// TIA Portal V17 export
// export: Created 2025-07-01T14:25:34.6961243Z, ExportSetting WithDefaults, DisplayName Totally Integrated Automation Portal, DisplayVersion V17 Update 8, DisplayName TIA Portal Openness, DisplayVersion V17 Update 8, DisplayName TIA Portal Version Control Interface, DisplayVersion V17, DisplayName SINAMICS Startdrive Advanced, DisplayVersion V17 SP2, DisplayName SINAMICS Startdrive G110M, G120, G120C, G120D, G120P, G115D, DisplayVersion V17 SP2, DisplayName SINAMICS Startdrive G130, G150, S120, S150, SINAMICS MV, S210, DisplayVersion V17 SP2, DisplayName STEP 7 Professional, DisplayVersion V17 Update 8, DisplayName SINUMERIK ONE STEP 7 Toolbox, DisplayVersion V17 Update 12, DisplayName SINUMERIK ONE PLC Basic Program Plus, DisplayVersion V17 Update 12, DisplayName SINUMERIK 840D sl STEP 7 Toolbox, DisplayVersion V17 Update 12, DisplayName STEP 7 Safety, DisplayVersion V17 Update 6, DisplayName WinCC Advanced, DisplayVersion V17 Update 8
FUNCTION "FC342_NCK_M_CH1_UNIT_1_STA_0" : Void   // FC342, LAD
TITLE = Channel 1 data
{ S7_Optimized_Access := 'FALSE' }
AUTHOR : ETXETAR
VERSION : 1.0
// stored: AutoNumber false, IsIECCheckEnabled false, SetENOAutomatically false, UDAEnableTagReadback false
BEGIN

REGION Network 1: ACKNOWLEDGE M404-UNIT 1 FIXTURE 1 VERIFY PART AND TOOL IS CLAMPED DURING MACHINING (WHEN TRUE DO). TOGGLED / ACKNOWLEDGE M46-VERIFY FIXTURE 1 PART AND TOOL IS CLAMPED DURING
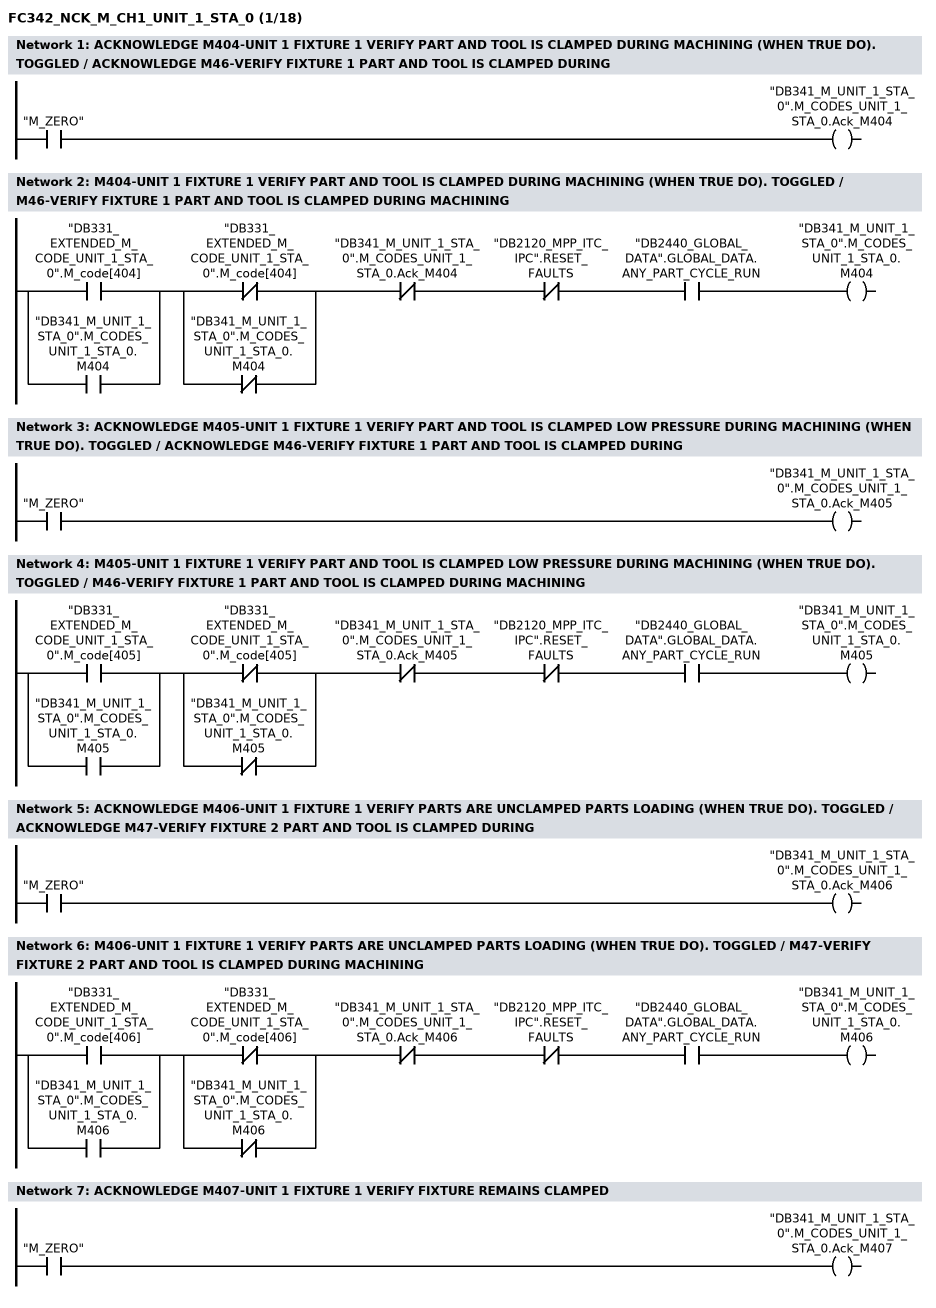
   RUNG wire#powerrail
      Contact( "M_ZERO" )
      Coil( "DB341_M_UNIT_1_STA_0".M_CODES_UNIT_1_STA_0.Ack_M404 )
   END_RUNG
   // the same network as SCL:
   "DB341_M_UNIT_1_STA_0".M_CODES_UNIT_1_STA_0.Ack_M404 := "M_ZERO";
END_REGION

REGION Network 2: M404-UNIT 1 FIXTURE 1 VERIFY PART AND TOOL IS CLAMPED DURING MACHINING (WHEN TRUE DO). TOGGLED / M46-VERIFY FIXTURE 1 PART AND TOOL IS CLAMPED DURING MACHINING
   RUNG wire#powerrail
      Contact( "DB331_EXTENDED_M_CODE_UNIT_1_STA_0".M_code[404] )
      wire#w1
      I_Contact( "DB331_EXTENDED_M_CODE_UNIT_1_STA_0".M_code[404] )
      wire#w2
      I_Contact( "DB341_M_UNIT_1_STA_0".M_CODES_UNIT_1_STA_0.Ack_M404 )
      I_Contact( "DB2120_MPP_ITC_IPC".RESET_FAULTS )
      Contact( "DB2440_GLOBAL_DATA".GLOBAL_DATA.ANY_PART_CYCLE_RUN )
      Coil( "DB341_M_UNIT_1_STA_0".M_CODES_UNIT_1_STA_0.M404 )
   END_RUNG
   RUNG wire#powerrail
      Contact( "DB341_M_UNIT_1_STA_0".M_CODES_UNIT_1_STA_0.M404 )
   END_RUNG wire#w1
   RUNG wire#w1
      I_Contact( "DB341_M_UNIT_1_STA_0".M_CODES_UNIT_1_STA_0.M404 )
   END_RUNG wire#w2
   // the same network as SCL:
   "DB341_M_UNIT_1_STA_0".M_CODES_UNIT_1_STA_0.M404 := ("DB331_EXTENDED_M_CODE_UNIT_1_STA_0".M_code[404] OR "DB341_M_UNIT_1_STA_0".M_CODES_UNIT_1_STA_0.M404) AND (NOT "DB331_EXTENDED_M_CODE_UNIT_1_STA_0".M_code[404] OR NOT "DB341_M_UNIT_1_STA_0".M_CODES_UNIT_1_STA_0.M404) AND NOT "DB341_M_UNIT_1_STA_0".M_CODES_UNIT_1_STA_0.Ack_M404 AND NOT "DB2120_MPP_ITC_IPC".RESET_FAULTS AND "DB2440_GLOBAL_DATA".GLOBAL_DATA.ANY_PART_CYCLE_RUN;
END_REGION

REGION Network 3: ACKNOWLEDGE M405-UNIT 1 FIXTURE 1 VERIFY PART AND TOOL IS CLAMPED LOW PRESSURE DURING MACHINING (WHEN TRUE DO). TOGGLED / ACKNOWLEDGE M46-VERIFY FIXTURE 1 PART AND TOOL IS CLAMPED DURING
   RUNG wire#powerrail
      Contact( "M_ZERO" )
      Coil( "DB341_M_UNIT_1_STA_0".M_CODES_UNIT_1_STA_0.Ack_M405 )
   END_RUNG
   // the same network as SCL:
   "DB341_M_UNIT_1_STA_0".M_CODES_UNIT_1_STA_0.Ack_M405 := "M_ZERO";
END_REGION

REGION Network 4: M405-UNIT 1 FIXTURE 1 VERIFY PART AND TOOL IS CLAMPED LOW PRESSURE DURING MACHINING (WHEN TRUE DO). TOGGLED / M46-VERIFY FIXTURE 1 PART AND TOOL IS CLAMPED DURING MACHINING
   RUNG wire#powerrail
      Contact( "DB331_EXTENDED_M_CODE_UNIT_1_STA_0".M_code[405] )
      wire#w1
      I_Contact( "DB331_EXTENDED_M_CODE_UNIT_1_STA_0".M_code[405] )
      wire#w2
      I_Contact( "DB341_M_UNIT_1_STA_0".M_CODES_UNIT_1_STA_0.Ack_M405 )
      I_Contact( "DB2120_MPP_ITC_IPC".RESET_FAULTS )
      Contact( "DB2440_GLOBAL_DATA".GLOBAL_DATA.ANY_PART_CYCLE_RUN )
      Coil( "DB341_M_UNIT_1_STA_0".M_CODES_UNIT_1_STA_0.M405 )
   END_RUNG
   RUNG wire#powerrail
      Contact( "DB341_M_UNIT_1_STA_0".M_CODES_UNIT_1_STA_0.M405 )
   END_RUNG wire#w1
   RUNG wire#w1
      I_Contact( "DB341_M_UNIT_1_STA_0".M_CODES_UNIT_1_STA_0.M405 )
   END_RUNG wire#w2
   // the same network as SCL:
   "DB341_M_UNIT_1_STA_0".M_CODES_UNIT_1_STA_0.M405 := ("DB331_EXTENDED_M_CODE_UNIT_1_STA_0".M_code[405] OR "DB341_M_UNIT_1_STA_0".M_CODES_UNIT_1_STA_0.M405) AND (NOT "DB331_EXTENDED_M_CODE_UNIT_1_STA_0".M_code[405] OR NOT "DB341_M_UNIT_1_STA_0".M_CODES_UNIT_1_STA_0.M405) AND NOT "DB341_M_UNIT_1_STA_0".M_CODES_UNIT_1_STA_0.Ack_M405 AND NOT "DB2120_MPP_ITC_IPC".RESET_FAULTS AND "DB2440_GLOBAL_DATA".GLOBAL_DATA.ANY_PART_CYCLE_RUN;
END_REGION

REGION Network 5: ACKNOWLEDGE M406-UNIT 1 FIXTURE 1 VERIFY PARTS ARE UNCLAMPED PARTS LOADING (WHEN TRUE DO). TOGGLED / ACKNOWLEDGE M47-VERIFY FIXTURE 2 PART AND TOOL IS CLAMPED DURING
   RUNG wire#powerrail
      Contact( "M_ZERO" )
      Coil( "DB341_M_UNIT_1_STA_0".M_CODES_UNIT_1_STA_0.Ack_M406 )
   END_RUNG
   // the same network as SCL:
   "DB341_M_UNIT_1_STA_0".M_CODES_UNIT_1_STA_0.Ack_M406 := "M_ZERO";
END_REGION

REGION Network 6: M406-UNIT 1 FIXTURE 1 VERIFY PARTS ARE UNCLAMPED PARTS LOADING (WHEN TRUE DO). TOGGLED / M47-VERIFY FIXTURE 2 PART AND TOOL IS CLAMPED DURING MACHINING
   RUNG wire#powerrail
      Contact( "DB331_EXTENDED_M_CODE_UNIT_1_STA_0".M_code[406] )
      wire#w1
      I_Contact( "DB331_EXTENDED_M_CODE_UNIT_1_STA_0".M_code[406] )
      wire#w2
      I_Contact( "DB341_M_UNIT_1_STA_0".M_CODES_UNIT_1_STA_0.Ack_M406 )
      I_Contact( "DB2120_MPP_ITC_IPC".RESET_FAULTS )
      Contact( "DB2440_GLOBAL_DATA".GLOBAL_DATA.ANY_PART_CYCLE_RUN )
      Coil( "DB341_M_UNIT_1_STA_0".M_CODES_UNIT_1_STA_0.M406 )
   END_RUNG
   RUNG wire#powerrail
      Contact( "DB341_M_UNIT_1_STA_0".M_CODES_UNIT_1_STA_0.M406 )
   END_RUNG wire#w1
   RUNG wire#w1
      I_Contact( "DB341_M_UNIT_1_STA_0".M_CODES_UNIT_1_STA_0.M406 )
   END_RUNG wire#w2
   // the same network as SCL:
   "DB341_M_UNIT_1_STA_0".M_CODES_UNIT_1_STA_0.M406 := ("DB331_EXTENDED_M_CODE_UNIT_1_STA_0".M_code[406] OR "DB341_M_UNIT_1_STA_0".M_CODES_UNIT_1_STA_0.M406) AND (NOT "DB331_EXTENDED_M_CODE_UNIT_1_STA_0".M_code[406] OR NOT "DB341_M_UNIT_1_STA_0".M_CODES_UNIT_1_STA_0.M406) AND NOT "DB341_M_UNIT_1_STA_0".M_CODES_UNIT_1_STA_0.Ack_M406 AND NOT "DB2120_MPP_ITC_IPC".RESET_FAULTS AND "DB2440_GLOBAL_DATA".GLOBAL_DATA.ANY_PART_CYCLE_RUN;
END_REGION

REGION Network 7: ACKNOWLEDGE M407-UNIT 1 FIXTURE 1 VERIFY FIXTURE REMAINS CLAMPED
   RUNG wire#powerrail
      Contact( "M_ZERO" )
      Coil( "DB341_M_UNIT_1_STA_0".M_CODES_UNIT_1_STA_0.Ack_M407 )
   END_RUNG
   // the same network as SCL:
   "DB341_M_UNIT_1_STA_0".M_CODES_UNIT_1_STA_0.Ack_M407 := "M_ZERO";
END_REGION

REGION Network 8: M407-UNIT 1 FIXTURE 1 VERIFY FIXTURE REMAINS CLAMPED
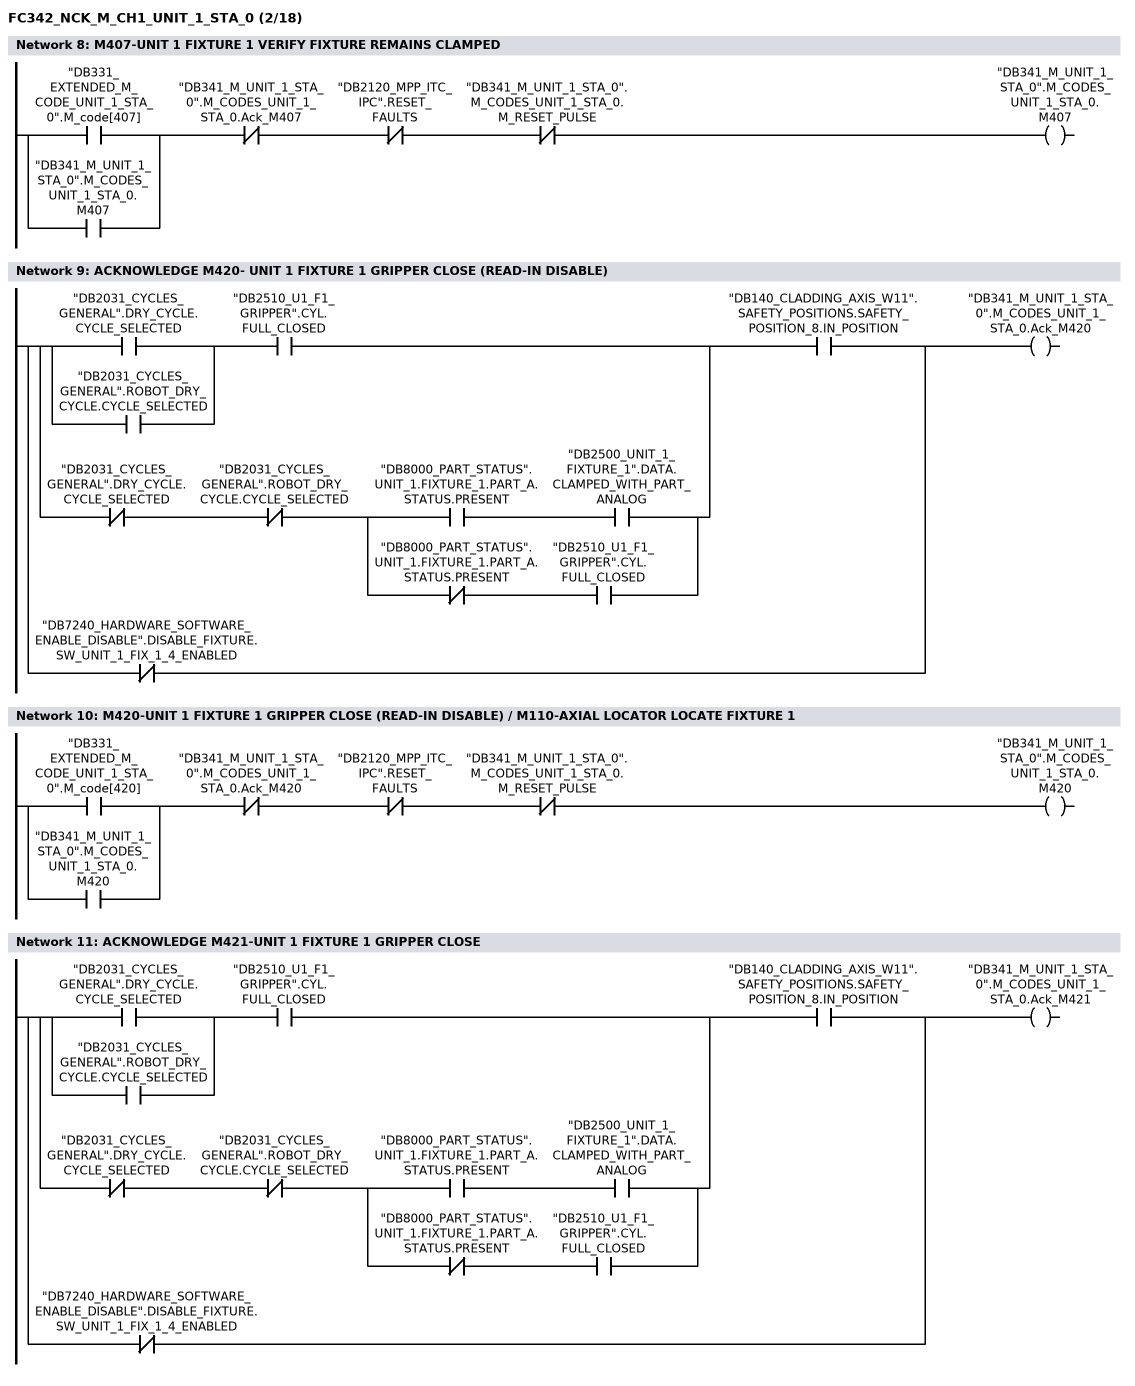
   RUNG wire#powerrail
      Contact( "DB331_EXTENDED_M_CODE_UNIT_1_STA_0".M_code[407] )
      wire#w1
      I_Contact( "DB341_M_UNIT_1_STA_0".M_CODES_UNIT_1_STA_0.Ack_M407 )
      I_Contact( "DB2120_MPP_ITC_IPC".RESET_FAULTS )
      I_Contact( "DB341_M_UNIT_1_STA_0".M_CODES_UNIT_1_STA_0.M_RESET_PULSE )
      Coil( "DB341_M_UNIT_1_STA_0".M_CODES_UNIT_1_STA_0.M407 )
   END_RUNG
   RUNG wire#powerrail
      Contact( "DB341_M_UNIT_1_STA_0".M_CODES_UNIT_1_STA_0.M407 )
   END_RUNG wire#w1
   // the same network as SCL:
   "DB341_M_UNIT_1_STA_0".M_CODES_UNIT_1_STA_0.M407 := ("DB331_EXTENDED_M_CODE_UNIT_1_STA_0".M_code[407] OR "DB341_M_UNIT_1_STA_0".M_CODES_UNIT_1_STA_0.M407) AND NOT "DB341_M_UNIT_1_STA_0".M_CODES_UNIT_1_STA_0.Ack_M407 AND NOT "DB2120_MPP_ITC_IPC".RESET_FAULTS AND NOT "DB341_M_UNIT_1_STA_0".M_CODES_UNIT_1_STA_0.M_RESET_PULSE;
END_REGION

REGION Network 9: ACKNOWLEDGE M420- UNIT 1 FIXTURE 1 GRIPPER CLOSE (READ-IN DISABLE)
   RUNG wire#powerrail
      Contact( "DB2031_CYCLES_GENERAL".DRY_CYCLE.CYCLE_SELECTED )
      wire#w1
      Contact( "DB2510_U1_F1_GRIPPER".CYL.FULL_CLOSED )
      wire#w2
      Contact( "DB140_CLADDING_AXIS_W11".SAFETY_POSITIONS.SAFETY_POSITION_8.IN_POSITION )
      wire#w4
      Coil( "DB341_M_UNIT_1_STA_0".M_CODES_UNIT_1_STA_0.Ack_M420 )
   END_RUNG
   RUNG wire#powerrail
      Contact( "DB2031_CYCLES_GENERAL".ROBOT_DRY_CYCLE.CYCLE_SELECTED )
   END_RUNG wire#w1
   RUNG wire#powerrail
      I_Contact( "DB2031_CYCLES_GENERAL".DRY_CYCLE.CYCLE_SELECTED )
      I_Contact( "DB2031_CYCLES_GENERAL".ROBOT_DRY_CYCLE.CYCLE_SELECTED )
      wire#w3
      Contact( "DB8000_PART_STATUS".UNIT_1.FIXTURE_1.PART_A.STATUS.PRESENT )
      Contact( "DB2500_UNIT_1_FIXTURE_1".DATA.CLAMPED_WITH_PART_ANALOG )
   END_RUNG wire#w2
   RUNG wire#w3
      I_Contact( "DB8000_PART_STATUS".UNIT_1.FIXTURE_1.PART_A.STATUS.PRESENT )
      Contact( "DB2510_U1_F1_GRIPPER".CYL.FULL_CLOSED )
   END_RUNG wire#w2
   RUNG wire#powerrail
      I_Contact( "DB7240_HARDWARE_SOFTWARE_ENABLE_DISABLE".DISABLE_FIXTURE.SW_UNIT_1_FIX_1_4_ENABLED )
   END_RUNG wire#w4
   // the same network as SCL:
   "DB341_M_UNIT_1_STA_0".M_CODES_UNIT_1_STA_0.Ack_M420 := (((("DB2031_CYCLES_GENERAL".DRY_CYCLE.CYCLE_SELECTED OR "DB2031_CYCLES_GENERAL".ROBOT_DRY_CYCLE.CYCLE_SELECTED) AND "DB2510_U1_F1_GRIPPER".CYL.FULL_CLOSED) OR (NOT "DB2031_CYCLES_GENERAL".DRY_CYCLE.CYCLE_SELECTED AND NOT "DB2031_CYCLES_GENERAL".ROBOT_DRY_CYCLE.CYCLE_SELECTED AND (("DB8000_PART_STATUS".UNIT_1.FIXTURE_1.PART_A.STATUS.PRESENT AND "DB2500_UNIT_1_FIXTURE_1".DATA.CLAMPED_WITH_PART_ANALOG) OR (NOT "DB8000_PART_STATUS".UNIT_1.FIXTURE_1.PART_A.STATUS.PRESENT AND "DB2510_U1_F1_GRIPPER".CYL.FULL_CLOSED)))) AND "DB140_CLADDING_AXIS_W11".SAFETY_POSITIONS.SAFETY_POSITION_8.IN_POSITION) OR NOT "DB7240_HARDWARE_SOFTWARE_ENABLE_DISABLE".DISABLE_FIXTURE.SW_UNIT_1_FIX_1_4_ENABLED;
END_REGION

REGION Network 10: M420-UNIT 1 FIXTURE 1 GRIPPER CLOSE (READ-IN DISABLE) / M110-AXIAL LOCATOR LOCATE FIXTURE 1
   RUNG wire#powerrail
      Contact( "DB331_EXTENDED_M_CODE_UNIT_1_STA_0".M_code[420] )
      wire#w1
      I_Contact( "DB341_M_UNIT_1_STA_0".M_CODES_UNIT_1_STA_0.Ack_M420 )
      I_Contact( "DB2120_MPP_ITC_IPC".RESET_FAULTS )
      I_Contact( "DB341_M_UNIT_1_STA_0".M_CODES_UNIT_1_STA_0.M_RESET_PULSE )
      Coil( "DB341_M_UNIT_1_STA_0".M_CODES_UNIT_1_STA_0.M420 )
   END_RUNG
   RUNG wire#powerrail
      Contact( "DB341_M_UNIT_1_STA_0".M_CODES_UNIT_1_STA_0.M420 )
   END_RUNG wire#w1
   // the same network as SCL:
   "DB341_M_UNIT_1_STA_0".M_CODES_UNIT_1_STA_0.M420 := ("DB331_EXTENDED_M_CODE_UNIT_1_STA_0".M_code[420] OR "DB341_M_UNIT_1_STA_0".M_CODES_UNIT_1_STA_0.M420) AND NOT "DB341_M_UNIT_1_STA_0".M_CODES_UNIT_1_STA_0.Ack_M420 AND NOT "DB2120_MPP_ITC_IPC".RESET_FAULTS AND NOT "DB341_M_UNIT_1_STA_0".M_CODES_UNIT_1_STA_0.M_RESET_PULSE;
END_REGION

REGION Network 11: ACKNOWLEDGE M421-UNIT 1 FIXTURE 1 GRIPPER CLOSE
   RUNG wire#powerrail
      Contact( "DB2031_CYCLES_GENERAL".DRY_CYCLE.CYCLE_SELECTED )
      wire#w1
      Contact( "DB2510_U1_F1_GRIPPER".CYL.FULL_CLOSED )
      wire#w2
      Contact( "DB140_CLADDING_AXIS_W11".SAFETY_POSITIONS.SAFETY_POSITION_8.IN_POSITION )
      wire#w4
      Coil( "DB341_M_UNIT_1_STA_0".M_CODES_UNIT_1_STA_0.Ack_M421 )
   END_RUNG
   RUNG wire#powerrail
      Contact( "DB2031_CYCLES_GENERAL".ROBOT_DRY_CYCLE.CYCLE_SELECTED )
   END_RUNG wire#w1
   RUNG wire#powerrail
      I_Contact( "DB2031_CYCLES_GENERAL".DRY_CYCLE.CYCLE_SELECTED )
      I_Contact( "DB2031_CYCLES_GENERAL".ROBOT_DRY_CYCLE.CYCLE_SELECTED )
      wire#w3
      Contact( "DB8000_PART_STATUS".UNIT_1.FIXTURE_1.PART_A.STATUS.PRESENT )
      Contact( "DB2500_UNIT_1_FIXTURE_1".DATA.CLAMPED_WITH_PART_ANALOG )
   END_RUNG wire#w2
   RUNG wire#w3
      I_Contact( "DB8000_PART_STATUS".UNIT_1.FIXTURE_1.PART_A.STATUS.PRESENT )
      Contact( "DB2510_U1_F1_GRIPPER".CYL.FULL_CLOSED )
   END_RUNG wire#w2
   RUNG wire#powerrail
      I_Contact( "DB7240_HARDWARE_SOFTWARE_ENABLE_DISABLE".DISABLE_FIXTURE.SW_UNIT_1_FIX_1_4_ENABLED )
   END_RUNG wire#w4
   // the same network as SCL:
   "DB341_M_UNIT_1_STA_0".M_CODES_UNIT_1_STA_0.Ack_M421 := (((("DB2031_CYCLES_GENERAL".DRY_CYCLE.CYCLE_SELECTED OR "DB2031_CYCLES_GENERAL".ROBOT_DRY_CYCLE.CYCLE_SELECTED) AND "DB2510_U1_F1_GRIPPER".CYL.FULL_CLOSED) OR (NOT "DB2031_CYCLES_GENERAL".DRY_CYCLE.CYCLE_SELECTED AND NOT "DB2031_CYCLES_GENERAL".ROBOT_DRY_CYCLE.CYCLE_SELECTED AND (("DB8000_PART_STATUS".UNIT_1.FIXTURE_1.PART_A.STATUS.PRESENT AND "DB2500_UNIT_1_FIXTURE_1".DATA.CLAMPED_WITH_PART_ANALOG) OR (NOT "DB8000_PART_STATUS".UNIT_1.FIXTURE_1.PART_A.STATUS.PRESENT AND "DB2510_U1_F1_GRIPPER".CYL.FULL_CLOSED)))) AND "DB140_CLADDING_AXIS_W11".SAFETY_POSITIONS.SAFETY_POSITION_8.IN_POSITION) OR NOT "DB7240_HARDWARE_SOFTWARE_ENABLE_DISABLE".DISABLE_FIXTURE.SW_UNIT_1_FIX_1_4_ENABLED;
END_REGION

REGION Network 12: M421-UNIT 1 FIXTURE 1 GRIPPER CLOSE / M110-AXIAL LOCATOR LOCATE FIXTURE 1
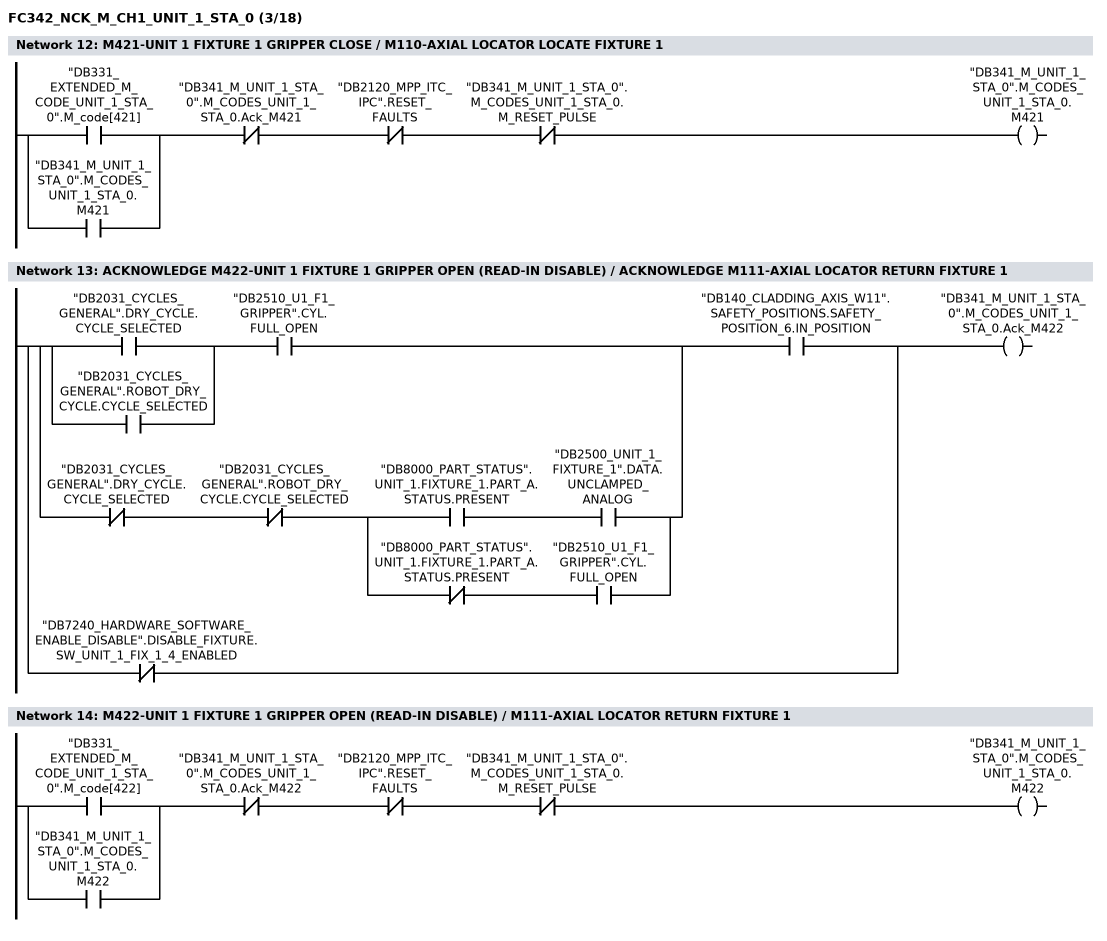
   RUNG wire#powerrail
      Contact( "DB331_EXTENDED_M_CODE_UNIT_1_STA_0".M_code[421] )
      wire#w1
      I_Contact( "DB341_M_UNIT_1_STA_0".M_CODES_UNIT_1_STA_0.Ack_M421 )
      I_Contact( "DB2120_MPP_ITC_IPC".RESET_FAULTS )
      I_Contact( "DB341_M_UNIT_1_STA_0".M_CODES_UNIT_1_STA_0.M_RESET_PULSE )
      Coil( "DB341_M_UNIT_1_STA_0".M_CODES_UNIT_1_STA_0.M421 )
   END_RUNG
   RUNG wire#powerrail
      Contact( "DB341_M_UNIT_1_STA_0".M_CODES_UNIT_1_STA_0.M421 )
   END_RUNG wire#w1
   // the same network as SCL:
   "DB341_M_UNIT_1_STA_0".M_CODES_UNIT_1_STA_0.M421 := ("DB331_EXTENDED_M_CODE_UNIT_1_STA_0".M_code[421] OR "DB341_M_UNIT_1_STA_0".M_CODES_UNIT_1_STA_0.M421) AND NOT "DB341_M_UNIT_1_STA_0".M_CODES_UNIT_1_STA_0.Ack_M421 AND NOT "DB2120_MPP_ITC_IPC".RESET_FAULTS AND NOT "DB341_M_UNIT_1_STA_0".M_CODES_UNIT_1_STA_0.M_RESET_PULSE;
END_REGION

REGION Network 13: ACKNOWLEDGE M422-UNIT 1 FIXTURE 1 GRIPPER OPEN (READ-IN DISABLE) / ACKNOWLEDGE M111-AXIAL LOCATOR RETURN FIXTURE 1
   RUNG wire#powerrail
      Contact( "DB2031_CYCLES_GENERAL".DRY_CYCLE.CYCLE_SELECTED )
      wire#w1
      Contact( "DB2510_U1_F1_GRIPPER".CYL.FULL_OPEN )
      wire#w2
      Contact( "DB140_CLADDING_AXIS_W11".SAFETY_POSITIONS.SAFETY_POSITION_6.IN_POSITION )
      wire#w4
      Coil( "DB341_M_UNIT_1_STA_0".M_CODES_UNIT_1_STA_0.Ack_M422 )
   END_RUNG
   RUNG wire#powerrail
      Contact( "DB2031_CYCLES_GENERAL".ROBOT_DRY_CYCLE.CYCLE_SELECTED )
   END_RUNG wire#w1
   RUNG wire#powerrail
      I_Contact( "DB2031_CYCLES_GENERAL".DRY_CYCLE.CYCLE_SELECTED )
      I_Contact( "DB2031_CYCLES_GENERAL".ROBOT_DRY_CYCLE.CYCLE_SELECTED )
      wire#w3
      Contact( "DB8000_PART_STATUS".UNIT_1.FIXTURE_1.PART_A.STATUS.PRESENT )
      Contact( "DB2500_UNIT_1_FIXTURE_1".DATA.UNCLAMPED_ANALOG )
   END_RUNG wire#w2
   RUNG wire#w3
      I_Contact( "DB8000_PART_STATUS".UNIT_1.FIXTURE_1.PART_A.STATUS.PRESENT )
      Contact( "DB2510_U1_F1_GRIPPER".CYL.FULL_OPEN )
   END_RUNG wire#w2
   RUNG wire#powerrail
      I_Contact( "DB7240_HARDWARE_SOFTWARE_ENABLE_DISABLE".DISABLE_FIXTURE.SW_UNIT_1_FIX_1_4_ENABLED )
   END_RUNG wire#w4
   // the same network as SCL:
   "DB341_M_UNIT_1_STA_0".M_CODES_UNIT_1_STA_0.Ack_M422 := (((("DB2031_CYCLES_GENERAL".DRY_CYCLE.CYCLE_SELECTED OR "DB2031_CYCLES_GENERAL".ROBOT_DRY_CYCLE.CYCLE_SELECTED) AND "DB2510_U1_F1_GRIPPER".CYL.FULL_OPEN) OR (NOT "DB2031_CYCLES_GENERAL".DRY_CYCLE.CYCLE_SELECTED AND NOT "DB2031_CYCLES_GENERAL".ROBOT_DRY_CYCLE.CYCLE_SELECTED AND (("DB8000_PART_STATUS".UNIT_1.FIXTURE_1.PART_A.STATUS.PRESENT AND "DB2500_UNIT_1_FIXTURE_1".DATA.UNCLAMPED_ANALOG) OR (NOT "DB8000_PART_STATUS".UNIT_1.FIXTURE_1.PART_A.STATUS.PRESENT AND "DB2510_U1_F1_GRIPPER".CYL.FULL_OPEN)))) AND "DB140_CLADDING_AXIS_W11".SAFETY_POSITIONS.SAFETY_POSITION_6.IN_POSITION) OR NOT "DB7240_HARDWARE_SOFTWARE_ENABLE_DISABLE".DISABLE_FIXTURE.SW_UNIT_1_FIX_1_4_ENABLED;
END_REGION

REGION Network 14: M422-UNIT 1 FIXTURE 1 GRIPPER OPEN (READ-IN DISABLE) / M111-AXIAL LOCATOR RETURN FIXTURE 1
   RUNG wire#powerrail
      Contact( "DB331_EXTENDED_M_CODE_UNIT_1_STA_0".M_code[422] )
      wire#w1
      I_Contact( "DB341_M_UNIT_1_STA_0".M_CODES_UNIT_1_STA_0.Ack_M422 )
      I_Contact( "DB2120_MPP_ITC_IPC".RESET_FAULTS )
      I_Contact( "DB341_M_UNIT_1_STA_0".M_CODES_UNIT_1_STA_0.M_RESET_PULSE )
      Coil( "DB341_M_UNIT_1_STA_0".M_CODES_UNIT_1_STA_0.M422 )
   END_RUNG
   RUNG wire#powerrail
      Contact( "DB341_M_UNIT_1_STA_0".M_CODES_UNIT_1_STA_0.M422 )
   END_RUNG wire#w1
   // the same network as SCL:
   "DB341_M_UNIT_1_STA_0".M_CODES_UNIT_1_STA_0.M422 := ("DB331_EXTENDED_M_CODE_UNIT_1_STA_0".M_code[422] OR "DB341_M_UNIT_1_STA_0".M_CODES_UNIT_1_STA_0.M422) AND NOT "DB341_M_UNIT_1_STA_0".M_CODES_UNIT_1_STA_0.Ack_M422 AND NOT "DB2120_MPP_ITC_IPC".RESET_FAULTS AND NOT "DB341_M_UNIT_1_STA_0".M_CODES_UNIT_1_STA_0.M_RESET_PULSE;
END_REGION

REGION Network 15: ACKNOWLEDGE M423-UNIT 1 FIXTURE 1 GRIPPER OPEN / ACKNOWLEDGE M111-AXIAL LOCATOR RETURN FIXTURE 1
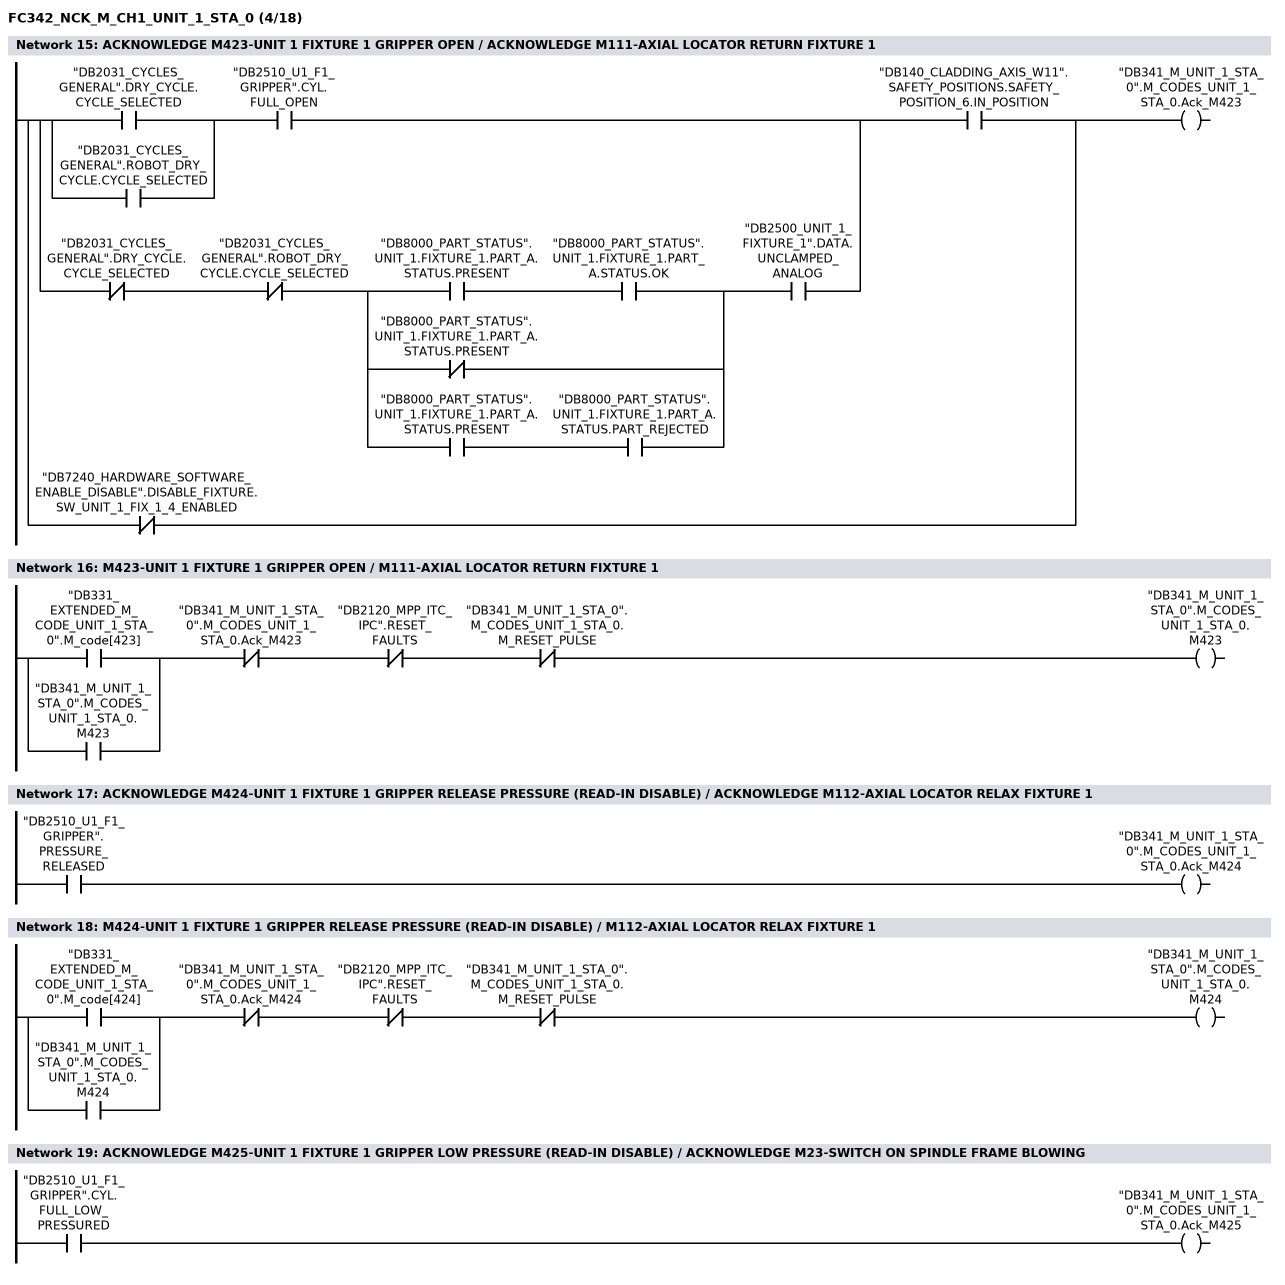
   RUNG wire#powerrail
      Contact( "DB2031_CYCLES_GENERAL".DRY_CYCLE.CYCLE_SELECTED )
      wire#w1
      Contact( "DB2510_U1_F1_GRIPPER".CYL.FULL_OPEN )
      wire#w2
      Contact( "DB140_CLADDING_AXIS_W11".SAFETY_POSITIONS.SAFETY_POSITION_6.IN_POSITION )
      wire#w5
      Coil( "DB341_M_UNIT_1_STA_0".M_CODES_UNIT_1_STA_0.Ack_M423 )
   END_RUNG
   RUNG wire#powerrail
      Contact( "DB2031_CYCLES_GENERAL".ROBOT_DRY_CYCLE.CYCLE_SELECTED )
   END_RUNG wire#w1
   RUNG wire#powerrail
      I_Contact( "DB2031_CYCLES_GENERAL".DRY_CYCLE.CYCLE_SELECTED )
      I_Contact( "DB2031_CYCLES_GENERAL".ROBOT_DRY_CYCLE.CYCLE_SELECTED )
      wire#w3
      Contact( "DB8000_PART_STATUS".UNIT_1.FIXTURE_1.PART_A.STATUS.PRESENT )
      Contact( "DB8000_PART_STATUS".UNIT_1.FIXTURE_1.PART_A.STATUS.OK )
      wire#w4
      Contact( "DB2500_UNIT_1_FIXTURE_1".DATA.UNCLAMPED_ANALOG )
   END_RUNG wire#w2
   RUNG wire#w3
      I_Contact( "DB8000_PART_STATUS".UNIT_1.FIXTURE_1.PART_A.STATUS.PRESENT )
   END_RUNG wire#w4
   RUNG wire#w3
      Contact( "DB8000_PART_STATUS".UNIT_1.FIXTURE_1.PART_A.STATUS.PRESENT )
      Contact( "DB8000_PART_STATUS".UNIT_1.FIXTURE_1.PART_A.STATUS.PART_REJECTED )
   END_RUNG wire#w4
   RUNG wire#powerrail
      I_Contact( "DB7240_HARDWARE_SOFTWARE_ENABLE_DISABLE".DISABLE_FIXTURE.SW_UNIT_1_FIX_1_4_ENABLED )
   END_RUNG wire#w5
   // the same network as SCL:
   "DB341_M_UNIT_1_STA_0".M_CODES_UNIT_1_STA_0.Ack_M423 := (((("DB2031_CYCLES_GENERAL".DRY_CYCLE.CYCLE_SELECTED OR "DB2031_CYCLES_GENERAL".ROBOT_DRY_CYCLE.CYCLE_SELECTED) AND "DB2510_U1_F1_GRIPPER".CYL.FULL_OPEN) OR (NOT "DB2031_CYCLES_GENERAL".DRY_CYCLE.CYCLE_SELECTED AND NOT "DB2031_CYCLES_GENERAL".ROBOT_DRY_CYCLE.CYCLE_SELECTED AND (("DB8000_PART_STATUS".UNIT_1.FIXTURE_1.PART_A.STATUS.PRESENT AND "DB8000_PART_STATUS".UNIT_1.FIXTURE_1.PART_A.STATUS.OK) OR NOT "DB8000_PART_STATUS".UNIT_1.FIXTURE_1.PART_A.STATUS.PRESENT OR ("DB8000_PART_STATUS".UNIT_1.FIXTURE_1.PART_A.STATUS.PRESENT AND "DB8000_PART_STATUS".UNIT_1.FIXTURE_1.PART_A.STATUS.PART_REJECTED)) AND "DB2500_UNIT_1_FIXTURE_1".DATA.UNCLAMPED_ANALOG)) AND "DB140_CLADDING_AXIS_W11".SAFETY_POSITIONS.SAFETY_POSITION_6.IN_POSITION) OR NOT "DB7240_HARDWARE_SOFTWARE_ENABLE_DISABLE".DISABLE_FIXTURE.SW_UNIT_1_FIX_1_4_ENABLED;
END_REGION

REGION Network 16: M423-UNIT 1 FIXTURE 1 GRIPPER OPEN / M111-AXIAL LOCATOR RETURN FIXTURE 1
   RUNG wire#powerrail
      Contact( "DB331_EXTENDED_M_CODE_UNIT_1_STA_0".M_code[423] )
      wire#w1
      I_Contact( "DB341_M_UNIT_1_STA_0".M_CODES_UNIT_1_STA_0.Ack_M423 )
      I_Contact( "DB2120_MPP_ITC_IPC".RESET_FAULTS )
      I_Contact( "DB341_M_UNIT_1_STA_0".M_CODES_UNIT_1_STA_0.M_RESET_PULSE )
      Coil( "DB341_M_UNIT_1_STA_0".M_CODES_UNIT_1_STA_0.M423 )
   END_RUNG
   RUNG wire#powerrail
      Contact( "DB341_M_UNIT_1_STA_0".M_CODES_UNIT_1_STA_0.M423 )
   END_RUNG wire#w1
   // the same network as SCL:
   "DB341_M_UNIT_1_STA_0".M_CODES_UNIT_1_STA_0.M423 := ("DB331_EXTENDED_M_CODE_UNIT_1_STA_0".M_code[423] OR "DB341_M_UNIT_1_STA_0".M_CODES_UNIT_1_STA_0.M423) AND NOT "DB341_M_UNIT_1_STA_0".M_CODES_UNIT_1_STA_0.Ack_M423 AND NOT "DB2120_MPP_ITC_IPC".RESET_FAULTS AND NOT "DB341_M_UNIT_1_STA_0".M_CODES_UNIT_1_STA_0.M_RESET_PULSE;
END_REGION

REGION Network 17: ACKNOWLEDGE M424-UNIT 1 FIXTURE 1 GRIPPER RELEASE PRESSURE (READ-IN DISABLE) / ACKNOWLEDGE M112-AXIAL LOCATOR RELAX FIXTURE 1
   RUNG wire#powerrail
      Contact( "DB2510_U1_F1_GRIPPER".PRESSURE_RELEASED )
      Coil( "DB341_M_UNIT_1_STA_0".M_CODES_UNIT_1_STA_0.Ack_M424 )
   END_RUNG
   // the same network as SCL:
   "DB341_M_UNIT_1_STA_0".M_CODES_UNIT_1_STA_0.Ack_M424 := "DB2510_U1_F1_GRIPPER".PRESSURE_RELEASED;
END_REGION

REGION Network 18: M424-UNIT 1 FIXTURE 1 GRIPPER RELEASE PRESSURE (READ-IN DISABLE) / M112-AXIAL LOCATOR RELAX FIXTURE 1
   RUNG wire#powerrail
      Contact( "DB331_EXTENDED_M_CODE_UNIT_1_STA_0".M_code[424] )
      wire#w1
      I_Contact( "DB341_M_UNIT_1_STA_0".M_CODES_UNIT_1_STA_0.Ack_M424 )
      I_Contact( "DB2120_MPP_ITC_IPC".RESET_FAULTS )
      I_Contact( "DB341_M_UNIT_1_STA_0".M_CODES_UNIT_1_STA_0.M_RESET_PULSE )
      Coil( "DB341_M_UNIT_1_STA_0".M_CODES_UNIT_1_STA_0.M424 )
   END_RUNG
   RUNG wire#powerrail
      Contact( "DB341_M_UNIT_1_STA_0".M_CODES_UNIT_1_STA_0.M424 )
   END_RUNG wire#w1
   // the same network as SCL:
   "DB341_M_UNIT_1_STA_0".M_CODES_UNIT_1_STA_0.M424 := ("DB331_EXTENDED_M_CODE_UNIT_1_STA_0".M_code[424] OR "DB341_M_UNIT_1_STA_0".M_CODES_UNIT_1_STA_0.M424) AND NOT "DB341_M_UNIT_1_STA_0".M_CODES_UNIT_1_STA_0.Ack_M424 AND NOT "DB2120_MPP_ITC_IPC".RESET_FAULTS AND NOT "DB341_M_UNIT_1_STA_0".M_CODES_UNIT_1_STA_0.M_RESET_PULSE;
END_REGION

REGION Network 19: ACKNOWLEDGE M425-UNIT 1 FIXTURE 1 GRIPPER LOW PRESSURE (READ-IN DISABLE) / ACKNOWLEDGE M23-SWITCH ON SPINDLE FRAME BLOWING
   RUNG wire#powerrail
      Contact( "DB2510_U1_F1_GRIPPER".CYL.FULL_LOW_PRESSURED )
      Coil( "DB341_M_UNIT_1_STA_0".M_CODES_UNIT_1_STA_0.Ack_M425 )
   END_RUNG
   // the same network as SCL:
   "DB341_M_UNIT_1_STA_0".M_CODES_UNIT_1_STA_0.Ack_M425 := "DB2510_U1_F1_GRIPPER".CYL.FULL_LOW_PRESSURED;
END_REGION

REGION Network 20: M425-UNIT 1 FIXTURE 1 GRIPPER LOW PRESSURE (READ-IN DISABLE) / M23-SWITCH ON SPINDLE FRAME BLOWING
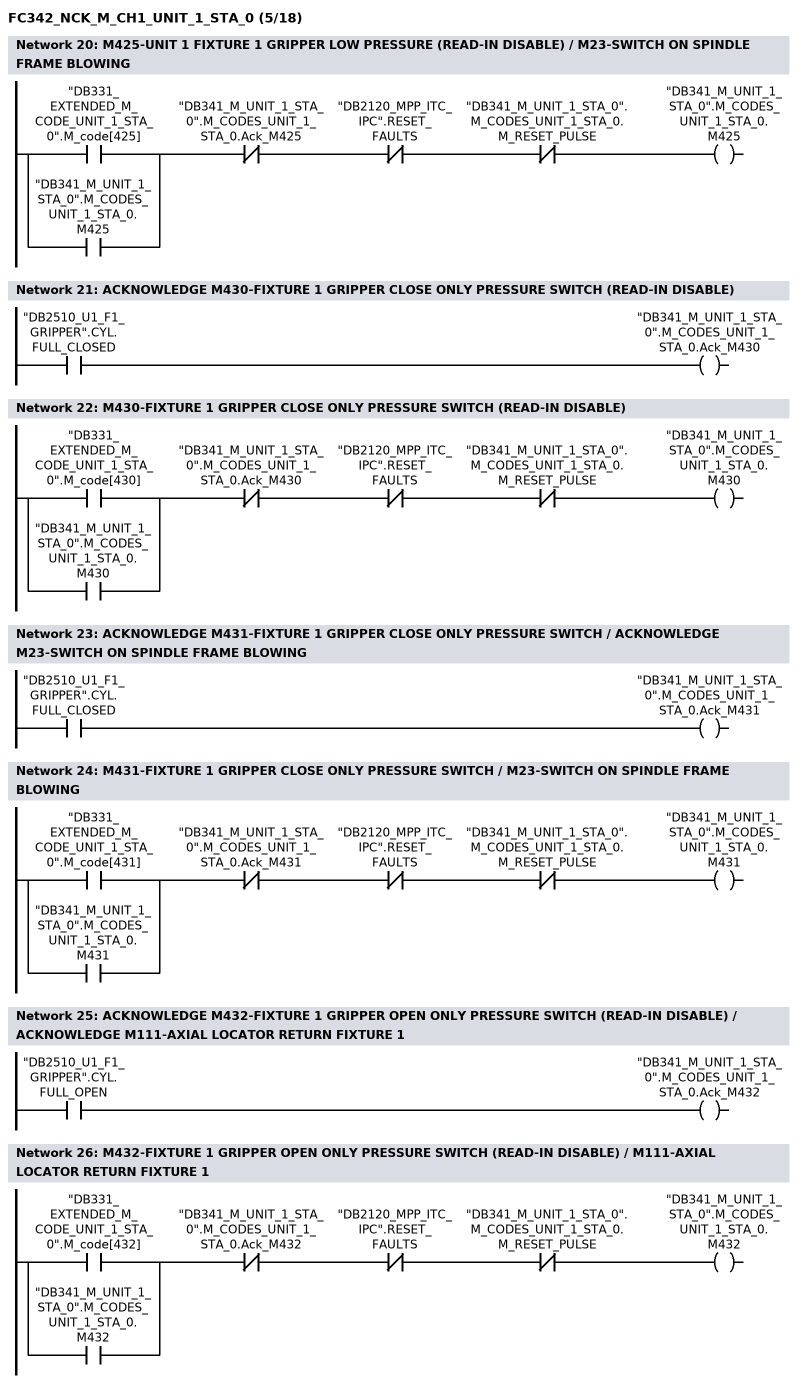
   RUNG wire#powerrail
      Contact( "DB331_EXTENDED_M_CODE_UNIT_1_STA_0".M_code[425] )
      wire#w1
      I_Contact( "DB341_M_UNIT_1_STA_0".M_CODES_UNIT_1_STA_0.Ack_M425 )
      I_Contact( "DB2120_MPP_ITC_IPC".RESET_FAULTS )
      I_Contact( "DB341_M_UNIT_1_STA_0".M_CODES_UNIT_1_STA_0.M_RESET_PULSE )
      Coil( "DB341_M_UNIT_1_STA_0".M_CODES_UNIT_1_STA_0.M425 )
   END_RUNG
   RUNG wire#powerrail
      Contact( "DB341_M_UNIT_1_STA_0".M_CODES_UNIT_1_STA_0.M425 )
   END_RUNG wire#w1
   // the same network as SCL:
   "DB341_M_UNIT_1_STA_0".M_CODES_UNIT_1_STA_0.M425 := ("DB331_EXTENDED_M_CODE_UNIT_1_STA_0".M_code[425] OR "DB341_M_UNIT_1_STA_0".M_CODES_UNIT_1_STA_0.M425) AND NOT "DB341_M_UNIT_1_STA_0".M_CODES_UNIT_1_STA_0.Ack_M425 AND NOT "DB2120_MPP_ITC_IPC".RESET_FAULTS AND NOT "DB341_M_UNIT_1_STA_0".M_CODES_UNIT_1_STA_0.M_RESET_PULSE;
END_REGION

REGION Network 21: ACKNOWLEDGE M430-FIXTURE 1 GRIPPER CLOSE ONLY PRESSURE SWITCH (READ-IN DISABLE)
   RUNG wire#powerrail
      Contact( "DB2510_U1_F1_GRIPPER".CYL.FULL_CLOSED )
      Coil( "DB341_M_UNIT_1_STA_0".M_CODES_UNIT_1_STA_0.Ack_M430 )
   END_RUNG
   // the same network as SCL:
   "DB341_M_UNIT_1_STA_0".M_CODES_UNIT_1_STA_0.Ack_M430 := "DB2510_U1_F1_GRIPPER".CYL.FULL_CLOSED;
END_REGION

REGION Network 22: M430-FIXTURE 1 GRIPPER CLOSE ONLY PRESSURE SWITCH (READ-IN DISABLE)
   RUNG wire#powerrail
      Contact( "DB331_EXTENDED_M_CODE_UNIT_1_STA_0".M_code[430] )
      wire#w1
      I_Contact( "DB341_M_UNIT_1_STA_0".M_CODES_UNIT_1_STA_0.Ack_M430 )
      I_Contact( "DB2120_MPP_ITC_IPC".RESET_FAULTS )
      I_Contact( "DB341_M_UNIT_1_STA_0".M_CODES_UNIT_1_STA_0.M_RESET_PULSE )
      Coil( "DB341_M_UNIT_1_STA_0".M_CODES_UNIT_1_STA_0.M430 )
   END_RUNG
   RUNG wire#powerrail
      Contact( "DB341_M_UNIT_1_STA_0".M_CODES_UNIT_1_STA_0.M430 )
   END_RUNG wire#w1
   // the same network as SCL:
   "DB341_M_UNIT_1_STA_0".M_CODES_UNIT_1_STA_0.M430 := ("DB331_EXTENDED_M_CODE_UNIT_1_STA_0".M_code[430] OR "DB341_M_UNIT_1_STA_0".M_CODES_UNIT_1_STA_0.M430) AND NOT "DB341_M_UNIT_1_STA_0".M_CODES_UNIT_1_STA_0.Ack_M430 AND NOT "DB2120_MPP_ITC_IPC".RESET_FAULTS AND NOT "DB341_M_UNIT_1_STA_0".M_CODES_UNIT_1_STA_0.M_RESET_PULSE;
END_REGION

REGION Network 23: ACKNOWLEDGE M431-FIXTURE 1 GRIPPER CLOSE ONLY PRESSURE SWITCH / ACKNOWLEDGE M23-SWITCH ON SPINDLE FRAME BLOWING
   RUNG wire#powerrail
      Contact( "DB2510_U1_F1_GRIPPER".CYL.FULL_CLOSED )
      Coil( "DB341_M_UNIT_1_STA_0".M_CODES_UNIT_1_STA_0.Ack_M431 )
   END_RUNG
   // the same network as SCL:
   "DB341_M_UNIT_1_STA_0".M_CODES_UNIT_1_STA_0.Ack_M431 := "DB2510_U1_F1_GRIPPER".CYL.FULL_CLOSED;
END_REGION

REGION Network 24: M431-FIXTURE 1 GRIPPER CLOSE ONLY PRESSURE SWITCH / M23-SWITCH ON SPINDLE FRAME BLOWING
   RUNG wire#powerrail
      Contact( "DB331_EXTENDED_M_CODE_UNIT_1_STA_0".M_code[431] )
      wire#w1
      I_Contact( "DB341_M_UNIT_1_STA_0".M_CODES_UNIT_1_STA_0.Ack_M431 )
      I_Contact( "DB2120_MPP_ITC_IPC".RESET_FAULTS )
      I_Contact( "DB341_M_UNIT_1_STA_0".M_CODES_UNIT_1_STA_0.M_RESET_PULSE )
      Coil( "DB341_M_UNIT_1_STA_0".M_CODES_UNIT_1_STA_0.M431 )
   END_RUNG
   RUNG wire#powerrail
      Contact( "DB341_M_UNIT_1_STA_0".M_CODES_UNIT_1_STA_0.M431 )
   END_RUNG wire#w1
   // the same network as SCL:
   "DB341_M_UNIT_1_STA_0".M_CODES_UNIT_1_STA_0.M431 := ("DB331_EXTENDED_M_CODE_UNIT_1_STA_0".M_code[431] OR "DB341_M_UNIT_1_STA_0".M_CODES_UNIT_1_STA_0.M431) AND NOT "DB341_M_UNIT_1_STA_0".M_CODES_UNIT_1_STA_0.Ack_M431 AND NOT "DB2120_MPP_ITC_IPC".RESET_FAULTS AND NOT "DB341_M_UNIT_1_STA_0".M_CODES_UNIT_1_STA_0.M_RESET_PULSE;
END_REGION

REGION Network 25: ACKNOWLEDGE M432-FIXTURE 1 GRIPPER OPEN ONLY PRESSURE SWITCH (READ-IN DISABLE) / ACKNOWLEDGE M111-AXIAL LOCATOR RETURN FIXTURE 1
   RUNG wire#powerrail
      Contact( "DB2510_U1_F1_GRIPPER".CYL.FULL_OPEN )
      Coil( "DB341_M_UNIT_1_STA_0".M_CODES_UNIT_1_STA_0.Ack_M432 )
   END_RUNG
   // the same network as SCL:
   "DB341_M_UNIT_1_STA_0".M_CODES_UNIT_1_STA_0.Ack_M432 := "DB2510_U1_F1_GRIPPER".CYL.FULL_OPEN;
END_REGION

REGION Network 26: M432-FIXTURE 1 GRIPPER OPEN ONLY PRESSURE SWITCH (READ-IN DISABLE) / M111-AXIAL LOCATOR RETURN FIXTURE 1
   RUNG wire#powerrail
      Contact( "DB331_EXTENDED_M_CODE_UNIT_1_STA_0".M_code[432] )
      wire#w1
      I_Contact( "DB341_M_UNIT_1_STA_0".M_CODES_UNIT_1_STA_0.Ack_M432 )
      I_Contact( "DB2120_MPP_ITC_IPC".RESET_FAULTS )
      I_Contact( "DB341_M_UNIT_1_STA_0".M_CODES_UNIT_1_STA_0.M_RESET_PULSE )
      Coil( "DB341_M_UNIT_1_STA_0".M_CODES_UNIT_1_STA_0.M432 )
   END_RUNG
   RUNG wire#powerrail
      Contact( "DB341_M_UNIT_1_STA_0".M_CODES_UNIT_1_STA_0.M432 )
   END_RUNG wire#w1
   // the same network as SCL:
   "DB341_M_UNIT_1_STA_0".M_CODES_UNIT_1_STA_0.M432 := ("DB331_EXTENDED_M_CODE_UNIT_1_STA_0".M_code[432] OR "DB341_M_UNIT_1_STA_0".M_CODES_UNIT_1_STA_0.M432) AND NOT "DB341_M_UNIT_1_STA_0".M_CODES_UNIT_1_STA_0.Ack_M432 AND NOT "DB2120_MPP_ITC_IPC".RESET_FAULTS AND NOT "DB341_M_UNIT_1_STA_0".M_CODES_UNIT_1_STA_0.M_RESET_PULSE;
END_REGION

REGION Network 27: ACKNOWLEDGE M433-FIXTURE 1 GRIPPER OPEN ONLY PRESSURE SWITCH / ACKNOWLEDGE M111-AXIAL LOCATOR RETURN FIXTURE 1
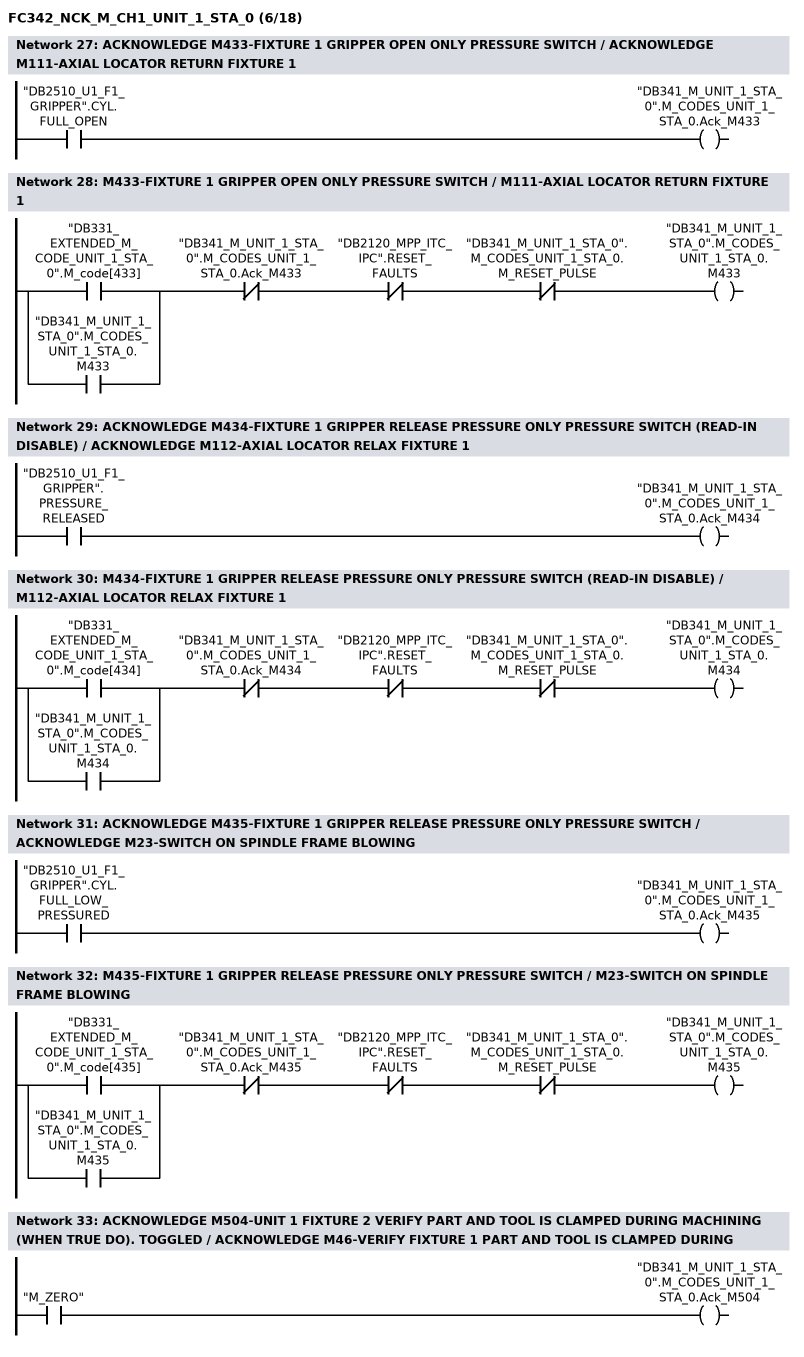
   RUNG wire#powerrail
      Contact( "DB2510_U1_F1_GRIPPER".CYL.FULL_OPEN )
      Coil( "DB341_M_UNIT_1_STA_0".M_CODES_UNIT_1_STA_0.Ack_M433 )
   END_RUNG
   // the same network as SCL:
   "DB341_M_UNIT_1_STA_0".M_CODES_UNIT_1_STA_0.Ack_M433 := "DB2510_U1_F1_GRIPPER".CYL.FULL_OPEN;
END_REGION

REGION Network 28: M433-FIXTURE 1 GRIPPER OPEN ONLY PRESSURE SWITCH / M111-AXIAL LOCATOR RETURN FIXTURE 1
   RUNG wire#powerrail
      Contact( "DB331_EXTENDED_M_CODE_UNIT_1_STA_0".M_code[433] )
      wire#w1
      I_Contact( "DB341_M_UNIT_1_STA_0".M_CODES_UNIT_1_STA_0.Ack_M433 )
      I_Contact( "DB2120_MPP_ITC_IPC".RESET_FAULTS )
      I_Contact( "DB341_M_UNIT_1_STA_0".M_CODES_UNIT_1_STA_0.M_RESET_PULSE )
      Coil( "DB341_M_UNIT_1_STA_0".M_CODES_UNIT_1_STA_0.M433 )
   END_RUNG
   RUNG wire#powerrail
      Contact( "DB341_M_UNIT_1_STA_0".M_CODES_UNIT_1_STA_0.M433 )
   END_RUNG wire#w1
   // the same network as SCL:
   "DB341_M_UNIT_1_STA_0".M_CODES_UNIT_1_STA_0.M433 := ("DB331_EXTENDED_M_CODE_UNIT_1_STA_0".M_code[433] OR "DB341_M_UNIT_1_STA_0".M_CODES_UNIT_1_STA_0.M433) AND NOT "DB341_M_UNIT_1_STA_0".M_CODES_UNIT_1_STA_0.Ack_M433 AND NOT "DB2120_MPP_ITC_IPC".RESET_FAULTS AND NOT "DB341_M_UNIT_1_STA_0".M_CODES_UNIT_1_STA_0.M_RESET_PULSE;
END_REGION

REGION Network 29: ACKNOWLEDGE M434-FIXTURE 1 GRIPPER RELEASE PRESSURE ONLY PRESSURE SWITCH (READ-IN DISABLE) / ACKNOWLEDGE M112-AXIAL LOCATOR RELAX FIXTURE 1
   RUNG wire#powerrail
      Contact( "DB2510_U1_F1_GRIPPER".PRESSURE_RELEASED )
      Coil( "DB341_M_UNIT_1_STA_0".M_CODES_UNIT_1_STA_0.Ack_M434 )
   END_RUNG
   // the same network as SCL:
   "DB341_M_UNIT_1_STA_0".M_CODES_UNIT_1_STA_0.Ack_M434 := "DB2510_U1_F1_GRIPPER".PRESSURE_RELEASED;
END_REGION

REGION Network 30: M434-FIXTURE 1 GRIPPER RELEASE PRESSURE ONLY PRESSURE SWITCH (READ-IN DISABLE) / M112-AXIAL LOCATOR RELAX FIXTURE 1
   RUNG wire#powerrail
      Contact( "DB331_EXTENDED_M_CODE_UNIT_1_STA_0".M_code[434] )
      wire#w1
      I_Contact( "DB341_M_UNIT_1_STA_0".M_CODES_UNIT_1_STA_0.Ack_M434 )
      I_Contact( "DB2120_MPP_ITC_IPC".RESET_FAULTS )
      I_Contact( "DB341_M_UNIT_1_STA_0".M_CODES_UNIT_1_STA_0.M_RESET_PULSE )
      Coil( "DB341_M_UNIT_1_STA_0".M_CODES_UNIT_1_STA_0.M434 )
   END_RUNG
   RUNG wire#powerrail
      Contact( "DB341_M_UNIT_1_STA_0".M_CODES_UNIT_1_STA_0.M434 )
   END_RUNG wire#w1
   // the same network as SCL:
   "DB341_M_UNIT_1_STA_0".M_CODES_UNIT_1_STA_0.M434 := ("DB331_EXTENDED_M_CODE_UNIT_1_STA_0".M_code[434] OR "DB341_M_UNIT_1_STA_0".M_CODES_UNIT_1_STA_0.M434) AND NOT "DB341_M_UNIT_1_STA_0".M_CODES_UNIT_1_STA_0.Ack_M434 AND NOT "DB2120_MPP_ITC_IPC".RESET_FAULTS AND NOT "DB341_M_UNIT_1_STA_0".M_CODES_UNIT_1_STA_0.M_RESET_PULSE;
END_REGION

REGION Network 31: ACKNOWLEDGE M435-FIXTURE 1 GRIPPER RELEASE PRESSURE ONLY PRESSURE SWITCH / ACKNOWLEDGE M23-SWITCH ON SPINDLE FRAME BLOWING
   RUNG wire#powerrail
      Contact( "DB2510_U1_F1_GRIPPER".CYL.FULL_LOW_PRESSURED )
      Coil( "DB341_M_UNIT_1_STA_0".M_CODES_UNIT_1_STA_0.Ack_M435 )
   END_RUNG
   // the same network as SCL:
   "DB341_M_UNIT_1_STA_0".M_CODES_UNIT_1_STA_0.Ack_M435 := "DB2510_U1_F1_GRIPPER".CYL.FULL_LOW_PRESSURED;
END_REGION

REGION Network 32: M435-FIXTURE 1 GRIPPER RELEASE PRESSURE ONLY PRESSURE SWITCH / M23-SWITCH ON SPINDLE FRAME BLOWING
   RUNG wire#powerrail
      Contact( "DB331_EXTENDED_M_CODE_UNIT_1_STA_0".M_code[435] )
      wire#w1
      I_Contact( "DB341_M_UNIT_1_STA_0".M_CODES_UNIT_1_STA_0.Ack_M435 )
      I_Contact( "DB2120_MPP_ITC_IPC".RESET_FAULTS )
      I_Contact( "DB341_M_UNIT_1_STA_0".M_CODES_UNIT_1_STA_0.M_RESET_PULSE )
      Coil( "DB341_M_UNIT_1_STA_0".M_CODES_UNIT_1_STA_0.M435 )
   END_RUNG
   RUNG wire#powerrail
      Contact( "DB341_M_UNIT_1_STA_0".M_CODES_UNIT_1_STA_0.M435 )
   END_RUNG wire#w1
   // the same network as SCL:
   "DB341_M_UNIT_1_STA_0".M_CODES_UNIT_1_STA_0.M435 := ("DB331_EXTENDED_M_CODE_UNIT_1_STA_0".M_code[435] OR "DB341_M_UNIT_1_STA_0".M_CODES_UNIT_1_STA_0.M435) AND NOT "DB341_M_UNIT_1_STA_0".M_CODES_UNIT_1_STA_0.Ack_M435 AND NOT "DB2120_MPP_ITC_IPC".RESET_FAULTS AND NOT "DB341_M_UNIT_1_STA_0".M_CODES_UNIT_1_STA_0.M_RESET_PULSE;
END_REGION

REGION Network 33: ACKNOWLEDGE M504-UNIT 1 FIXTURE 2 VERIFY PART AND TOOL IS CLAMPED DURING MACHINING (WHEN TRUE DO). TOGGLED / ACKNOWLEDGE M46-VERIFY FIXTURE 1 PART AND TOOL IS CLAMPED DURING
   RUNG wire#powerrail
      Contact( "M_ZERO" )
      Coil( "DB341_M_UNIT_1_STA_0".M_CODES_UNIT_1_STA_0.Ack_M504 )
   END_RUNG
   // the same network as SCL:
   "DB341_M_UNIT_1_STA_0".M_CODES_UNIT_1_STA_0.Ack_M504 := "M_ZERO";
END_REGION

REGION Network 34: M504-UNIT 1 FIXTURE 2 VERIFY PART AND TOOL IS CLAMPED DURING MACHINING (WHEN TRUE DO). TOGGLED / M46-VERIFY FIXTURE 1 PART AND TOOL IS CLAMPED DURING MACHINING
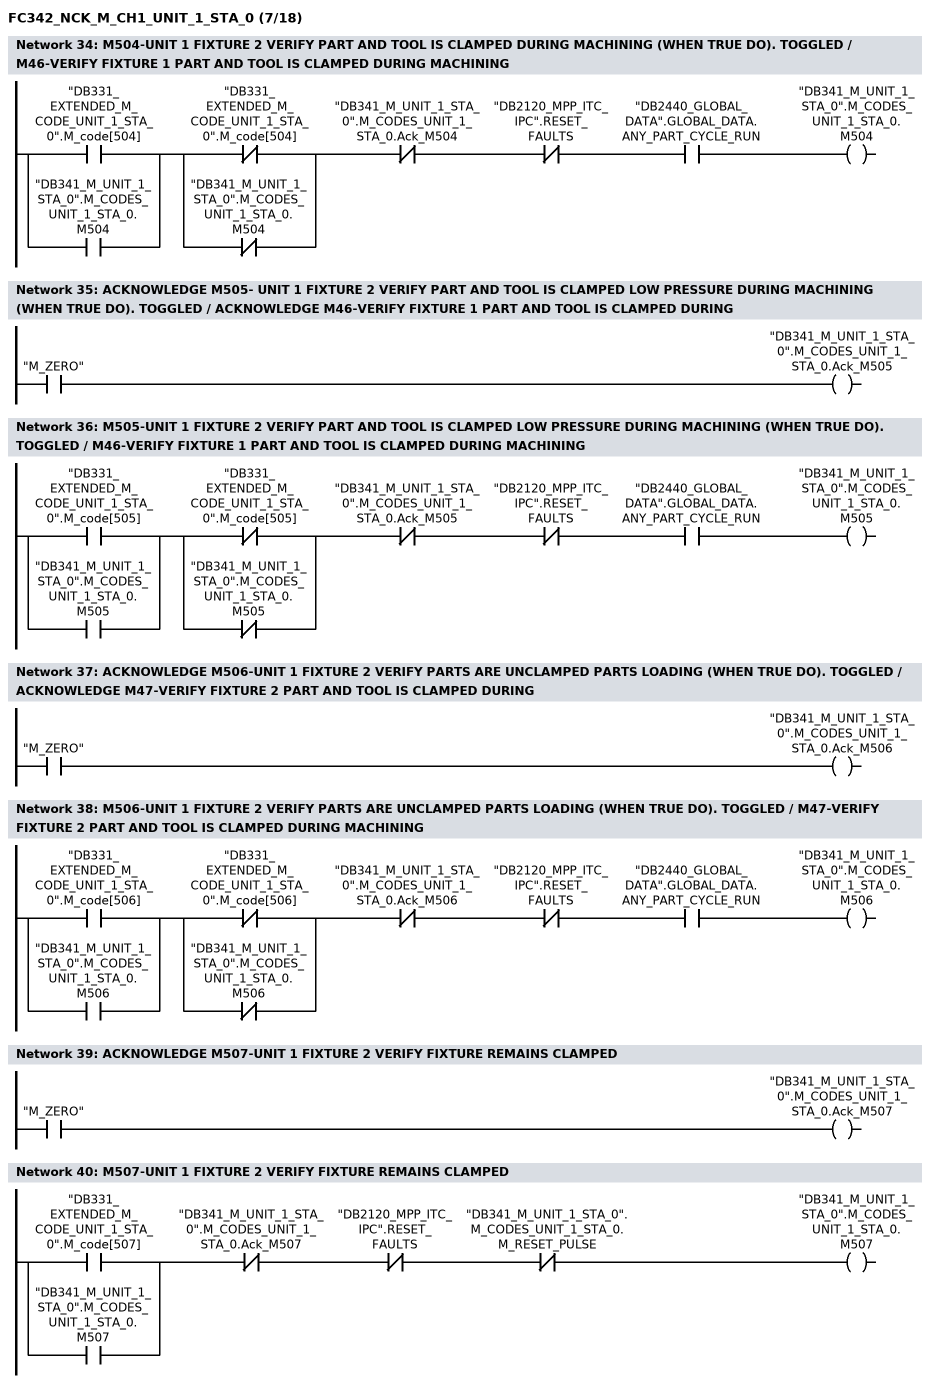
   RUNG wire#powerrail
      Contact( "DB331_EXTENDED_M_CODE_UNIT_1_STA_0".M_code[504] )
      wire#w1
      I_Contact( "DB331_EXTENDED_M_CODE_UNIT_1_STA_0".M_code[504] )
      wire#w2
      I_Contact( "DB341_M_UNIT_1_STA_0".M_CODES_UNIT_1_STA_0.Ack_M504 )
      I_Contact( "DB2120_MPP_ITC_IPC".RESET_FAULTS )
      Contact( "DB2440_GLOBAL_DATA".GLOBAL_DATA.ANY_PART_CYCLE_RUN )
      Coil( "DB341_M_UNIT_1_STA_0".M_CODES_UNIT_1_STA_0.M504 )
   END_RUNG
   RUNG wire#powerrail
      Contact( "DB341_M_UNIT_1_STA_0".M_CODES_UNIT_1_STA_0.M504 )
   END_RUNG wire#w1
   RUNG wire#w1
      I_Contact( "DB341_M_UNIT_1_STA_0".M_CODES_UNIT_1_STA_0.M504 )
   END_RUNG wire#w2
   // the same network as SCL:
   "DB341_M_UNIT_1_STA_0".M_CODES_UNIT_1_STA_0.M504 := ("DB331_EXTENDED_M_CODE_UNIT_1_STA_0".M_code[504] OR "DB341_M_UNIT_1_STA_0".M_CODES_UNIT_1_STA_0.M504) AND (NOT "DB331_EXTENDED_M_CODE_UNIT_1_STA_0".M_code[504] OR NOT "DB341_M_UNIT_1_STA_0".M_CODES_UNIT_1_STA_0.M504) AND NOT "DB341_M_UNIT_1_STA_0".M_CODES_UNIT_1_STA_0.Ack_M504 AND NOT "DB2120_MPP_ITC_IPC".RESET_FAULTS AND "DB2440_GLOBAL_DATA".GLOBAL_DATA.ANY_PART_CYCLE_RUN;
END_REGION

REGION Network 35: ACKNOWLEDGE M505- UNIT 1 FIXTURE 2 VERIFY PART AND TOOL IS CLAMPED LOW PRESSURE DURING MACHINING (WHEN TRUE DO). TOGGLED / ACKNOWLEDGE M46-VERIFY FIXTURE 1 PART AND TOOL IS CLAMPED DURING
   RUNG wire#powerrail
      Contact( "M_ZERO" )
      Coil( "DB341_M_UNIT_1_STA_0".M_CODES_UNIT_1_STA_0.Ack_M505 )
   END_RUNG
   // the same network as SCL:
   "DB341_M_UNIT_1_STA_0".M_CODES_UNIT_1_STA_0.Ack_M505 := "M_ZERO";
END_REGION

REGION Network 36: M505-UNIT 1 FIXTURE 2 VERIFY PART AND TOOL IS CLAMPED LOW PRESSURE DURING MACHINING (WHEN TRUE DO). TOGGLED / M46-VERIFY FIXTURE 1 PART AND TOOL IS CLAMPED DURING MACHINING
   RUNG wire#powerrail
      Contact( "DB331_EXTENDED_M_CODE_UNIT_1_STA_0".M_code[505] )
      wire#w1
      I_Contact( "DB331_EXTENDED_M_CODE_UNIT_1_STA_0".M_code[505] )
      wire#w2
      I_Contact( "DB341_M_UNIT_1_STA_0".M_CODES_UNIT_1_STA_0.Ack_M505 )
      I_Contact( "DB2120_MPP_ITC_IPC".RESET_FAULTS )
      Contact( "DB2440_GLOBAL_DATA".GLOBAL_DATA.ANY_PART_CYCLE_RUN )
      Coil( "DB341_M_UNIT_1_STA_0".M_CODES_UNIT_1_STA_0.M505 )
   END_RUNG
   RUNG wire#powerrail
      Contact( "DB341_M_UNIT_1_STA_0".M_CODES_UNIT_1_STA_0.M505 )
   END_RUNG wire#w1
   RUNG wire#w1
      I_Contact( "DB341_M_UNIT_1_STA_0".M_CODES_UNIT_1_STA_0.M505 )
   END_RUNG wire#w2
   // the same network as SCL:
   "DB341_M_UNIT_1_STA_0".M_CODES_UNIT_1_STA_0.M505 := ("DB331_EXTENDED_M_CODE_UNIT_1_STA_0".M_code[505] OR "DB341_M_UNIT_1_STA_0".M_CODES_UNIT_1_STA_0.M505) AND (NOT "DB331_EXTENDED_M_CODE_UNIT_1_STA_0".M_code[505] OR NOT "DB341_M_UNIT_1_STA_0".M_CODES_UNIT_1_STA_0.M505) AND NOT "DB341_M_UNIT_1_STA_0".M_CODES_UNIT_1_STA_0.Ack_M505 AND NOT "DB2120_MPP_ITC_IPC".RESET_FAULTS AND "DB2440_GLOBAL_DATA".GLOBAL_DATA.ANY_PART_CYCLE_RUN;
END_REGION

REGION Network 37: ACKNOWLEDGE M506-UNIT 1 FIXTURE 2 VERIFY PARTS ARE UNCLAMPED PARTS LOADING (WHEN TRUE DO). TOGGLED / ACKNOWLEDGE M47-VERIFY FIXTURE 2 PART AND TOOL IS CLAMPED DURING
   RUNG wire#powerrail
      Contact( "M_ZERO" )
      Coil( "DB341_M_UNIT_1_STA_0".M_CODES_UNIT_1_STA_0.Ack_M506 )
   END_RUNG
   // the same network as SCL:
   "DB341_M_UNIT_1_STA_0".M_CODES_UNIT_1_STA_0.Ack_M506 := "M_ZERO";
END_REGION

REGION Network 38: M506-UNIT 1 FIXTURE 2 VERIFY PARTS ARE UNCLAMPED PARTS LOADING (WHEN TRUE DO). TOGGLED / M47-VERIFY FIXTURE 2 PART AND TOOL IS CLAMPED DURING MACHINING
   RUNG wire#powerrail
      Contact( "DB331_EXTENDED_M_CODE_UNIT_1_STA_0".M_code[506] )
      wire#w1
      I_Contact( "DB331_EXTENDED_M_CODE_UNIT_1_STA_0".M_code[506] )
      wire#w2
      I_Contact( "DB341_M_UNIT_1_STA_0".M_CODES_UNIT_1_STA_0.Ack_M506 )
      I_Contact( "DB2120_MPP_ITC_IPC".RESET_FAULTS )
      Contact( "DB2440_GLOBAL_DATA".GLOBAL_DATA.ANY_PART_CYCLE_RUN )
      Coil( "DB341_M_UNIT_1_STA_0".M_CODES_UNIT_1_STA_0.M506 )
   END_RUNG
   RUNG wire#powerrail
      Contact( "DB341_M_UNIT_1_STA_0".M_CODES_UNIT_1_STA_0.M506 )
   END_RUNG wire#w1
   RUNG wire#w1
      I_Contact( "DB341_M_UNIT_1_STA_0".M_CODES_UNIT_1_STA_0.M506 )
   END_RUNG wire#w2
   // the same network as SCL:
   "DB341_M_UNIT_1_STA_0".M_CODES_UNIT_1_STA_0.M506 := ("DB331_EXTENDED_M_CODE_UNIT_1_STA_0".M_code[506] OR "DB341_M_UNIT_1_STA_0".M_CODES_UNIT_1_STA_0.M506) AND (NOT "DB331_EXTENDED_M_CODE_UNIT_1_STA_0".M_code[506] OR NOT "DB341_M_UNIT_1_STA_0".M_CODES_UNIT_1_STA_0.M506) AND NOT "DB341_M_UNIT_1_STA_0".M_CODES_UNIT_1_STA_0.Ack_M506 AND NOT "DB2120_MPP_ITC_IPC".RESET_FAULTS AND "DB2440_GLOBAL_DATA".GLOBAL_DATA.ANY_PART_CYCLE_RUN;
END_REGION

REGION Network 39: ACKNOWLEDGE M507-UNIT 1 FIXTURE 2 VERIFY FIXTURE REMAINS CLAMPED
   RUNG wire#powerrail
      Contact( "M_ZERO" )
      Coil( "DB341_M_UNIT_1_STA_0".M_CODES_UNIT_1_STA_0.Ack_M507 )
   END_RUNG
   // the same network as SCL:
   "DB341_M_UNIT_1_STA_0".M_CODES_UNIT_1_STA_0.Ack_M507 := "M_ZERO";
END_REGION

REGION Network 40: M507-UNIT 1 FIXTURE 2 VERIFY FIXTURE REMAINS CLAMPED
   RUNG wire#powerrail
      Contact( "DB331_EXTENDED_M_CODE_UNIT_1_STA_0".M_code[507] )
      wire#w1
      I_Contact( "DB341_M_UNIT_1_STA_0".M_CODES_UNIT_1_STA_0.Ack_M507 )
      I_Contact( "DB2120_MPP_ITC_IPC".RESET_FAULTS )
      I_Contact( "DB341_M_UNIT_1_STA_0".M_CODES_UNIT_1_STA_0.M_RESET_PULSE )
      Coil( "DB341_M_UNIT_1_STA_0".M_CODES_UNIT_1_STA_0.M507 )
   END_RUNG
   RUNG wire#powerrail
      Contact( "DB341_M_UNIT_1_STA_0".M_CODES_UNIT_1_STA_0.M507 )
   END_RUNG wire#w1
   // the same network as SCL:
   "DB341_M_UNIT_1_STA_0".M_CODES_UNIT_1_STA_0.M507 := ("DB331_EXTENDED_M_CODE_UNIT_1_STA_0".M_code[507] OR "DB341_M_UNIT_1_STA_0".M_CODES_UNIT_1_STA_0.M507) AND NOT "DB341_M_UNIT_1_STA_0".M_CODES_UNIT_1_STA_0.Ack_M507 AND NOT "DB2120_MPP_ITC_IPC".RESET_FAULTS AND NOT "DB341_M_UNIT_1_STA_0".M_CODES_UNIT_1_STA_0.M_RESET_PULSE;
END_REGION

REGION Network 41: ACKNOWLEDGE M520- UNIT 1 FIXTURE 2 GRIPPER CLOSE (READ-IN DISABLE)
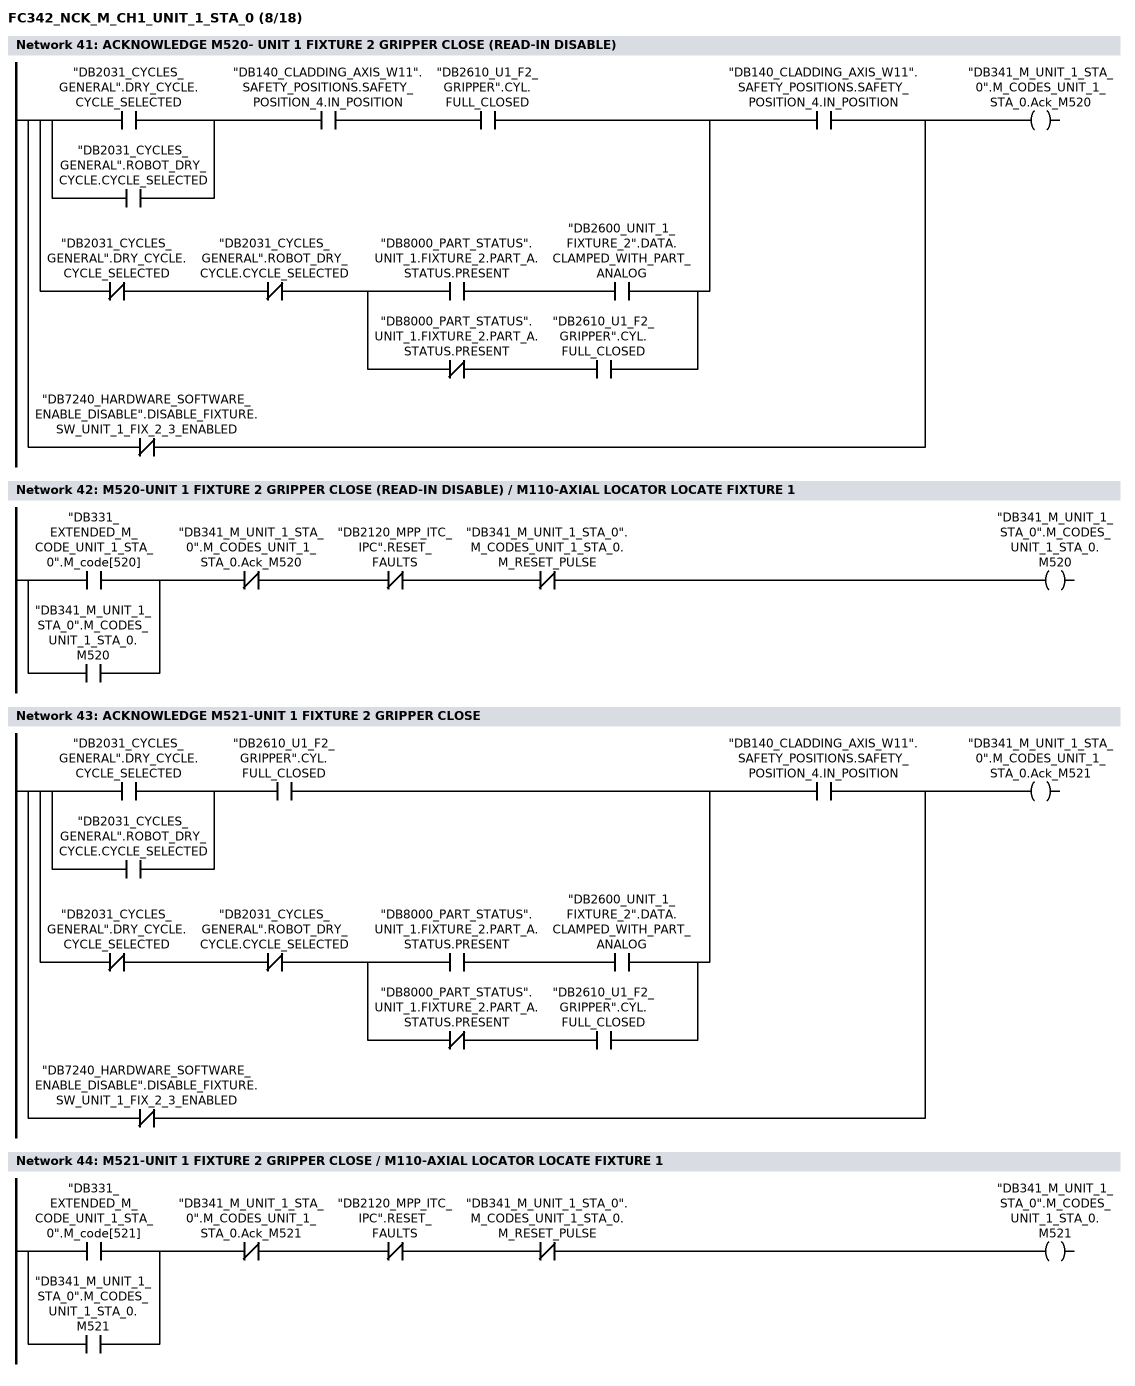
   RUNG wire#powerrail
      Contact( "DB2031_CYCLES_GENERAL".DRY_CYCLE.CYCLE_SELECTED )
      wire#w1
      Contact( "DB140_CLADDING_AXIS_W11".SAFETY_POSITIONS.SAFETY_POSITION_4.IN_POSITION )
      Contact( "DB2610_U1_F2_GRIPPER".CYL.FULL_CLOSED )
      wire#w2
      Contact( "DB140_CLADDING_AXIS_W11".SAFETY_POSITIONS.SAFETY_POSITION_4.IN_POSITION )
      wire#w4
      Coil( "DB341_M_UNIT_1_STA_0".M_CODES_UNIT_1_STA_0.Ack_M520 )
   END_RUNG
   RUNG wire#powerrail
      Contact( "DB2031_CYCLES_GENERAL".ROBOT_DRY_CYCLE.CYCLE_SELECTED )
   END_RUNG wire#w1
   RUNG wire#powerrail
      I_Contact( "DB2031_CYCLES_GENERAL".DRY_CYCLE.CYCLE_SELECTED )
      I_Contact( "DB2031_CYCLES_GENERAL".ROBOT_DRY_CYCLE.CYCLE_SELECTED )
      wire#w3
      Contact( "DB8000_PART_STATUS".UNIT_1.FIXTURE_2.PART_A.STATUS.PRESENT )
      Contact( "DB2600_UNIT_1_FIXTURE_2".DATA.CLAMPED_WITH_PART_ANALOG )
   END_RUNG wire#w2
   RUNG wire#w3
      I_Contact( "DB8000_PART_STATUS".UNIT_1.FIXTURE_2.PART_A.STATUS.PRESENT )
      Contact( "DB2610_U1_F2_GRIPPER".CYL.FULL_CLOSED )
   END_RUNG wire#w2
   RUNG wire#powerrail
      I_Contact( "DB7240_HARDWARE_SOFTWARE_ENABLE_DISABLE".DISABLE_FIXTURE.SW_UNIT_1_FIX_2_3_ENABLED )
   END_RUNG wire#w4
   // the same network as SCL:
   "DB341_M_UNIT_1_STA_0".M_CODES_UNIT_1_STA_0.Ack_M520 := (((("DB2031_CYCLES_GENERAL".DRY_CYCLE.CYCLE_SELECTED OR "DB2031_CYCLES_GENERAL".ROBOT_DRY_CYCLE.CYCLE_SELECTED) AND "DB140_CLADDING_AXIS_W11".SAFETY_POSITIONS.SAFETY_POSITION_4.IN_POSITION AND "DB2610_U1_F2_GRIPPER".CYL.FULL_CLOSED) OR (NOT "DB2031_CYCLES_GENERAL".DRY_CYCLE.CYCLE_SELECTED AND NOT "DB2031_CYCLES_GENERAL".ROBOT_DRY_CYCLE.CYCLE_SELECTED AND (("DB8000_PART_STATUS".UNIT_1.FIXTURE_2.PART_A.STATUS.PRESENT AND "DB2600_UNIT_1_FIXTURE_2".DATA.CLAMPED_WITH_PART_ANALOG) OR (NOT "DB8000_PART_STATUS".UNIT_1.FIXTURE_2.PART_A.STATUS.PRESENT AND "DB2610_U1_F2_GRIPPER".CYL.FULL_CLOSED)))) AND "DB140_CLADDING_AXIS_W11".SAFETY_POSITIONS.SAFETY_POSITION_4.IN_POSITION) OR NOT "DB7240_HARDWARE_SOFTWARE_ENABLE_DISABLE".DISABLE_FIXTURE.SW_UNIT_1_FIX_2_3_ENABLED;
END_REGION

REGION Network 42: M520-UNIT 1 FIXTURE 2 GRIPPER CLOSE (READ-IN DISABLE) / M110-AXIAL LOCATOR LOCATE FIXTURE 1
   RUNG wire#powerrail
      Contact( "DB331_EXTENDED_M_CODE_UNIT_1_STA_0".M_code[520] )
      wire#w1
      I_Contact( "DB341_M_UNIT_1_STA_0".M_CODES_UNIT_1_STA_0.Ack_M520 )
      I_Contact( "DB2120_MPP_ITC_IPC".RESET_FAULTS )
      I_Contact( "DB341_M_UNIT_1_STA_0".M_CODES_UNIT_1_STA_0.M_RESET_PULSE )
      Coil( "DB341_M_UNIT_1_STA_0".M_CODES_UNIT_1_STA_0.M520 )
   END_RUNG
   RUNG wire#powerrail
      Contact( "DB341_M_UNIT_1_STA_0".M_CODES_UNIT_1_STA_0.M520 )
   END_RUNG wire#w1
   // the same network as SCL:
   "DB341_M_UNIT_1_STA_0".M_CODES_UNIT_1_STA_0.M520 := ("DB331_EXTENDED_M_CODE_UNIT_1_STA_0".M_code[520] OR "DB341_M_UNIT_1_STA_0".M_CODES_UNIT_1_STA_0.M520) AND NOT "DB341_M_UNIT_1_STA_0".M_CODES_UNIT_1_STA_0.Ack_M520 AND NOT "DB2120_MPP_ITC_IPC".RESET_FAULTS AND NOT "DB341_M_UNIT_1_STA_0".M_CODES_UNIT_1_STA_0.M_RESET_PULSE;
END_REGION

REGION Network 43: ACKNOWLEDGE M521-UNIT 1 FIXTURE 2 GRIPPER CLOSE
   RUNG wire#powerrail
      Contact( "DB2031_CYCLES_GENERAL".DRY_CYCLE.CYCLE_SELECTED )
      wire#w1
      Contact( "DB2610_U1_F2_GRIPPER".CYL.FULL_CLOSED )
      wire#w2
      Contact( "DB140_CLADDING_AXIS_W11".SAFETY_POSITIONS.SAFETY_POSITION_4.IN_POSITION )
      wire#w4
      Coil( "DB341_M_UNIT_1_STA_0".M_CODES_UNIT_1_STA_0.Ack_M521 )
   END_RUNG
   RUNG wire#powerrail
      Contact( "DB2031_CYCLES_GENERAL".ROBOT_DRY_CYCLE.CYCLE_SELECTED )
   END_RUNG wire#w1
   RUNG wire#powerrail
      I_Contact( "DB2031_CYCLES_GENERAL".DRY_CYCLE.CYCLE_SELECTED )
      I_Contact( "DB2031_CYCLES_GENERAL".ROBOT_DRY_CYCLE.CYCLE_SELECTED )
      wire#w3
      Contact( "DB8000_PART_STATUS".UNIT_1.FIXTURE_2.PART_A.STATUS.PRESENT )
      Contact( "DB2600_UNIT_1_FIXTURE_2".DATA.CLAMPED_WITH_PART_ANALOG )
   END_RUNG wire#w2
   RUNG wire#w3
      I_Contact( "DB8000_PART_STATUS".UNIT_1.FIXTURE_2.PART_A.STATUS.PRESENT )
      Contact( "DB2610_U1_F2_GRIPPER".CYL.FULL_CLOSED )
   END_RUNG wire#w2
   RUNG wire#powerrail
      I_Contact( "DB7240_HARDWARE_SOFTWARE_ENABLE_DISABLE".DISABLE_FIXTURE.SW_UNIT_1_FIX_2_3_ENABLED )
   END_RUNG wire#w4
   // the same network as SCL:
   "DB341_M_UNIT_1_STA_0".M_CODES_UNIT_1_STA_0.Ack_M521 := (((("DB2031_CYCLES_GENERAL".DRY_CYCLE.CYCLE_SELECTED OR "DB2031_CYCLES_GENERAL".ROBOT_DRY_CYCLE.CYCLE_SELECTED) AND "DB2610_U1_F2_GRIPPER".CYL.FULL_CLOSED) OR (NOT "DB2031_CYCLES_GENERAL".DRY_CYCLE.CYCLE_SELECTED AND NOT "DB2031_CYCLES_GENERAL".ROBOT_DRY_CYCLE.CYCLE_SELECTED AND (("DB8000_PART_STATUS".UNIT_1.FIXTURE_2.PART_A.STATUS.PRESENT AND "DB2600_UNIT_1_FIXTURE_2".DATA.CLAMPED_WITH_PART_ANALOG) OR (NOT "DB8000_PART_STATUS".UNIT_1.FIXTURE_2.PART_A.STATUS.PRESENT AND "DB2610_U1_F2_GRIPPER".CYL.FULL_CLOSED)))) AND "DB140_CLADDING_AXIS_W11".SAFETY_POSITIONS.SAFETY_POSITION_4.IN_POSITION) OR NOT "DB7240_HARDWARE_SOFTWARE_ENABLE_DISABLE".DISABLE_FIXTURE.SW_UNIT_1_FIX_2_3_ENABLED;
END_REGION

REGION Network 44: M521-UNIT 1 FIXTURE 2 GRIPPER CLOSE / M110-AXIAL LOCATOR LOCATE FIXTURE 1
   RUNG wire#powerrail
      Contact( "DB331_EXTENDED_M_CODE_UNIT_1_STA_0".M_code[521] )
      wire#w1
      I_Contact( "DB341_M_UNIT_1_STA_0".M_CODES_UNIT_1_STA_0.Ack_M521 )
      I_Contact( "DB2120_MPP_ITC_IPC".RESET_FAULTS )
      I_Contact( "DB341_M_UNIT_1_STA_0".M_CODES_UNIT_1_STA_0.M_RESET_PULSE )
      Coil( "DB341_M_UNIT_1_STA_0".M_CODES_UNIT_1_STA_0.M521 )
   END_RUNG
   RUNG wire#powerrail
      Contact( "DB341_M_UNIT_1_STA_0".M_CODES_UNIT_1_STA_0.M521 )
   END_RUNG wire#w1
   // the same network as SCL:
   "DB341_M_UNIT_1_STA_0".M_CODES_UNIT_1_STA_0.M521 := ("DB331_EXTENDED_M_CODE_UNIT_1_STA_0".M_code[521] OR "DB341_M_UNIT_1_STA_0".M_CODES_UNIT_1_STA_0.M521) AND NOT "DB341_M_UNIT_1_STA_0".M_CODES_UNIT_1_STA_0.Ack_M521 AND NOT "DB2120_MPP_ITC_IPC".RESET_FAULTS AND NOT "DB341_M_UNIT_1_STA_0".M_CODES_UNIT_1_STA_0.M_RESET_PULSE;
END_REGION

REGION Network 45: ACKNOWLEDGE M522-UNIT 1 FIXTURE 2 GRIPPER OPEN (READ-IN DISABLE) / ACKNOWLEDGE M111-AXIAL LOCATOR RETURN FIXTURE 1
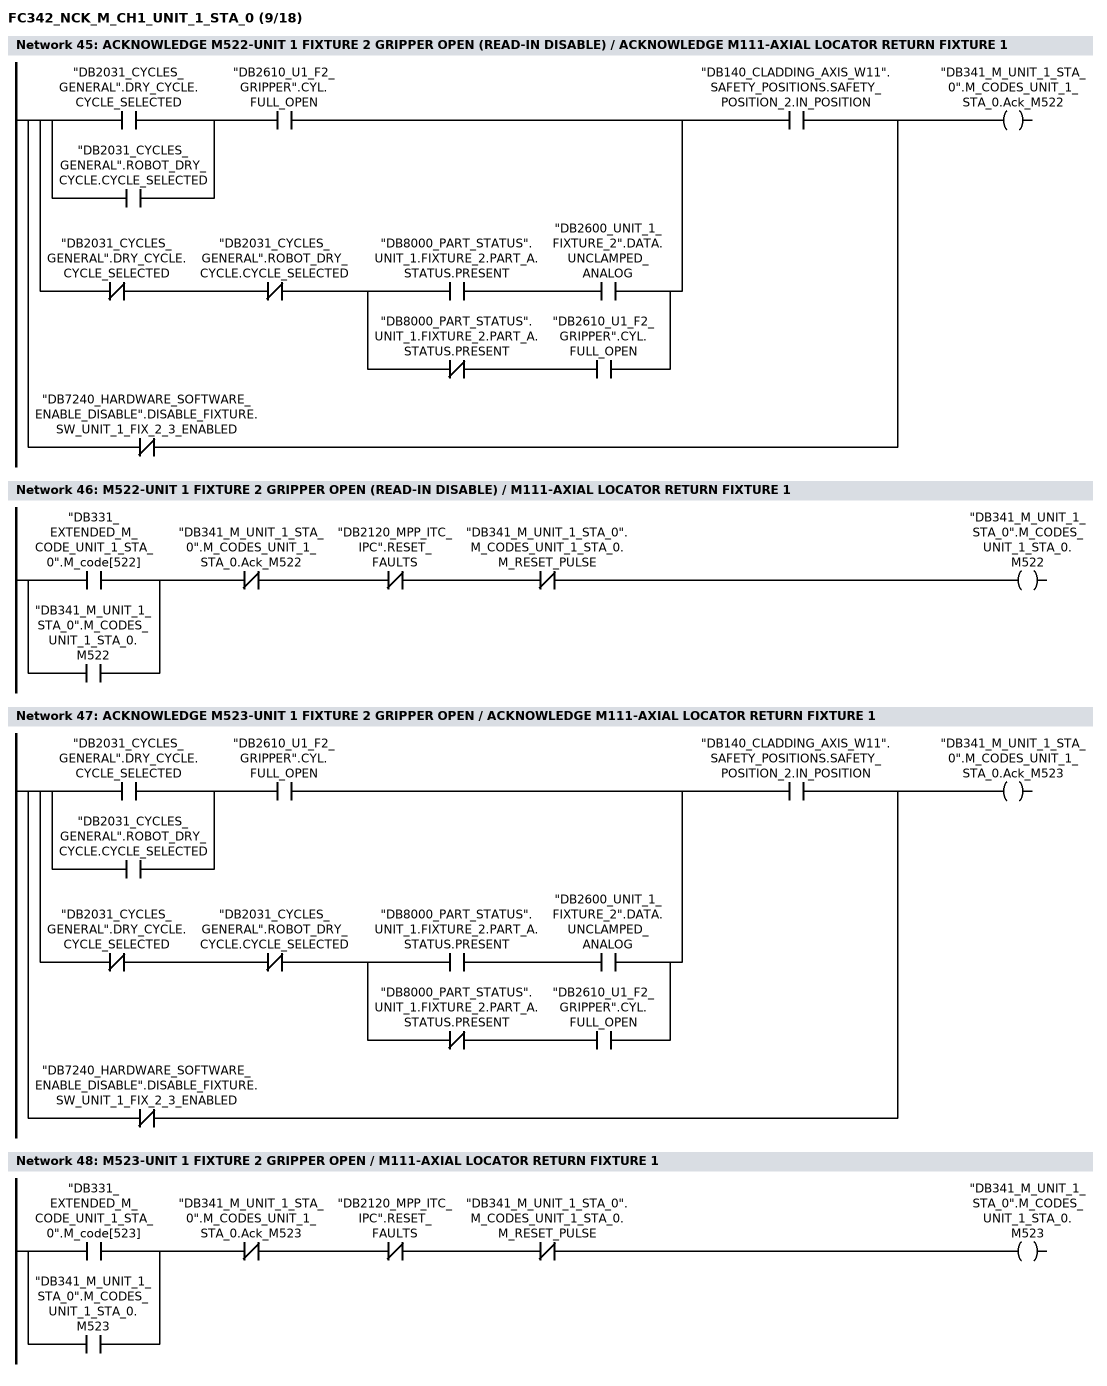
   RUNG wire#powerrail
      Contact( "DB2031_CYCLES_GENERAL".DRY_CYCLE.CYCLE_SELECTED )
      wire#w1
      Contact( "DB2610_U1_F2_GRIPPER".CYL.FULL_OPEN )
      wire#w2
      Contact( "DB140_CLADDING_AXIS_W11".SAFETY_POSITIONS.SAFETY_POSITION_2.IN_POSITION )
      wire#w4
      Coil( "DB341_M_UNIT_1_STA_0".M_CODES_UNIT_1_STA_0.Ack_M522 )
   END_RUNG
   RUNG wire#powerrail
      Contact( "DB2031_CYCLES_GENERAL".ROBOT_DRY_CYCLE.CYCLE_SELECTED )
   END_RUNG wire#w1
   RUNG wire#powerrail
      I_Contact( "DB2031_CYCLES_GENERAL".DRY_CYCLE.CYCLE_SELECTED )
      I_Contact( "DB2031_CYCLES_GENERAL".ROBOT_DRY_CYCLE.CYCLE_SELECTED )
      wire#w3
      Contact( "DB8000_PART_STATUS".UNIT_1.FIXTURE_2.PART_A.STATUS.PRESENT )
      Contact( "DB2600_UNIT_1_FIXTURE_2".DATA.UNCLAMPED_ANALOG )
   END_RUNG wire#w2
   RUNG wire#w3
      I_Contact( "DB8000_PART_STATUS".UNIT_1.FIXTURE_2.PART_A.STATUS.PRESENT )
      Contact( "DB2610_U1_F2_GRIPPER".CYL.FULL_OPEN )
   END_RUNG wire#w2
   RUNG wire#powerrail
      I_Contact( "DB7240_HARDWARE_SOFTWARE_ENABLE_DISABLE".DISABLE_FIXTURE.SW_UNIT_1_FIX_2_3_ENABLED )
   END_RUNG wire#w4
   // the same network as SCL:
   "DB341_M_UNIT_1_STA_0".M_CODES_UNIT_1_STA_0.Ack_M522 := (((("DB2031_CYCLES_GENERAL".DRY_CYCLE.CYCLE_SELECTED OR "DB2031_CYCLES_GENERAL".ROBOT_DRY_CYCLE.CYCLE_SELECTED) AND "DB2610_U1_F2_GRIPPER".CYL.FULL_OPEN) OR (NOT "DB2031_CYCLES_GENERAL".DRY_CYCLE.CYCLE_SELECTED AND NOT "DB2031_CYCLES_GENERAL".ROBOT_DRY_CYCLE.CYCLE_SELECTED AND (("DB8000_PART_STATUS".UNIT_1.FIXTURE_2.PART_A.STATUS.PRESENT AND "DB2600_UNIT_1_FIXTURE_2".DATA.UNCLAMPED_ANALOG) OR (NOT "DB8000_PART_STATUS".UNIT_1.FIXTURE_2.PART_A.STATUS.PRESENT AND "DB2610_U1_F2_GRIPPER".CYL.FULL_OPEN)))) AND "DB140_CLADDING_AXIS_W11".SAFETY_POSITIONS.SAFETY_POSITION_2.IN_POSITION) OR NOT "DB7240_HARDWARE_SOFTWARE_ENABLE_DISABLE".DISABLE_FIXTURE.SW_UNIT_1_FIX_2_3_ENABLED;
END_REGION

REGION Network 46: M522-UNIT 1 FIXTURE 2 GRIPPER OPEN (READ-IN DISABLE) / M111-AXIAL LOCATOR RETURN FIXTURE 1
   RUNG wire#powerrail
      Contact( "DB331_EXTENDED_M_CODE_UNIT_1_STA_0".M_code[522] )
      wire#w1
      I_Contact( "DB341_M_UNIT_1_STA_0".M_CODES_UNIT_1_STA_0.Ack_M522 )
      I_Contact( "DB2120_MPP_ITC_IPC".RESET_FAULTS )
      I_Contact( "DB341_M_UNIT_1_STA_0".M_CODES_UNIT_1_STA_0.M_RESET_PULSE )
      Coil( "DB341_M_UNIT_1_STA_0".M_CODES_UNIT_1_STA_0.M522 )
   END_RUNG
   RUNG wire#powerrail
      Contact( "DB341_M_UNIT_1_STA_0".M_CODES_UNIT_1_STA_0.M522 )
   END_RUNG wire#w1
   // the same network as SCL:
   "DB341_M_UNIT_1_STA_0".M_CODES_UNIT_1_STA_0.M522 := ("DB331_EXTENDED_M_CODE_UNIT_1_STA_0".M_code[522] OR "DB341_M_UNIT_1_STA_0".M_CODES_UNIT_1_STA_0.M522) AND NOT "DB341_M_UNIT_1_STA_0".M_CODES_UNIT_1_STA_0.Ack_M522 AND NOT "DB2120_MPP_ITC_IPC".RESET_FAULTS AND NOT "DB341_M_UNIT_1_STA_0".M_CODES_UNIT_1_STA_0.M_RESET_PULSE;
END_REGION

REGION Network 47: ACKNOWLEDGE M523-UNIT 1 FIXTURE 2 GRIPPER OPEN / ACKNOWLEDGE M111-AXIAL LOCATOR RETURN FIXTURE 1
   RUNG wire#powerrail
      Contact( "DB2031_CYCLES_GENERAL".DRY_CYCLE.CYCLE_SELECTED )
      wire#w1
      Contact( "DB2610_U1_F2_GRIPPER".CYL.FULL_OPEN )
      wire#w2
      Contact( "DB140_CLADDING_AXIS_W11".SAFETY_POSITIONS.SAFETY_POSITION_2.IN_POSITION )
      wire#w4
      Coil( "DB341_M_UNIT_1_STA_0".M_CODES_UNIT_1_STA_0.Ack_M523 )
   END_RUNG
   RUNG wire#powerrail
      Contact( "DB2031_CYCLES_GENERAL".ROBOT_DRY_CYCLE.CYCLE_SELECTED )
   END_RUNG wire#w1
   RUNG wire#powerrail
      I_Contact( "DB2031_CYCLES_GENERAL".DRY_CYCLE.CYCLE_SELECTED )
      I_Contact( "DB2031_CYCLES_GENERAL".ROBOT_DRY_CYCLE.CYCLE_SELECTED )
      wire#w3
      Contact( "DB8000_PART_STATUS".UNIT_1.FIXTURE_2.PART_A.STATUS.PRESENT )
      Contact( "DB2600_UNIT_1_FIXTURE_2".DATA.UNCLAMPED_ANALOG )
   END_RUNG wire#w2
   RUNG wire#w3
      I_Contact( "DB8000_PART_STATUS".UNIT_1.FIXTURE_2.PART_A.STATUS.PRESENT )
      Contact( "DB2610_U1_F2_GRIPPER".CYL.FULL_OPEN )
   END_RUNG wire#w2
   RUNG wire#powerrail
      I_Contact( "DB7240_HARDWARE_SOFTWARE_ENABLE_DISABLE".DISABLE_FIXTURE.SW_UNIT_1_FIX_2_3_ENABLED )
   END_RUNG wire#w4
   // the same network as SCL:
   "DB341_M_UNIT_1_STA_0".M_CODES_UNIT_1_STA_0.Ack_M523 := (((("DB2031_CYCLES_GENERAL".DRY_CYCLE.CYCLE_SELECTED OR "DB2031_CYCLES_GENERAL".ROBOT_DRY_CYCLE.CYCLE_SELECTED) AND "DB2610_U1_F2_GRIPPER".CYL.FULL_OPEN) OR (NOT "DB2031_CYCLES_GENERAL".DRY_CYCLE.CYCLE_SELECTED AND NOT "DB2031_CYCLES_GENERAL".ROBOT_DRY_CYCLE.CYCLE_SELECTED AND (("DB8000_PART_STATUS".UNIT_1.FIXTURE_2.PART_A.STATUS.PRESENT AND "DB2600_UNIT_1_FIXTURE_2".DATA.UNCLAMPED_ANALOG) OR (NOT "DB8000_PART_STATUS".UNIT_1.FIXTURE_2.PART_A.STATUS.PRESENT AND "DB2610_U1_F2_GRIPPER".CYL.FULL_OPEN)))) AND "DB140_CLADDING_AXIS_W11".SAFETY_POSITIONS.SAFETY_POSITION_2.IN_POSITION) OR NOT "DB7240_HARDWARE_SOFTWARE_ENABLE_DISABLE".DISABLE_FIXTURE.SW_UNIT_1_FIX_2_3_ENABLED;
END_REGION

REGION Network 48: M523-UNIT 1 FIXTURE 2 GRIPPER OPEN / M111-AXIAL LOCATOR RETURN FIXTURE 1
   RUNG wire#powerrail
      Contact( "DB331_EXTENDED_M_CODE_UNIT_1_STA_0".M_code[523] )
      wire#w1
      I_Contact( "DB341_M_UNIT_1_STA_0".M_CODES_UNIT_1_STA_0.Ack_M523 )
      I_Contact( "DB2120_MPP_ITC_IPC".RESET_FAULTS )
      I_Contact( "DB341_M_UNIT_1_STA_0".M_CODES_UNIT_1_STA_0.M_RESET_PULSE )
      Coil( "DB341_M_UNIT_1_STA_0".M_CODES_UNIT_1_STA_0.M523 )
   END_RUNG
   RUNG wire#powerrail
      Contact( "DB341_M_UNIT_1_STA_0".M_CODES_UNIT_1_STA_0.M523 )
   END_RUNG wire#w1
   // the same network as SCL:
   "DB341_M_UNIT_1_STA_0".M_CODES_UNIT_1_STA_0.M523 := ("DB331_EXTENDED_M_CODE_UNIT_1_STA_0".M_code[523] OR "DB341_M_UNIT_1_STA_0".M_CODES_UNIT_1_STA_0.M523) AND NOT "DB341_M_UNIT_1_STA_0".M_CODES_UNIT_1_STA_0.Ack_M523 AND NOT "DB2120_MPP_ITC_IPC".RESET_FAULTS AND NOT "DB341_M_UNIT_1_STA_0".M_CODES_UNIT_1_STA_0.M_RESET_PULSE;
END_REGION

REGION Network 49: ACKNOWLEDGE M524-UNIT 1 FIXTURE 2 GRIPPER RELEASE PRESSURE (READ-IN DISABLE) / ACKNOWLEDGE M112-AXIAL LOCATOR RELAX FIXTURE 1
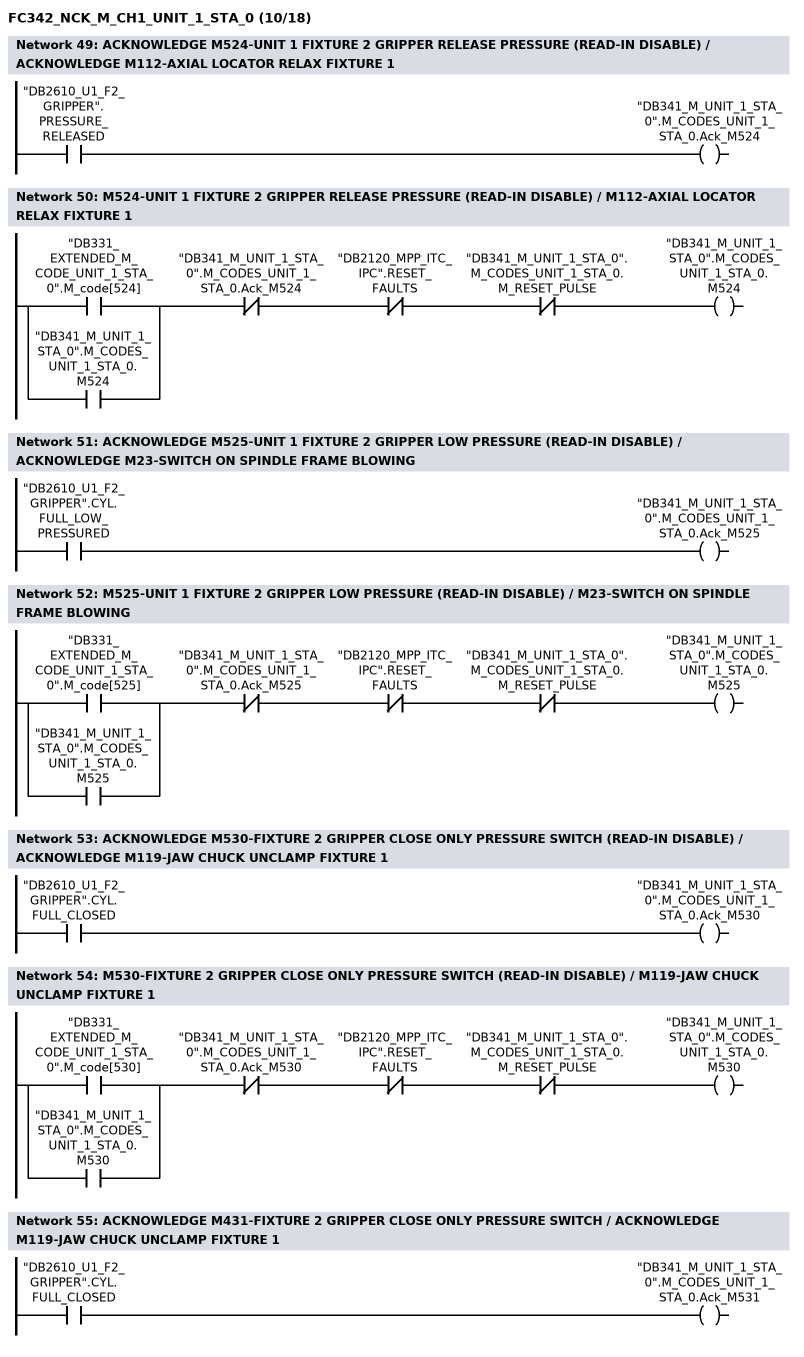
   RUNG wire#powerrail
      Contact( "DB2610_U1_F2_GRIPPER".PRESSURE_RELEASED )
      Coil( "DB341_M_UNIT_1_STA_0".M_CODES_UNIT_1_STA_0.Ack_M524 )
   END_RUNG
   // the same network as SCL:
   "DB341_M_UNIT_1_STA_0".M_CODES_UNIT_1_STA_0.Ack_M524 := "DB2610_U1_F2_GRIPPER".PRESSURE_RELEASED;
END_REGION

REGION Network 50: M524-UNIT 1 FIXTURE 2 GRIPPER RELEASE PRESSURE (READ-IN DISABLE) / M112-AXIAL LOCATOR RELAX FIXTURE 1
   RUNG wire#powerrail
      Contact( "DB331_EXTENDED_M_CODE_UNIT_1_STA_0".M_code[524] )
      wire#w1
      I_Contact( "DB341_M_UNIT_1_STA_0".M_CODES_UNIT_1_STA_0.Ack_M524 )
      I_Contact( "DB2120_MPP_ITC_IPC".RESET_FAULTS )
      I_Contact( "DB341_M_UNIT_1_STA_0".M_CODES_UNIT_1_STA_0.M_RESET_PULSE )
      Coil( "DB341_M_UNIT_1_STA_0".M_CODES_UNIT_1_STA_0.M524 )
   END_RUNG
   RUNG wire#powerrail
      Contact( "DB341_M_UNIT_1_STA_0".M_CODES_UNIT_1_STA_0.M524 )
   END_RUNG wire#w1
   // the same network as SCL:
   "DB341_M_UNIT_1_STA_0".M_CODES_UNIT_1_STA_0.M524 := ("DB331_EXTENDED_M_CODE_UNIT_1_STA_0".M_code[524] OR "DB341_M_UNIT_1_STA_0".M_CODES_UNIT_1_STA_0.M524) AND NOT "DB341_M_UNIT_1_STA_0".M_CODES_UNIT_1_STA_0.Ack_M524 AND NOT "DB2120_MPP_ITC_IPC".RESET_FAULTS AND NOT "DB341_M_UNIT_1_STA_0".M_CODES_UNIT_1_STA_0.M_RESET_PULSE;
END_REGION

REGION Network 51: ACKNOWLEDGE M525-UNIT 1 FIXTURE 2 GRIPPER LOW PRESSURE (READ-IN DISABLE) / ACKNOWLEDGE M23-SWITCH ON SPINDLE FRAME BLOWING
   RUNG wire#powerrail
      Contact( "DB2610_U1_F2_GRIPPER".CYL.FULL_LOW_PRESSURED )
      Coil( "DB341_M_UNIT_1_STA_0".M_CODES_UNIT_1_STA_0.Ack_M525 )
   END_RUNG
   // the same network as SCL:
   "DB341_M_UNIT_1_STA_0".M_CODES_UNIT_1_STA_0.Ack_M525 := "DB2610_U1_F2_GRIPPER".CYL.FULL_LOW_PRESSURED;
END_REGION

REGION Network 52: M525-UNIT 1 FIXTURE 2 GRIPPER LOW PRESSURE (READ-IN DISABLE) / M23-SWITCH ON SPINDLE FRAME BLOWING
   RUNG wire#powerrail
      Contact( "DB331_EXTENDED_M_CODE_UNIT_1_STA_0".M_code[525] )
      wire#w1
      I_Contact( "DB341_M_UNIT_1_STA_0".M_CODES_UNIT_1_STA_0.Ack_M525 )
      I_Contact( "DB2120_MPP_ITC_IPC".RESET_FAULTS )
      I_Contact( "DB341_M_UNIT_1_STA_0".M_CODES_UNIT_1_STA_0.M_RESET_PULSE )
      Coil( "DB341_M_UNIT_1_STA_0".M_CODES_UNIT_1_STA_0.M525 )
   END_RUNG
   RUNG wire#powerrail
      Contact( "DB341_M_UNIT_1_STA_0".M_CODES_UNIT_1_STA_0.M525 )
   END_RUNG wire#w1
   // the same network as SCL:
   "DB341_M_UNIT_1_STA_0".M_CODES_UNIT_1_STA_0.M525 := ("DB331_EXTENDED_M_CODE_UNIT_1_STA_0".M_code[525] OR "DB341_M_UNIT_1_STA_0".M_CODES_UNIT_1_STA_0.M525) AND NOT "DB341_M_UNIT_1_STA_0".M_CODES_UNIT_1_STA_0.Ack_M525 AND NOT "DB2120_MPP_ITC_IPC".RESET_FAULTS AND NOT "DB341_M_UNIT_1_STA_0".M_CODES_UNIT_1_STA_0.M_RESET_PULSE;
END_REGION

REGION Network 53: ACKNOWLEDGE M530-FIXTURE 2 GRIPPER CLOSE ONLY PRESSURE SWITCH (READ-IN DISABLE) / ACKNOWLEDGE M119-JAW CHUCK UNCLAMP FIXTURE 1
   RUNG wire#powerrail
      Contact( "DB2610_U1_F2_GRIPPER".CYL.FULL_CLOSED )
      Coil( "DB341_M_UNIT_1_STA_0".M_CODES_UNIT_1_STA_0.Ack_M530 )
   END_RUNG
   // the same network as SCL:
   "DB341_M_UNIT_1_STA_0".M_CODES_UNIT_1_STA_0.Ack_M530 := "DB2610_U1_F2_GRIPPER".CYL.FULL_CLOSED;
END_REGION

REGION Network 54: M530-FIXTURE 2 GRIPPER CLOSE ONLY PRESSURE SWITCH (READ-IN DISABLE) / M119-JAW CHUCK UNCLAMP FIXTURE 1
   RUNG wire#powerrail
      Contact( "DB331_EXTENDED_M_CODE_UNIT_1_STA_0".M_code[530] )
      wire#w1
      I_Contact( "DB341_M_UNIT_1_STA_0".M_CODES_UNIT_1_STA_0.Ack_M530 )
      I_Contact( "DB2120_MPP_ITC_IPC".RESET_FAULTS )
      I_Contact( "DB341_M_UNIT_1_STA_0".M_CODES_UNIT_1_STA_0.M_RESET_PULSE )
      Coil( "DB341_M_UNIT_1_STA_0".M_CODES_UNIT_1_STA_0.M530 )
   END_RUNG
   RUNG wire#powerrail
      Contact( "DB341_M_UNIT_1_STA_0".M_CODES_UNIT_1_STA_0.M530 )
   END_RUNG wire#w1
   // the same network as SCL:
   "DB341_M_UNIT_1_STA_0".M_CODES_UNIT_1_STA_0.M530 := ("DB331_EXTENDED_M_CODE_UNIT_1_STA_0".M_code[530] OR "DB341_M_UNIT_1_STA_0".M_CODES_UNIT_1_STA_0.M530) AND NOT "DB341_M_UNIT_1_STA_0".M_CODES_UNIT_1_STA_0.Ack_M530 AND NOT "DB2120_MPP_ITC_IPC".RESET_FAULTS AND NOT "DB341_M_UNIT_1_STA_0".M_CODES_UNIT_1_STA_0.M_RESET_PULSE;
END_REGION

REGION Network 55: ACKNOWLEDGE M431-FIXTURE 2 GRIPPER CLOSE ONLY PRESSURE SWITCH / ACKNOWLEDGE M119-JAW CHUCK UNCLAMP FIXTURE 1
   RUNG wire#powerrail
      Contact( "DB2610_U1_F2_GRIPPER".CYL.FULL_CLOSED )
      Coil( "DB341_M_UNIT_1_STA_0".M_CODES_UNIT_1_STA_0.Ack_M531 )
   END_RUNG
   // the same network as SCL:
   "DB341_M_UNIT_1_STA_0".M_CODES_UNIT_1_STA_0.Ack_M531 := "DB2610_U1_F2_GRIPPER".CYL.FULL_CLOSED;
END_REGION

REGION Network 56: M531-FIXTURE 2 GRIPPER CLOSE ONLY PRESSURE SWITCH / M119-JAW CHUCK UNCLAMP FIXTURE 1
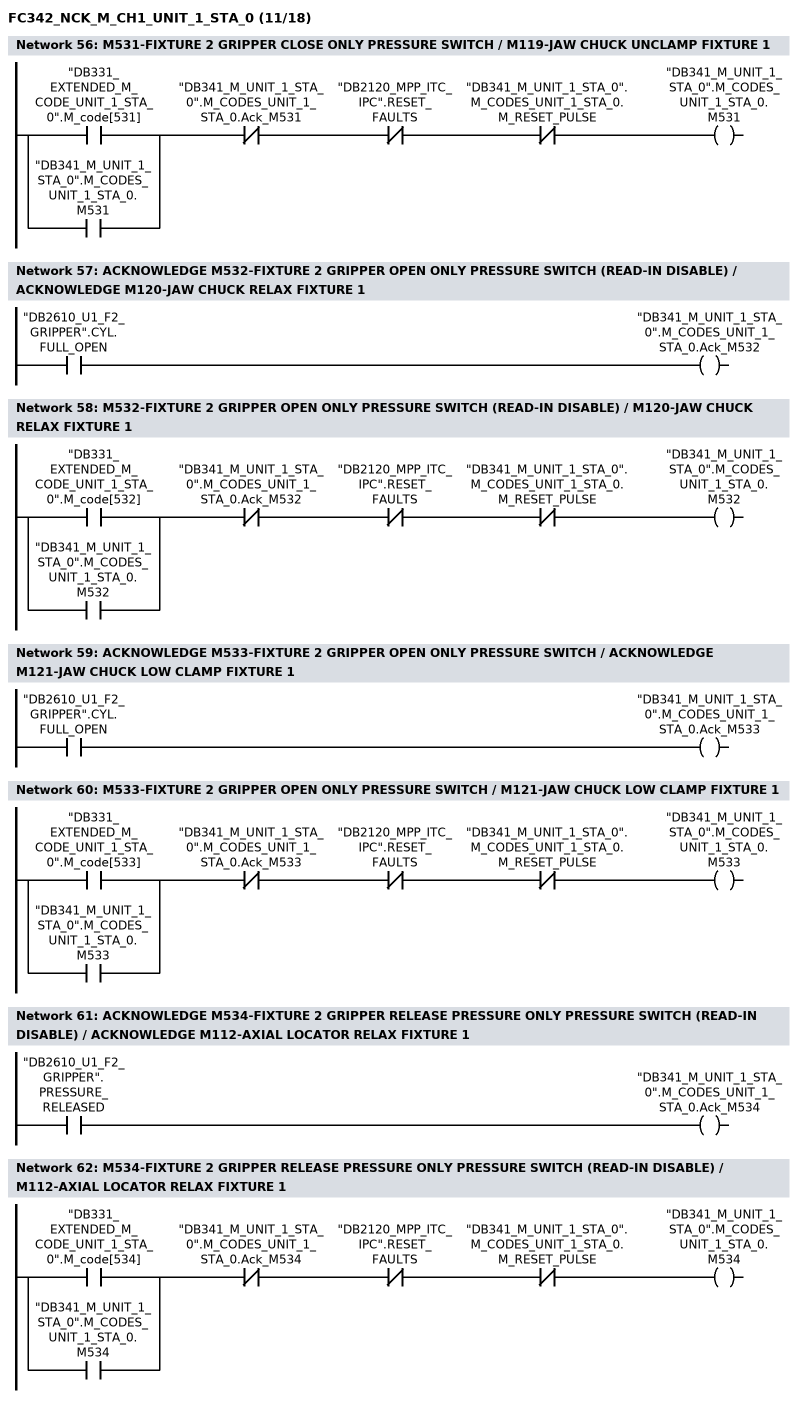
   RUNG wire#powerrail
      Contact( "DB331_EXTENDED_M_CODE_UNIT_1_STA_0".M_code[531] )
      wire#w1
      I_Contact( "DB341_M_UNIT_1_STA_0".M_CODES_UNIT_1_STA_0.Ack_M531 )
      I_Contact( "DB2120_MPP_ITC_IPC".RESET_FAULTS )
      I_Contact( "DB341_M_UNIT_1_STA_0".M_CODES_UNIT_1_STA_0.M_RESET_PULSE )
      Coil( "DB341_M_UNIT_1_STA_0".M_CODES_UNIT_1_STA_0.M531 )
   END_RUNG
   RUNG wire#powerrail
      Contact( "DB341_M_UNIT_1_STA_0".M_CODES_UNIT_1_STA_0.M531 )
   END_RUNG wire#w1
   // the same network as SCL:
   "DB341_M_UNIT_1_STA_0".M_CODES_UNIT_1_STA_0.M531 := ("DB331_EXTENDED_M_CODE_UNIT_1_STA_0".M_code[531] OR "DB341_M_UNIT_1_STA_0".M_CODES_UNIT_1_STA_0.M531) AND NOT "DB341_M_UNIT_1_STA_0".M_CODES_UNIT_1_STA_0.Ack_M531 AND NOT "DB2120_MPP_ITC_IPC".RESET_FAULTS AND NOT "DB341_M_UNIT_1_STA_0".M_CODES_UNIT_1_STA_0.M_RESET_PULSE;
END_REGION

REGION Network 57: ACKNOWLEDGE M532-FIXTURE 2 GRIPPER OPEN ONLY PRESSURE SWITCH (READ-IN DISABLE) / ACKNOWLEDGE M120-JAW CHUCK RELAX FIXTURE 1
   RUNG wire#powerrail
      Contact( "DB2610_U1_F2_GRIPPER".CYL.FULL_OPEN )
      Coil( "DB341_M_UNIT_1_STA_0".M_CODES_UNIT_1_STA_0.Ack_M532 )
   END_RUNG
   // the same network as SCL:
   "DB341_M_UNIT_1_STA_0".M_CODES_UNIT_1_STA_0.Ack_M532 := "DB2610_U1_F2_GRIPPER".CYL.FULL_OPEN;
END_REGION

REGION Network 58: M532-FIXTURE 2 GRIPPER OPEN ONLY PRESSURE SWITCH (READ-IN DISABLE) / M120-JAW CHUCK RELAX FIXTURE 1
   RUNG wire#powerrail
      Contact( "DB331_EXTENDED_M_CODE_UNIT_1_STA_0".M_code[532] )
      wire#w1
      I_Contact( "DB341_M_UNIT_1_STA_0".M_CODES_UNIT_1_STA_0.Ack_M532 )
      I_Contact( "DB2120_MPP_ITC_IPC".RESET_FAULTS )
      I_Contact( "DB341_M_UNIT_1_STA_0".M_CODES_UNIT_1_STA_0.M_RESET_PULSE )
      Coil( "DB341_M_UNIT_1_STA_0".M_CODES_UNIT_1_STA_0.M532 )
   END_RUNG
   RUNG wire#powerrail
      Contact( "DB341_M_UNIT_1_STA_0".M_CODES_UNIT_1_STA_0.M532 )
   END_RUNG wire#w1
   // the same network as SCL:
   "DB341_M_UNIT_1_STA_0".M_CODES_UNIT_1_STA_0.M532 := ("DB331_EXTENDED_M_CODE_UNIT_1_STA_0".M_code[532] OR "DB341_M_UNIT_1_STA_0".M_CODES_UNIT_1_STA_0.M532) AND NOT "DB341_M_UNIT_1_STA_0".M_CODES_UNIT_1_STA_0.Ack_M532 AND NOT "DB2120_MPP_ITC_IPC".RESET_FAULTS AND NOT "DB341_M_UNIT_1_STA_0".M_CODES_UNIT_1_STA_0.M_RESET_PULSE;
END_REGION

REGION Network 59: ACKNOWLEDGE M533-FIXTURE 2 GRIPPER OPEN ONLY PRESSURE SWITCH / ACKNOWLEDGE M121-JAW CHUCK LOW CLAMP FIXTURE 1
   RUNG wire#powerrail
      Contact( "DB2610_U1_F2_GRIPPER".CYL.FULL_OPEN )
      Coil( "DB341_M_UNIT_1_STA_0".M_CODES_UNIT_1_STA_0.Ack_M533 )
   END_RUNG
   // the same network as SCL:
   "DB341_M_UNIT_1_STA_0".M_CODES_UNIT_1_STA_0.Ack_M533 := "DB2610_U1_F2_GRIPPER".CYL.FULL_OPEN;
END_REGION

REGION Network 60: M533-FIXTURE 2 GRIPPER OPEN ONLY PRESSURE SWITCH / M121-JAW CHUCK LOW CLAMP FIXTURE 1
   RUNG wire#powerrail
      Contact( "DB331_EXTENDED_M_CODE_UNIT_1_STA_0".M_code[533] )
      wire#w1
      I_Contact( "DB341_M_UNIT_1_STA_0".M_CODES_UNIT_1_STA_0.Ack_M533 )
      I_Contact( "DB2120_MPP_ITC_IPC".RESET_FAULTS )
      I_Contact( "DB341_M_UNIT_1_STA_0".M_CODES_UNIT_1_STA_0.M_RESET_PULSE )
      Coil( "DB341_M_UNIT_1_STA_0".M_CODES_UNIT_1_STA_0.M533 )
   END_RUNG
   RUNG wire#powerrail
      Contact( "DB341_M_UNIT_1_STA_0".M_CODES_UNIT_1_STA_0.M533 )
   END_RUNG wire#w1
   // the same network as SCL:
   "DB341_M_UNIT_1_STA_0".M_CODES_UNIT_1_STA_0.M533 := ("DB331_EXTENDED_M_CODE_UNIT_1_STA_0".M_code[533] OR "DB341_M_UNIT_1_STA_0".M_CODES_UNIT_1_STA_0.M533) AND NOT "DB341_M_UNIT_1_STA_0".M_CODES_UNIT_1_STA_0.Ack_M533 AND NOT "DB2120_MPP_ITC_IPC".RESET_FAULTS AND NOT "DB341_M_UNIT_1_STA_0".M_CODES_UNIT_1_STA_0.M_RESET_PULSE;
END_REGION

REGION Network 61: ACKNOWLEDGE M534-FIXTURE 2 GRIPPER RELEASE PRESSURE ONLY PRESSURE SWITCH (READ-IN DISABLE) / ACKNOWLEDGE M112-AXIAL LOCATOR RELAX FIXTURE 1
   RUNG wire#powerrail
      Contact( "DB2610_U1_F2_GRIPPER".PRESSURE_RELEASED )
      Coil( "DB341_M_UNIT_1_STA_0".M_CODES_UNIT_1_STA_0.Ack_M534 )
   END_RUNG
   // the same network as SCL:
   "DB341_M_UNIT_1_STA_0".M_CODES_UNIT_1_STA_0.Ack_M534 := "DB2610_U1_F2_GRIPPER".PRESSURE_RELEASED;
END_REGION

REGION Network 62: M534-FIXTURE 2 GRIPPER RELEASE PRESSURE ONLY PRESSURE SWITCH (READ-IN DISABLE) / M112-AXIAL LOCATOR RELAX FIXTURE 1
   RUNG wire#powerrail
      Contact( "DB331_EXTENDED_M_CODE_UNIT_1_STA_0".M_code[534] )
      wire#w1
      I_Contact( "DB341_M_UNIT_1_STA_0".M_CODES_UNIT_1_STA_0.Ack_M534 )
      I_Contact( "DB2120_MPP_ITC_IPC".RESET_FAULTS )
      I_Contact( "DB341_M_UNIT_1_STA_0".M_CODES_UNIT_1_STA_0.M_RESET_PULSE )
      Coil( "DB341_M_UNIT_1_STA_0".M_CODES_UNIT_1_STA_0.M534 )
   END_RUNG
   RUNG wire#powerrail
      Contact( "DB341_M_UNIT_1_STA_0".M_CODES_UNIT_1_STA_0.M534 )
   END_RUNG wire#w1
   // the same network as SCL:
   "DB341_M_UNIT_1_STA_0".M_CODES_UNIT_1_STA_0.M534 := ("DB331_EXTENDED_M_CODE_UNIT_1_STA_0".M_code[534] OR "DB341_M_UNIT_1_STA_0".M_CODES_UNIT_1_STA_0.M534) AND NOT "DB341_M_UNIT_1_STA_0".M_CODES_UNIT_1_STA_0.Ack_M534 AND NOT "DB2120_MPP_ITC_IPC".RESET_FAULTS AND NOT "DB341_M_UNIT_1_STA_0".M_CODES_UNIT_1_STA_0.M_RESET_PULSE;
END_REGION

REGION Network 63: ACKNOWLEDGE M535-FIXTURE 2 GRIPPER RELEASE PRESSURE ONLY PRESSURE SWITCH / ACKNOWLEDGE M23-SWITCH ON SPINDLE FRAME BLOWING
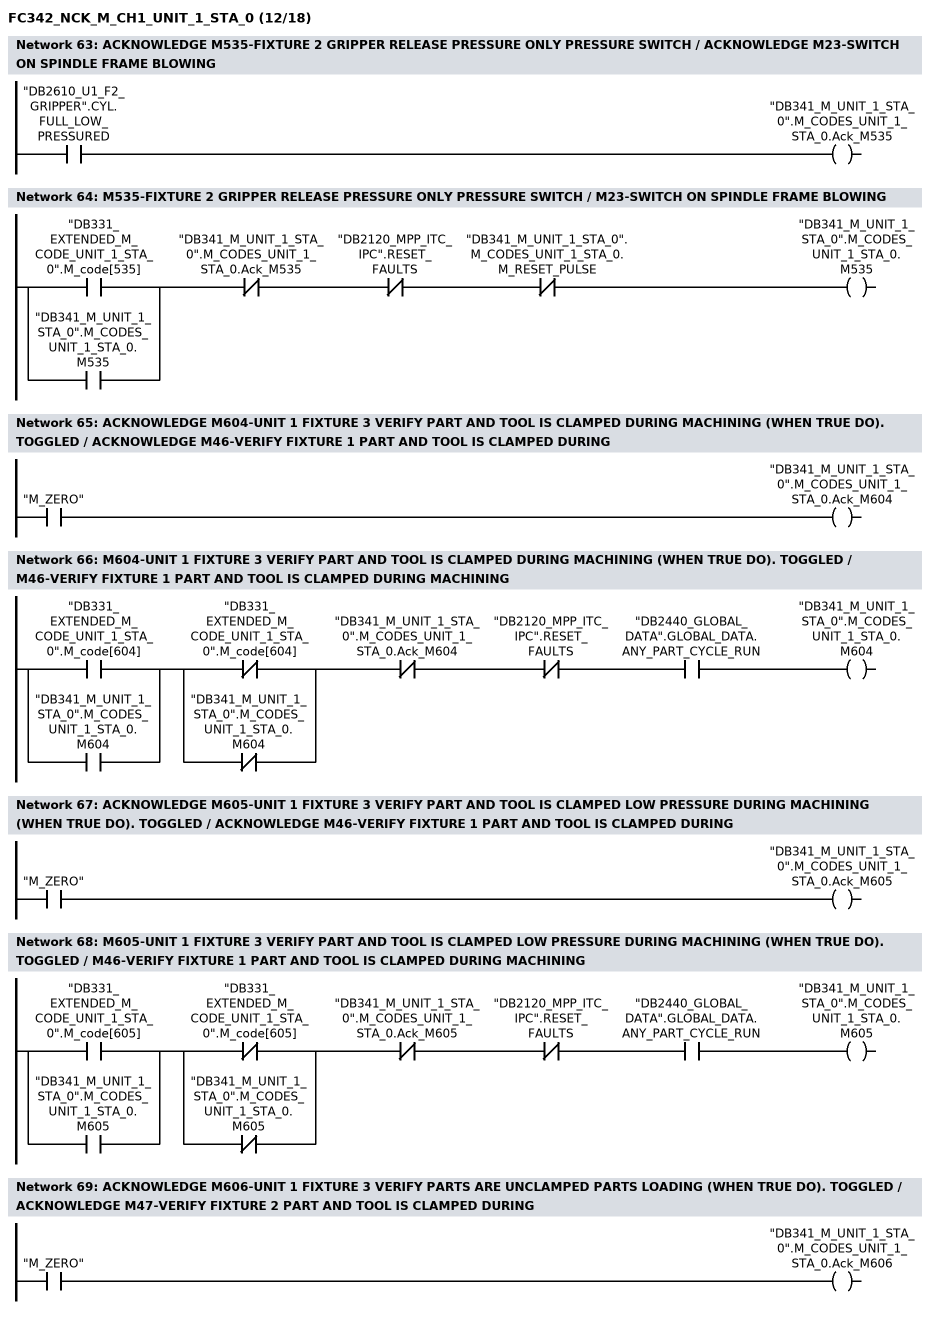
   RUNG wire#powerrail
      Contact( "DB2610_U1_F2_GRIPPER".CYL.FULL_LOW_PRESSURED )
      Coil( "DB341_M_UNIT_1_STA_0".M_CODES_UNIT_1_STA_0.Ack_M535 )
   END_RUNG
   // the same network as SCL:
   "DB341_M_UNIT_1_STA_0".M_CODES_UNIT_1_STA_0.Ack_M535 := "DB2610_U1_F2_GRIPPER".CYL.FULL_LOW_PRESSURED;
END_REGION

REGION Network 64: M535-FIXTURE 2 GRIPPER RELEASE PRESSURE ONLY PRESSURE SWITCH / M23-SWITCH ON SPINDLE FRAME BLOWING
   RUNG wire#powerrail
      Contact( "DB331_EXTENDED_M_CODE_UNIT_1_STA_0".M_code[535] )
      wire#w1
      I_Contact( "DB341_M_UNIT_1_STA_0".M_CODES_UNIT_1_STA_0.Ack_M535 )
      I_Contact( "DB2120_MPP_ITC_IPC".RESET_FAULTS )
      I_Contact( "DB341_M_UNIT_1_STA_0".M_CODES_UNIT_1_STA_0.M_RESET_PULSE )
      Coil( "DB341_M_UNIT_1_STA_0".M_CODES_UNIT_1_STA_0.M535 )
   END_RUNG
   RUNG wire#powerrail
      Contact( "DB341_M_UNIT_1_STA_0".M_CODES_UNIT_1_STA_0.M535 )
   END_RUNG wire#w1
   // the same network as SCL:
   "DB341_M_UNIT_1_STA_0".M_CODES_UNIT_1_STA_0.M535 := ("DB331_EXTENDED_M_CODE_UNIT_1_STA_0".M_code[535] OR "DB341_M_UNIT_1_STA_0".M_CODES_UNIT_1_STA_0.M535) AND NOT "DB341_M_UNIT_1_STA_0".M_CODES_UNIT_1_STA_0.Ack_M535 AND NOT "DB2120_MPP_ITC_IPC".RESET_FAULTS AND NOT "DB341_M_UNIT_1_STA_0".M_CODES_UNIT_1_STA_0.M_RESET_PULSE;
END_REGION

REGION Network 65: ACKNOWLEDGE M604-UNIT 1 FIXTURE 3 VERIFY PART AND TOOL IS CLAMPED DURING MACHINING (WHEN TRUE DO). TOGGLED / ACKNOWLEDGE M46-VERIFY FIXTURE 1 PART AND TOOL IS CLAMPED DURING
   RUNG wire#powerrail
      Contact( "M_ZERO" )
      Coil( "DB341_M_UNIT_1_STA_0".M_CODES_UNIT_1_STA_0.Ack_M604 )
   END_RUNG
   // the same network as SCL:
   "DB341_M_UNIT_1_STA_0".M_CODES_UNIT_1_STA_0.Ack_M604 := "M_ZERO";
END_REGION

REGION Network 66: M604-UNIT 1 FIXTURE 3 VERIFY PART AND TOOL IS CLAMPED DURING MACHINING (WHEN TRUE DO). TOGGLED / M46-VERIFY FIXTURE 1 PART AND TOOL IS CLAMPED DURING MACHINING
   RUNG wire#powerrail
      Contact( "DB331_EXTENDED_M_CODE_UNIT_1_STA_0".M_code[604] )
      wire#w1
      I_Contact( "DB331_EXTENDED_M_CODE_UNIT_1_STA_0".M_code[604] )
      wire#w2
      I_Contact( "DB341_M_UNIT_1_STA_0".M_CODES_UNIT_1_STA_0.Ack_M604 )
      I_Contact( "DB2120_MPP_ITC_IPC".RESET_FAULTS )
      Contact( "DB2440_GLOBAL_DATA".GLOBAL_DATA.ANY_PART_CYCLE_RUN )
      Coil( "DB341_M_UNIT_1_STA_0".M_CODES_UNIT_1_STA_0.M604 )
   END_RUNG
   RUNG wire#powerrail
      Contact( "DB341_M_UNIT_1_STA_0".M_CODES_UNIT_1_STA_0.M604 )
   END_RUNG wire#w1
   RUNG wire#w1
      I_Contact( "DB341_M_UNIT_1_STA_0".M_CODES_UNIT_1_STA_0.M604 )
   END_RUNG wire#w2
   // the same network as SCL:
   "DB341_M_UNIT_1_STA_0".M_CODES_UNIT_1_STA_0.M604 := ("DB331_EXTENDED_M_CODE_UNIT_1_STA_0".M_code[604] OR "DB341_M_UNIT_1_STA_0".M_CODES_UNIT_1_STA_0.M604) AND (NOT "DB331_EXTENDED_M_CODE_UNIT_1_STA_0".M_code[604] OR NOT "DB341_M_UNIT_1_STA_0".M_CODES_UNIT_1_STA_0.M604) AND NOT "DB341_M_UNIT_1_STA_0".M_CODES_UNIT_1_STA_0.Ack_M604 AND NOT "DB2120_MPP_ITC_IPC".RESET_FAULTS AND "DB2440_GLOBAL_DATA".GLOBAL_DATA.ANY_PART_CYCLE_RUN;
END_REGION

REGION Network 67: ACKNOWLEDGE M605-UNIT 1 FIXTURE 3 VERIFY PART AND TOOL IS CLAMPED LOW PRESSURE DURING MACHINING (WHEN TRUE DO). TOGGLED / ACKNOWLEDGE M46-VERIFY FIXTURE 1 PART AND TOOL IS CLAMPED DURING
   RUNG wire#powerrail
      Contact( "M_ZERO" )
      Coil( "DB341_M_UNIT_1_STA_0".M_CODES_UNIT_1_STA_0.Ack_M605 )
   END_RUNG
   // the same network as SCL:
   "DB341_M_UNIT_1_STA_0".M_CODES_UNIT_1_STA_0.Ack_M605 := "M_ZERO";
END_REGION

REGION Network 68: M605-UNIT 1 FIXTURE 3 VERIFY PART AND TOOL IS CLAMPED LOW PRESSURE DURING MACHINING (WHEN TRUE DO). TOGGLED / M46-VERIFY FIXTURE 1 PART AND TOOL IS CLAMPED DURING MACHINING
   RUNG wire#powerrail
      Contact( "DB331_EXTENDED_M_CODE_UNIT_1_STA_0".M_code[605] )
      wire#w1
      I_Contact( "DB331_EXTENDED_M_CODE_UNIT_1_STA_0".M_code[605] )
      wire#w2
      I_Contact( "DB341_M_UNIT_1_STA_0".M_CODES_UNIT_1_STA_0.Ack_M605 )
      I_Contact( "DB2120_MPP_ITC_IPC".RESET_FAULTS )
      Contact( "DB2440_GLOBAL_DATA".GLOBAL_DATA.ANY_PART_CYCLE_RUN )
      Coil( "DB341_M_UNIT_1_STA_0".M_CODES_UNIT_1_STA_0.M605 )
   END_RUNG
   RUNG wire#powerrail
      Contact( "DB341_M_UNIT_1_STA_0".M_CODES_UNIT_1_STA_0.M605 )
   END_RUNG wire#w1
   RUNG wire#w1
      I_Contact( "DB341_M_UNIT_1_STA_0".M_CODES_UNIT_1_STA_0.M605 )
   END_RUNG wire#w2
   // the same network as SCL:
   "DB341_M_UNIT_1_STA_0".M_CODES_UNIT_1_STA_0.M605 := ("DB331_EXTENDED_M_CODE_UNIT_1_STA_0".M_code[605] OR "DB341_M_UNIT_1_STA_0".M_CODES_UNIT_1_STA_0.M605) AND (NOT "DB331_EXTENDED_M_CODE_UNIT_1_STA_0".M_code[605] OR NOT "DB341_M_UNIT_1_STA_0".M_CODES_UNIT_1_STA_0.M605) AND NOT "DB341_M_UNIT_1_STA_0".M_CODES_UNIT_1_STA_0.Ack_M605 AND NOT "DB2120_MPP_ITC_IPC".RESET_FAULTS AND "DB2440_GLOBAL_DATA".GLOBAL_DATA.ANY_PART_CYCLE_RUN;
END_REGION

REGION Network 69: ACKNOWLEDGE M606-UNIT 1 FIXTURE 3 VERIFY PARTS ARE UNCLAMPED PARTS LOADING (WHEN TRUE DO). TOGGLED / ACKNOWLEDGE M47-VERIFY FIXTURE 2 PART AND TOOL IS CLAMPED DURING
   RUNG wire#powerrail
      Contact( "M_ZERO" )
      Coil( "DB341_M_UNIT_1_STA_0".M_CODES_UNIT_1_STA_0.Ack_M606 )
   END_RUNG
   // the same network as SCL:
   "DB341_M_UNIT_1_STA_0".M_CODES_UNIT_1_STA_0.Ack_M606 := "M_ZERO";
END_REGION

REGION Network 70: M606-UNIT 1 FIXTURE 3 VERIFY PARTS ARE UNCLAMPED PARTS LOADING (WHEN TRUE DO). TOGGLED / M47-VERIFY FIXTURE 2 PART AND TOOL IS CLAMPED DURING MACHINING
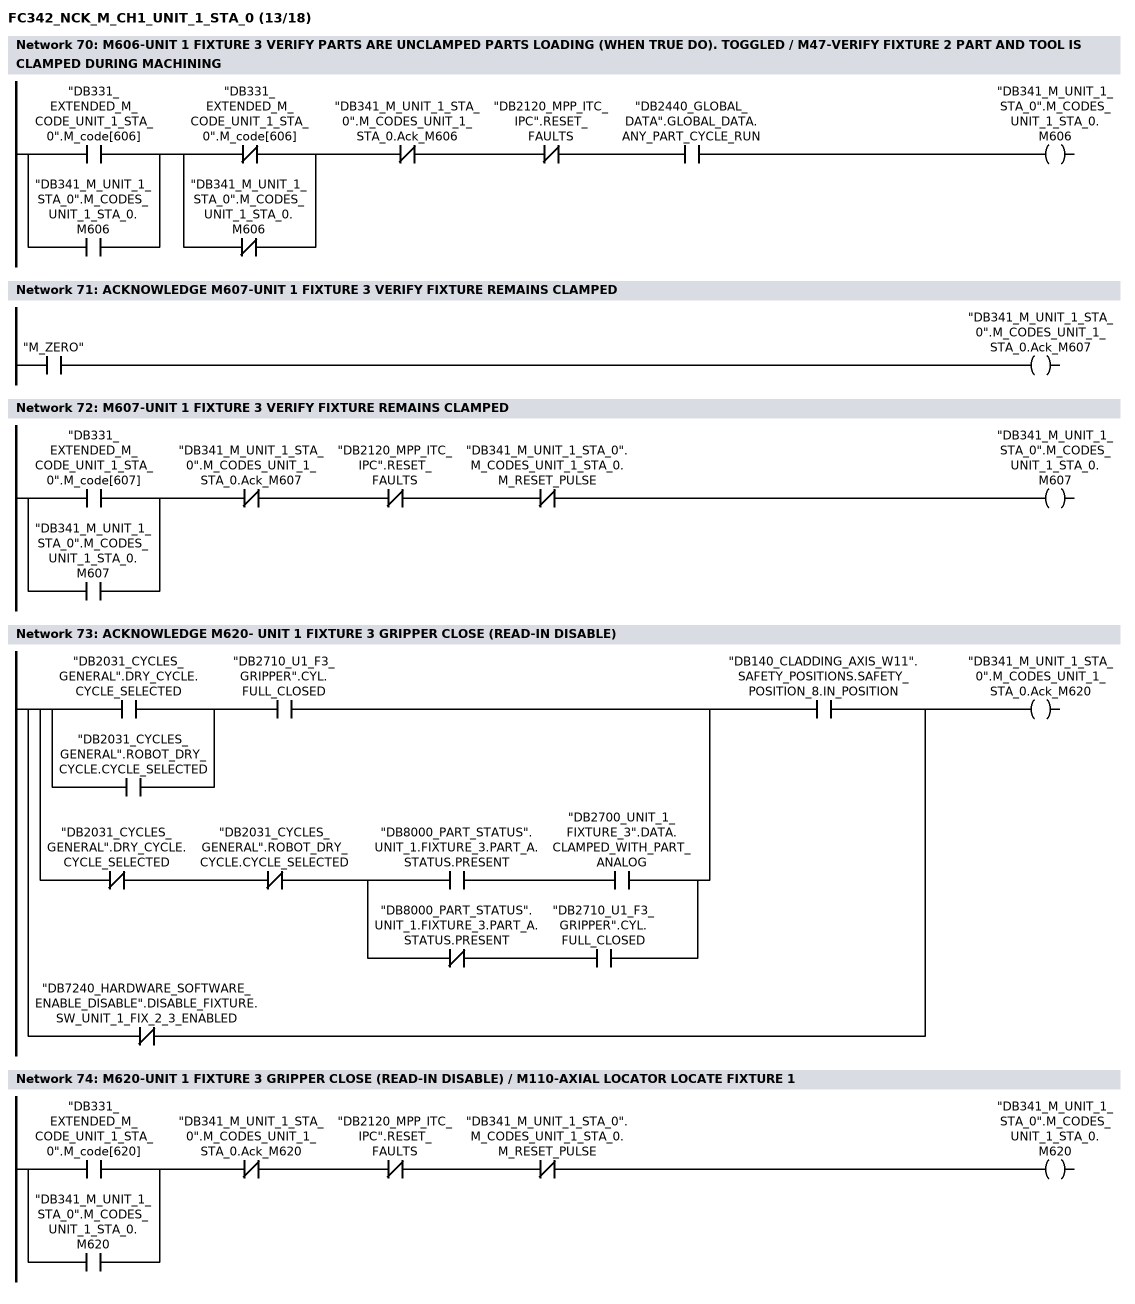
   RUNG wire#powerrail
      Contact( "DB331_EXTENDED_M_CODE_UNIT_1_STA_0".M_code[606] )
      wire#w1
      I_Contact( "DB331_EXTENDED_M_CODE_UNIT_1_STA_0".M_code[606] )
      wire#w2
      I_Contact( "DB341_M_UNIT_1_STA_0".M_CODES_UNIT_1_STA_0.Ack_M606 )
      I_Contact( "DB2120_MPP_ITC_IPC".RESET_FAULTS )
      Contact( "DB2440_GLOBAL_DATA".GLOBAL_DATA.ANY_PART_CYCLE_RUN )
      Coil( "DB341_M_UNIT_1_STA_0".M_CODES_UNIT_1_STA_0.M606 )
   END_RUNG
   RUNG wire#powerrail
      Contact( "DB341_M_UNIT_1_STA_0".M_CODES_UNIT_1_STA_0.M606 )
   END_RUNG wire#w1
   RUNG wire#w1
      I_Contact( "DB341_M_UNIT_1_STA_0".M_CODES_UNIT_1_STA_0.M606 )
   END_RUNG wire#w2
   // the same network as SCL:
   "DB341_M_UNIT_1_STA_0".M_CODES_UNIT_1_STA_0.M606 := ("DB331_EXTENDED_M_CODE_UNIT_1_STA_0".M_code[606] OR "DB341_M_UNIT_1_STA_0".M_CODES_UNIT_1_STA_0.M606) AND (NOT "DB331_EXTENDED_M_CODE_UNIT_1_STA_0".M_code[606] OR NOT "DB341_M_UNIT_1_STA_0".M_CODES_UNIT_1_STA_0.M606) AND NOT "DB341_M_UNIT_1_STA_0".M_CODES_UNIT_1_STA_0.Ack_M606 AND NOT "DB2120_MPP_ITC_IPC".RESET_FAULTS AND "DB2440_GLOBAL_DATA".GLOBAL_DATA.ANY_PART_CYCLE_RUN;
END_REGION

REGION Network 71: ACKNOWLEDGE M607-UNIT 1 FIXTURE 3 VERIFY FIXTURE REMAINS CLAMPED
   RUNG wire#powerrail
      Contact( "M_ZERO" )
      Coil( "DB341_M_UNIT_1_STA_0".M_CODES_UNIT_1_STA_0.Ack_M607 )
   END_RUNG
   // the same network as SCL:
   "DB341_M_UNIT_1_STA_0".M_CODES_UNIT_1_STA_0.Ack_M607 := "M_ZERO";
END_REGION

REGION Network 72: M607-UNIT 1 FIXTURE 3 VERIFY FIXTURE REMAINS CLAMPED
   RUNG wire#powerrail
      Contact( "DB331_EXTENDED_M_CODE_UNIT_1_STA_0".M_code[607] )
      wire#w1
      I_Contact( "DB341_M_UNIT_1_STA_0".M_CODES_UNIT_1_STA_0.Ack_M607 )
      I_Contact( "DB2120_MPP_ITC_IPC".RESET_FAULTS )
      I_Contact( "DB341_M_UNIT_1_STA_0".M_CODES_UNIT_1_STA_0.M_RESET_PULSE )
      Coil( "DB341_M_UNIT_1_STA_0".M_CODES_UNIT_1_STA_0.M607 )
   END_RUNG
   RUNG wire#powerrail
      Contact( "DB341_M_UNIT_1_STA_0".M_CODES_UNIT_1_STA_0.M607 )
   END_RUNG wire#w1
   // the same network as SCL:
   "DB341_M_UNIT_1_STA_0".M_CODES_UNIT_1_STA_0.M607 := ("DB331_EXTENDED_M_CODE_UNIT_1_STA_0".M_code[607] OR "DB341_M_UNIT_1_STA_0".M_CODES_UNIT_1_STA_0.M607) AND NOT "DB341_M_UNIT_1_STA_0".M_CODES_UNIT_1_STA_0.Ack_M607 AND NOT "DB2120_MPP_ITC_IPC".RESET_FAULTS AND NOT "DB341_M_UNIT_1_STA_0".M_CODES_UNIT_1_STA_0.M_RESET_PULSE;
END_REGION

REGION Network 73: ACKNOWLEDGE M620- UNIT 1 FIXTURE 3 GRIPPER CLOSE (READ-IN DISABLE)
   RUNG wire#powerrail
      Contact( "DB2031_CYCLES_GENERAL".DRY_CYCLE.CYCLE_SELECTED )
      wire#w1
      Contact( "DB2710_U1_F3_GRIPPER".CYL.FULL_CLOSED )
      wire#w2
      Contact( "DB140_CLADDING_AXIS_W11".SAFETY_POSITIONS.SAFETY_POSITION_8.IN_POSITION )
      wire#w4
      Coil( "DB341_M_UNIT_1_STA_0".M_CODES_UNIT_1_STA_0.Ack_M620 )
   END_RUNG
   RUNG wire#powerrail
      Contact( "DB2031_CYCLES_GENERAL".ROBOT_DRY_CYCLE.CYCLE_SELECTED )
   END_RUNG wire#w1
   RUNG wire#powerrail
      I_Contact( "DB2031_CYCLES_GENERAL".DRY_CYCLE.CYCLE_SELECTED )
      I_Contact( "DB2031_CYCLES_GENERAL".ROBOT_DRY_CYCLE.CYCLE_SELECTED )
      wire#w3
      Contact( "DB8000_PART_STATUS".UNIT_1.FIXTURE_3.PART_A.STATUS.PRESENT )
      Contact( "DB2700_UNIT_1_FIXTURE_3".DATA.CLAMPED_WITH_PART_ANALOG )
   END_RUNG wire#w2
   RUNG wire#w3
      I_Contact( "DB8000_PART_STATUS".UNIT_1.FIXTURE_3.PART_A.STATUS.PRESENT )
      Contact( "DB2710_U1_F3_GRIPPER".CYL.FULL_CLOSED )
   END_RUNG wire#w2
   RUNG wire#powerrail
      I_Contact( "DB7240_HARDWARE_SOFTWARE_ENABLE_DISABLE".DISABLE_FIXTURE.SW_UNIT_1_FIX_2_3_ENABLED )
   END_RUNG wire#w4
   // the same network as SCL:
   "DB341_M_UNIT_1_STA_0".M_CODES_UNIT_1_STA_0.Ack_M620 := (((("DB2031_CYCLES_GENERAL".DRY_CYCLE.CYCLE_SELECTED OR "DB2031_CYCLES_GENERAL".ROBOT_DRY_CYCLE.CYCLE_SELECTED) AND "DB2710_U1_F3_GRIPPER".CYL.FULL_CLOSED) OR (NOT "DB2031_CYCLES_GENERAL".DRY_CYCLE.CYCLE_SELECTED AND NOT "DB2031_CYCLES_GENERAL".ROBOT_DRY_CYCLE.CYCLE_SELECTED AND (("DB8000_PART_STATUS".UNIT_1.FIXTURE_3.PART_A.STATUS.PRESENT AND "DB2700_UNIT_1_FIXTURE_3".DATA.CLAMPED_WITH_PART_ANALOG) OR (NOT "DB8000_PART_STATUS".UNIT_1.FIXTURE_3.PART_A.STATUS.PRESENT AND "DB2710_U1_F3_GRIPPER".CYL.FULL_CLOSED)))) AND "DB140_CLADDING_AXIS_W11".SAFETY_POSITIONS.SAFETY_POSITION_8.IN_POSITION) OR NOT "DB7240_HARDWARE_SOFTWARE_ENABLE_DISABLE".DISABLE_FIXTURE.SW_UNIT_1_FIX_2_3_ENABLED;
END_REGION

REGION Network 74: M620-UNIT 1 FIXTURE 3 GRIPPER CLOSE (READ-IN DISABLE) / M110-AXIAL LOCATOR LOCATE FIXTURE 1
   RUNG wire#powerrail
      Contact( "DB331_EXTENDED_M_CODE_UNIT_1_STA_0".M_code[620] )
      wire#w1
      I_Contact( "DB341_M_UNIT_1_STA_0".M_CODES_UNIT_1_STA_0.Ack_M620 )
      I_Contact( "DB2120_MPP_ITC_IPC".RESET_FAULTS )
      I_Contact( "DB341_M_UNIT_1_STA_0".M_CODES_UNIT_1_STA_0.M_RESET_PULSE )
      Coil( "DB341_M_UNIT_1_STA_0".M_CODES_UNIT_1_STA_0.M620 )
   END_RUNG
   RUNG wire#powerrail
      Contact( "DB341_M_UNIT_1_STA_0".M_CODES_UNIT_1_STA_0.M620 )
   END_RUNG wire#w1
   // the same network as SCL:
   "DB341_M_UNIT_1_STA_0".M_CODES_UNIT_1_STA_0.M620 := ("DB331_EXTENDED_M_CODE_UNIT_1_STA_0".M_code[620] OR "DB341_M_UNIT_1_STA_0".M_CODES_UNIT_1_STA_0.M620) AND NOT "DB341_M_UNIT_1_STA_0".M_CODES_UNIT_1_STA_0.Ack_M620 AND NOT "DB2120_MPP_ITC_IPC".RESET_FAULTS AND NOT "DB341_M_UNIT_1_STA_0".M_CODES_UNIT_1_STA_0.M_RESET_PULSE;
END_REGION

REGION Network 75: ACKNOWLEDGE M621-UNIT 1 FIXTURE 3 GRIPPER CLOSE
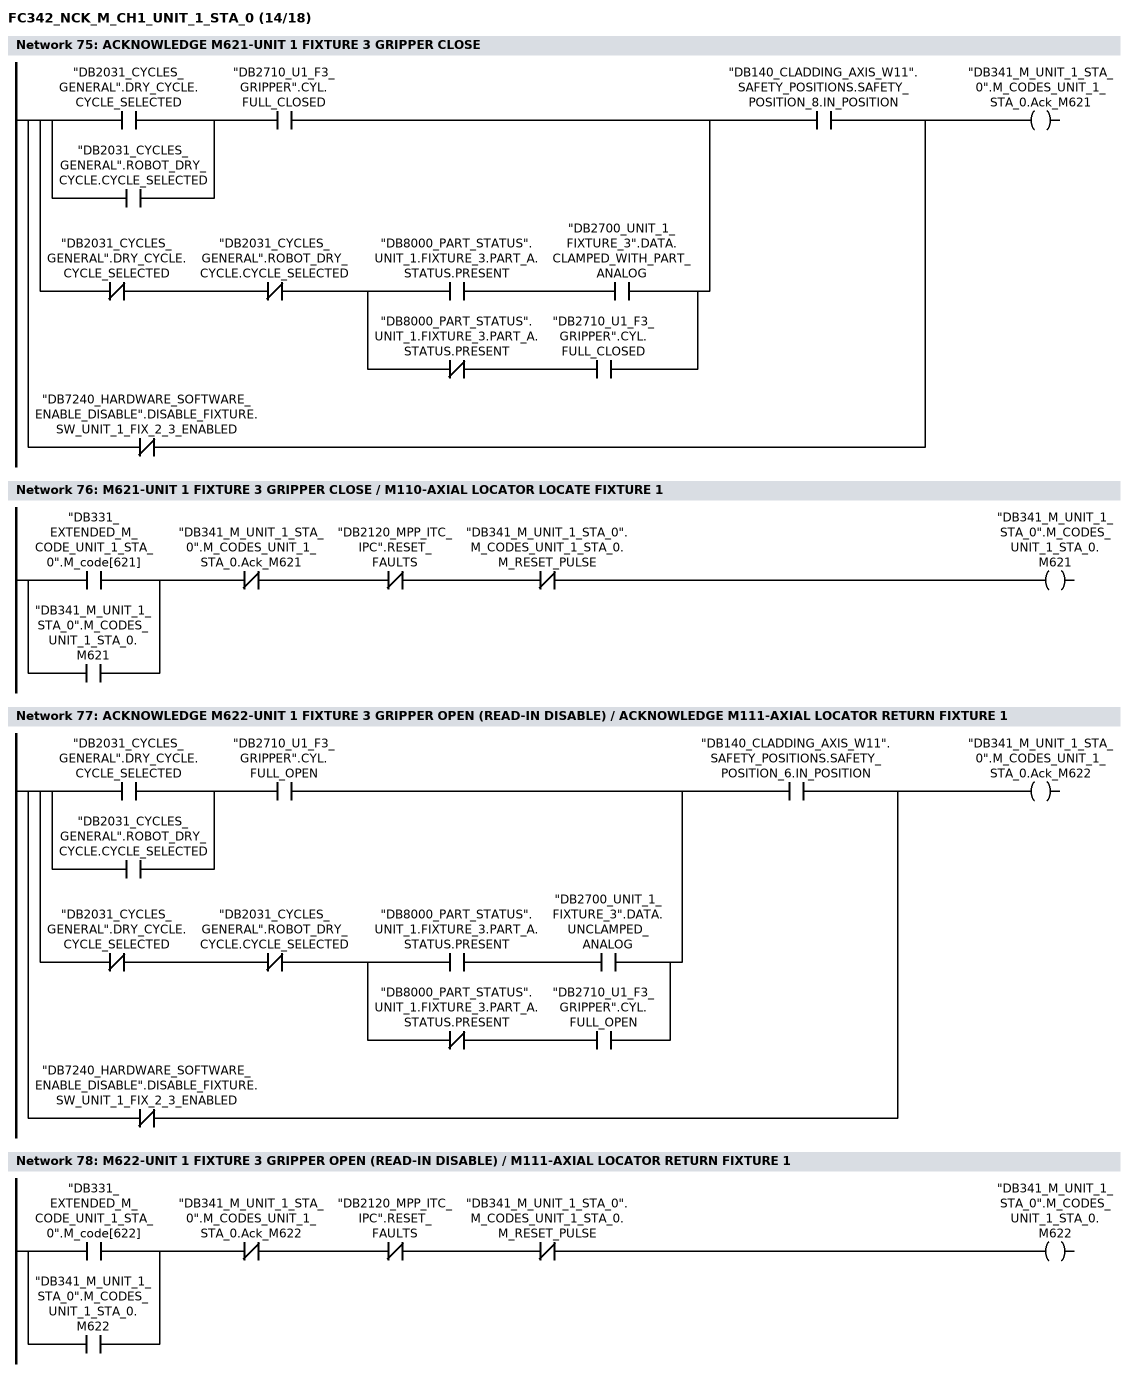
   RUNG wire#powerrail
      Contact( "DB2031_CYCLES_GENERAL".DRY_CYCLE.CYCLE_SELECTED )
      wire#w1
      Contact( "DB2710_U1_F3_GRIPPER".CYL.FULL_CLOSED )
      wire#w2
      Contact( "DB140_CLADDING_AXIS_W11".SAFETY_POSITIONS.SAFETY_POSITION_8.IN_POSITION )
      wire#w4
      Coil( "DB341_M_UNIT_1_STA_0".M_CODES_UNIT_1_STA_0.Ack_M621 )
   END_RUNG
   RUNG wire#powerrail
      Contact( "DB2031_CYCLES_GENERAL".ROBOT_DRY_CYCLE.CYCLE_SELECTED )
   END_RUNG wire#w1
   RUNG wire#powerrail
      I_Contact( "DB2031_CYCLES_GENERAL".DRY_CYCLE.CYCLE_SELECTED )
      I_Contact( "DB2031_CYCLES_GENERAL".ROBOT_DRY_CYCLE.CYCLE_SELECTED )
      wire#w3
      Contact( "DB8000_PART_STATUS".UNIT_1.FIXTURE_3.PART_A.STATUS.PRESENT )
      Contact( "DB2700_UNIT_1_FIXTURE_3".DATA.CLAMPED_WITH_PART_ANALOG )
   END_RUNG wire#w2
   RUNG wire#w3
      I_Contact( "DB8000_PART_STATUS".UNIT_1.FIXTURE_3.PART_A.STATUS.PRESENT )
      Contact( "DB2710_U1_F3_GRIPPER".CYL.FULL_CLOSED )
   END_RUNG wire#w2
   RUNG wire#powerrail
      I_Contact( "DB7240_HARDWARE_SOFTWARE_ENABLE_DISABLE".DISABLE_FIXTURE.SW_UNIT_1_FIX_2_3_ENABLED )
   END_RUNG wire#w4
   // the same network as SCL:
   "DB341_M_UNIT_1_STA_0".M_CODES_UNIT_1_STA_0.Ack_M621 := (((("DB2031_CYCLES_GENERAL".DRY_CYCLE.CYCLE_SELECTED OR "DB2031_CYCLES_GENERAL".ROBOT_DRY_CYCLE.CYCLE_SELECTED) AND "DB2710_U1_F3_GRIPPER".CYL.FULL_CLOSED) OR (NOT "DB2031_CYCLES_GENERAL".DRY_CYCLE.CYCLE_SELECTED AND NOT "DB2031_CYCLES_GENERAL".ROBOT_DRY_CYCLE.CYCLE_SELECTED AND (("DB8000_PART_STATUS".UNIT_1.FIXTURE_3.PART_A.STATUS.PRESENT AND "DB2700_UNIT_1_FIXTURE_3".DATA.CLAMPED_WITH_PART_ANALOG) OR (NOT "DB8000_PART_STATUS".UNIT_1.FIXTURE_3.PART_A.STATUS.PRESENT AND "DB2710_U1_F3_GRIPPER".CYL.FULL_CLOSED)))) AND "DB140_CLADDING_AXIS_W11".SAFETY_POSITIONS.SAFETY_POSITION_8.IN_POSITION) OR NOT "DB7240_HARDWARE_SOFTWARE_ENABLE_DISABLE".DISABLE_FIXTURE.SW_UNIT_1_FIX_2_3_ENABLED;
END_REGION

REGION Network 76: M621-UNIT 1 FIXTURE 3 GRIPPER CLOSE / M110-AXIAL LOCATOR LOCATE FIXTURE 1
   RUNG wire#powerrail
      Contact( "DB331_EXTENDED_M_CODE_UNIT_1_STA_0".M_code[621] )
      wire#w1
      I_Contact( "DB341_M_UNIT_1_STA_0".M_CODES_UNIT_1_STA_0.Ack_M621 )
      I_Contact( "DB2120_MPP_ITC_IPC".RESET_FAULTS )
      I_Contact( "DB341_M_UNIT_1_STA_0".M_CODES_UNIT_1_STA_0.M_RESET_PULSE )
      Coil( "DB341_M_UNIT_1_STA_0".M_CODES_UNIT_1_STA_0.M621 )
   END_RUNG
   RUNG wire#powerrail
      Contact( "DB341_M_UNIT_1_STA_0".M_CODES_UNIT_1_STA_0.M621 )
   END_RUNG wire#w1
   // the same network as SCL:
   "DB341_M_UNIT_1_STA_0".M_CODES_UNIT_1_STA_0.M621 := ("DB331_EXTENDED_M_CODE_UNIT_1_STA_0".M_code[621] OR "DB341_M_UNIT_1_STA_0".M_CODES_UNIT_1_STA_0.M621) AND NOT "DB341_M_UNIT_1_STA_0".M_CODES_UNIT_1_STA_0.Ack_M621 AND NOT "DB2120_MPP_ITC_IPC".RESET_FAULTS AND NOT "DB341_M_UNIT_1_STA_0".M_CODES_UNIT_1_STA_0.M_RESET_PULSE;
END_REGION

REGION Network 77: ACKNOWLEDGE M622-UNIT 1 FIXTURE 3 GRIPPER OPEN (READ-IN DISABLE) / ACKNOWLEDGE M111-AXIAL LOCATOR RETURN FIXTURE 1
   RUNG wire#powerrail
      Contact( "DB2031_CYCLES_GENERAL".DRY_CYCLE.CYCLE_SELECTED )
      wire#w1
      Contact( "DB2710_U1_F3_GRIPPER".CYL.FULL_OPEN )
      wire#w2
      Contact( "DB140_CLADDING_AXIS_W11".SAFETY_POSITIONS.SAFETY_POSITION_6.IN_POSITION )
      wire#w4
      Coil( "DB341_M_UNIT_1_STA_0".M_CODES_UNIT_1_STA_0.Ack_M622 )
   END_RUNG
   RUNG wire#powerrail
      Contact( "DB2031_CYCLES_GENERAL".ROBOT_DRY_CYCLE.CYCLE_SELECTED )
   END_RUNG wire#w1
   RUNG wire#powerrail
      I_Contact( "DB2031_CYCLES_GENERAL".DRY_CYCLE.CYCLE_SELECTED )
      I_Contact( "DB2031_CYCLES_GENERAL".ROBOT_DRY_CYCLE.CYCLE_SELECTED )
      wire#w3
      Contact( "DB8000_PART_STATUS".UNIT_1.FIXTURE_3.PART_A.STATUS.PRESENT )
      Contact( "DB2700_UNIT_1_FIXTURE_3".DATA.UNCLAMPED_ANALOG )
   END_RUNG wire#w2
   RUNG wire#w3
      I_Contact( "DB8000_PART_STATUS".UNIT_1.FIXTURE_3.PART_A.STATUS.PRESENT )
      Contact( "DB2710_U1_F3_GRIPPER".CYL.FULL_OPEN )
   END_RUNG wire#w2
   RUNG wire#powerrail
      I_Contact( "DB7240_HARDWARE_SOFTWARE_ENABLE_DISABLE".DISABLE_FIXTURE.SW_UNIT_1_FIX_2_3_ENABLED )
   END_RUNG wire#w4
   // the same network as SCL:
   "DB341_M_UNIT_1_STA_0".M_CODES_UNIT_1_STA_0.Ack_M622 := (((("DB2031_CYCLES_GENERAL".DRY_CYCLE.CYCLE_SELECTED OR "DB2031_CYCLES_GENERAL".ROBOT_DRY_CYCLE.CYCLE_SELECTED) AND "DB2710_U1_F3_GRIPPER".CYL.FULL_OPEN) OR (NOT "DB2031_CYCLES_GENERAL".DRY_CYCLE.CYCLE_SELECTED AND NOT "DB2031_CYCLES_GENERAL".ROBOT_DRY_CYCLE.CYCLE_SELECTED AND (("DB8000_PART_STATUS".UNIT_1.FIXTURE_3.PART_A.STATUS.PRESENT AND "DB2700_UNIT_1_FIXTURE_3".DATA.UNCLAMPED_ANALOG) OR (NOT "DB8000_PART_STATUS".UNIT_1.FIXTURE_3.PART_A.STATUS.PRESENT AND "DB2710_U1_F3_GRIPPER".CYL.FULL_OPEN)))) AND "DB140_CLADDING_AXIS_W11".SAFETY_POSITIONS.SAFETY_POSITION_6.IN_POSITION) OR NOT "DB7240_HARDWARE_SOFTWARE_ENABLE_DISABLE".DISABLE_FIXTURE.SW_UNIT_1_FIX_2_3_ENABLED;
END_REGION

REGION Network 78: M622-UNIT 1 FIXTURE 3 GRIPPER OPEN (READ-IN DISABLE) / M111-AXIAL LOCATOR RETURN FIXTURE 1
   RUNG wire#powerrail
      Contact( "DB331_EXTENDED_M_CODE_UNIT_1_STA_0".M_code[622] )
      wire#w1
      I_Contact( "DB341_M_UNIT_1_STA_0".M_CODES_UNIT_1_STA_0.Ack_M622 )
      I_Contact( "DB2120_MPP_ITC_IPC".RESET_FAULTS )
      I_Contact( "DB341_M_UNIT_1_STA_0".M_CODES_UNIT_1_STA_0.M_RESET_PULSE )
      Coil( "DB341_M_UNIT_1_STA_0".M_CODES_UNIT_1_STA_0.M622 )
   END_RUNG
   RUNG wire#powerrail
      Contact( "DB341_M_UNIT_1_STA_0".M_CODES_UNIT_1_STA_0.M622 )
   END_RUNG wire#w1
   // the same network as SCL:
   "DB341_M_UNIT_1_STA_0".M_CODES_UNIT_1_STA_0.M622 := ("DB331_EXTENDED_M_CODE_UNIT_1_STA_0".M_code[622] OR "DB341_M_UNIT_1_STA_0".M_CODES_UNIT_1_STA_0.M622) AND NOT "DB341_M_UNIT_1_STA_0".M_CODES_UNIT_1_STA_0.Ack_M622 AND NOT "DB2120_MPP_ITC_IPC".RESET_FAULTS AND NOT "DB341_M_UNIT_1_STA_0".M_CODES_UNIT_1_STA_0.M_RESET_PULSE;
END_REGION

REGION Network 79: ACKNOWLEDGE M623-UNIT 1 FIXTURE 3 GRIPPER OPEN / ACKNOWLEDGE M111-AXIAL LOCATOR RETURN FIXTURE 1
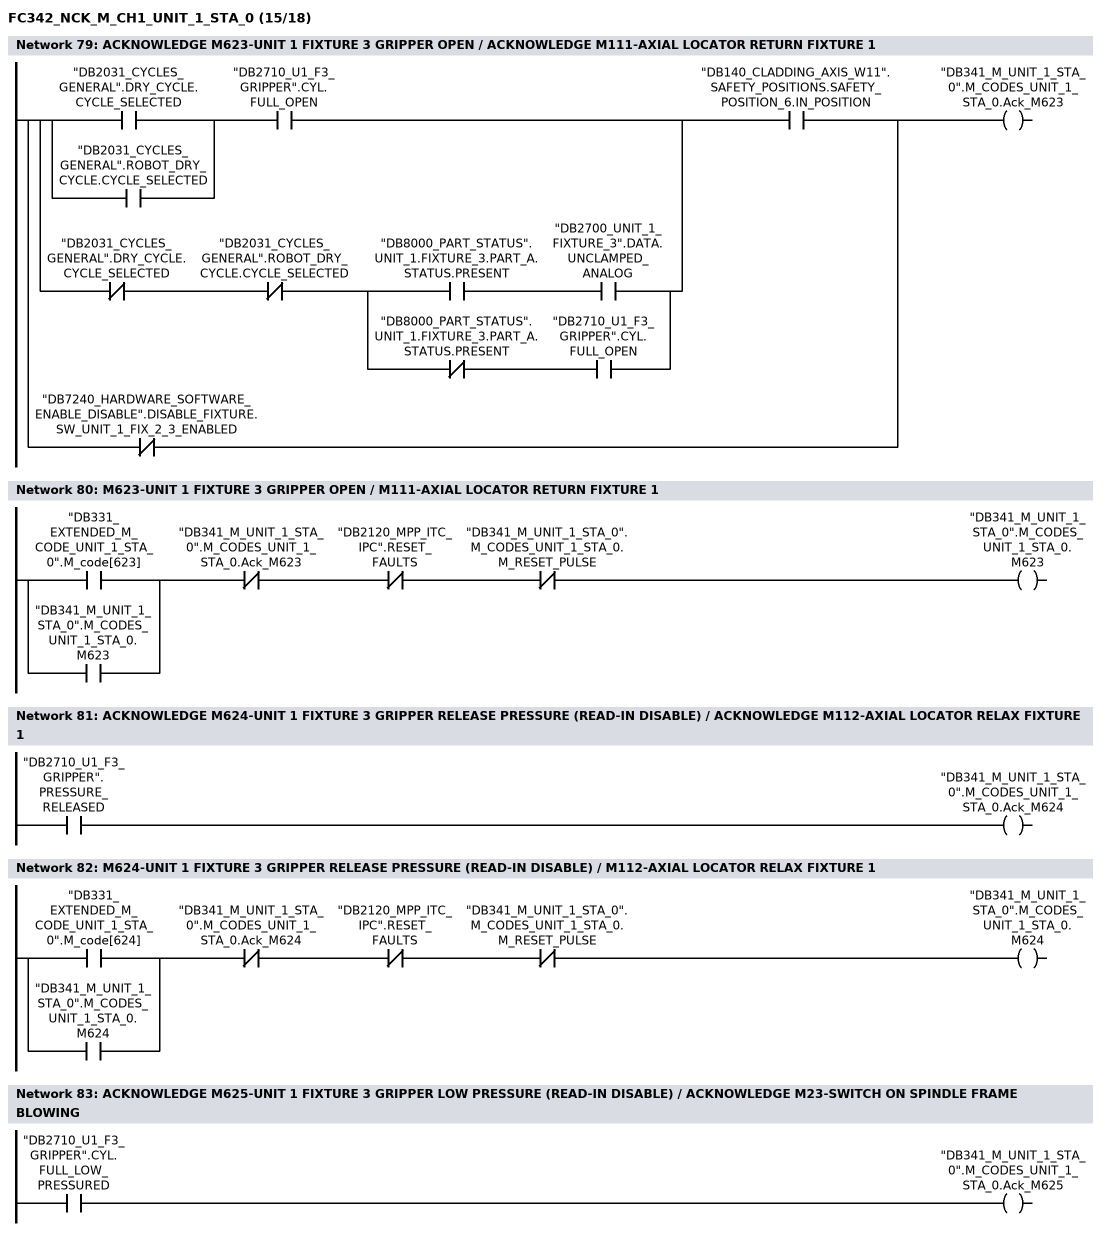
   RUNG wire#powerrail
      Contact( "DB2031_CYCLES_GENERAL".DRY_CYCLE.CYCLE_SELECTED )
      wire#w1
      Contact( "DB2710_U1_F3_GRIPPER".CYL.FULL_OPEN )
      wire#w2
      Contact( "DB140_CLADDING_AXIS_W11".SAFETY_POSITIONS.SAFETY_POSITION_6.IN_POSITION )
      wire#w4
      Coil( "DB341_M_UNIT_1_STA_0".M_CODES_UNIT_1_STA_0.Ack_M623 )
   END_RUNG
   RUNG wire#powerrail
      Contact( "DB2031_CYCLES_GENERAL".ROBOT_DRY_CYCLE.CYCLE_SELECTED )
   END_RUNG wire#w1
   RUNG wire#powerrail
      I_Contact( "DB2031_CYCLES_GENERAL".DRY_CYCLE.CYCLE_SELECTED )
      I_Contact( "DB2031_CYCLES_GENERAL".ROBOT_DRY_CYCLE.CYCLE_SELECTED )
      wire#w3
      Contact( "DB8000_PART_STATUS".UNIT_1.FIXTURE_3.PART_A.STATUS.PRESENT )
      Contact( "DB2700_UNIT_1_FIXTURE_3".DATA.UNCLAMPED_ANALOG )
   END_RUNG wire#w2
   RUNG wire#w3
      I_Contact( "DB8000_PART_STATUS".UNIT_1.FIXTURE_3.PART_A.STATUS.PRESENT )
      Contact( "DB2710_U1_F3_GRIPPER".CYL.FULL_OPEN )
   END_RUNG wire#w2
   RUNG wire#powerrail
      I_Contact( "DB7240_HARDWARE_SOFTWARE_ENABLE_DISABLE".DISABLE_FIXTURE.SW_UNIT_1_FIX_2_3_ENABLED )
   END_RUNG wire#w4
   // the same network as SCL:
   "DB341_M_UNIT_1_STA_0".M_CODES_UNIT_1_STA_0.Ack_M623 := (((("DB2031_CYCLES_GENERAL".DRY_CYCLE.CYCLE_SELECTED OR "DB2031_CYCLES_GENERAL".ROBOT_DRY_CYCLE.CYCLE_SELECTED) AND "DB2710_U1_F3_GRIPPER".CYL.FULL_OPEN) OR (NOT "DB2031_CYCLES_GENERAL".DRY_CYCLE.CYCLE_SELECTED AND NOT "DB2031_CYCLES_GENERAL".ROBOT_DRY_CYCLE.CYCLE_SELECTED AND (("DB8000_PART_STATUS".UNIT_1.FIXTURE_3.PART_A.STATUS.PRESENT AND "DB2700_UNIT_1_FIXTURE_3".DATA.UNCLAMPED_ANALOG) OR (NOT "DB8000_PART_STATUS".UNIT_1.FIXTURE_3.PART_A.STATUS.PRESENT AND "DB2710_U1_F3_GRIPPER".CYL.FULL_OPEN)))) AND "DB140_CLADDING_AXIS_W11".SAFETY_POSITIONS.SAFETY_POSITION_6.IN_POSITION) OR NOT "DB7240_HARDWARE_SOFTWARE_ENABLE_DISABLE".DISABLE_FIXTURE.SW_UNIT_1_FIX_2_3_ENABLED;
END_REGION

REGION Network 80: M623-UNIT 1 FIXTURE 3 GRIPPER OPEN / M111-AXIAL LOCATOR RETURN FIXTURE 1
   RUNG wire#powerrail
      Contact( "DB331_EXTENDED_M_CODE_UNIT_1_STA_0".M_code[623] )
      wire#w1
      I_Contact( "DB341_M_UNIT_1_STA_0".M_CODES_UNIT_1_STA_0.Ack_M623 )
      I_Contact( "DB2120_MPP_ITC_IPC".RESET_FAULTS )
      I_Contact( "DB341_M_UNIT_1_STA_0".M_CODES_UNIT_1_STA_0.M_RESET_PULSE )
      Coil( "DB341_M_UNIT_1_STA_0".M_CODES_UNIT_1_STA_0.M623 )
   END_RUNG
   RUNG wire#powerrail
      Contact( "DB341_M_UNIT_1_STA_0".M_CODES_UNIT_1_STA_0.M623 )
   END_RUNG wire#w1
   // the same network as SCL:
   "DB341_M_UNIT_1_STA_0".M_CODES_UNIT_1_STA_0.M623 := ("DB331_EXTENDED_M_CODE_UNIT_1_STA_0".M_code[623] OR "DB341_M_UNIT_1_STA_0".M_CODES_UNIT_1_STA_0.M623) AND NOT "DB341_M_UNIT_1_STA_0".M_CODES_UNIT_1_STA_0.Ack_M623 AND NOT "DB2120_MPP_ITC_IPC".RESET_FAULTS AND NOT "DB341_M_UNIT_1_STA_0".M_CODES_UNIT_1_STA_0.M_RESET_PULSE;
END_REGION

REGION Network 81: ACKNOWLEDGE M624-UNIT 1 FIXTURE 3 GRIPPER RELEASE PRESSURE (READ-IN DISABLE) / ACKNOWLEDGE M112-AXIAL LOCATOR RELAX FIXTURE 1
   RUNG wire#powerrail
      Contact( "DB2710_U1_F3_GRIPPER".PRESSURE_RELEASED )
      Coil( "DB341_M_UNIT_1_STA_0".M_CODES_UNIT_1_STA_0.Ack_M624 )
   END_RUNG
   // the same network as SCL:
   "DB341_M_UNIT_1_STA_0".M_CODES_UNIT_1_STA_0.Ack_M624 := "DB2710_U1_F3_GRIPPER".PRESSURE_RELEASED;
END_REGION

REGION Network 82: M624-UNIT 1 FIXTURE 3 GRIPPER RELEASE PRESSURE (READ-IN DISABLE) / M112-AXIAL LOCATOR RELAX FIXTURE 1
   RUNG wire#powerrail
      Contact( "DB331_EXTENDED_M_CODE_UNIT_1_STA_0".M_code[624] )
      wire#w1
      I_Contact( "DB341_M_UNIT_1_STA_0".M_CODES_UNIT_1_STA_0.Ack_M624 )
      I_Contact( "DB2120_MPP_ITC_IPC".RESET_FAULTS )
      I_Contact( "DB341_M_UNIT_1_STA_0".M_CODES_UNIT_1_STA_0.M_RESET_PULSE )
      Coil( "DB341_M_UNIT_1_STA_0".M_CODES_UNIT_1_STA_0.M624 )
   END_RUNG
   RUNG wire#powerrail
      Contact( "DB341_M_UNIT_1_STA_0".M_CODES_UNIT_1_STA_0.M624 )
   END_RUNG wire#w1
   // the same network as SCL:
   "DB341_M_UNIT_1_STA_0".M_CODES_UNIT_1_STA_0.M624 := ("DB331_EXTENDED_M_CODE_UNIT_1_STA_0".M_code[624] OR "DB341_M_UNIT_1_STA_0".M_CODES_UNIT_1_STA_0.M624) AND NOT "DB341_M_UNIT_1_STA_0".M_CODES_UNIT_1_STA_0.Ack_M624 AND NOT "DB2120_MPP_ITC_IPC".RESET_FAULTS AND NOT "DB341_M_UNIT_1_STA_0".M_CODES_UNIT_1_STA_0.M_RESET_PULSE;
END_REGION

REGION Network 83: ACKNOWLEDGE M625-UNIT 1 FIXTURE 3 GRIPPER LOW PRESSURE (READ-IN DISABLE) / ACKNOWLEDGE M23-SWITCH ON SPINDLE FRAME BLOWING
   RUNG wire#powerrail
      Contact( "DB2710_U1_F3_GRIPPER".CYL.FULL_LOW_PRESSURED )
      Coil( "DB341_M_UNIT_1_STA_0".M_CODES_UNIT_1_STA_0.Ack_M625 )
   END_RUNG
   // the same network as SCL:
   "DB341_M_UNIT_1_STA_0".M_CODES_UNIT_1_STA_0.Ack_M625 := "DB2710_U1_F3_GRIPPER".CYL.FULL_LOW_PRESSURED;
END_REGION

REGION Network 84: M625-UNIT 1 FIXTURE 3 GRIPPER LOW PRESSURE (READ-IN DISABLE) / M23-SWITCH ON SPINDLE FRAME BLOWING
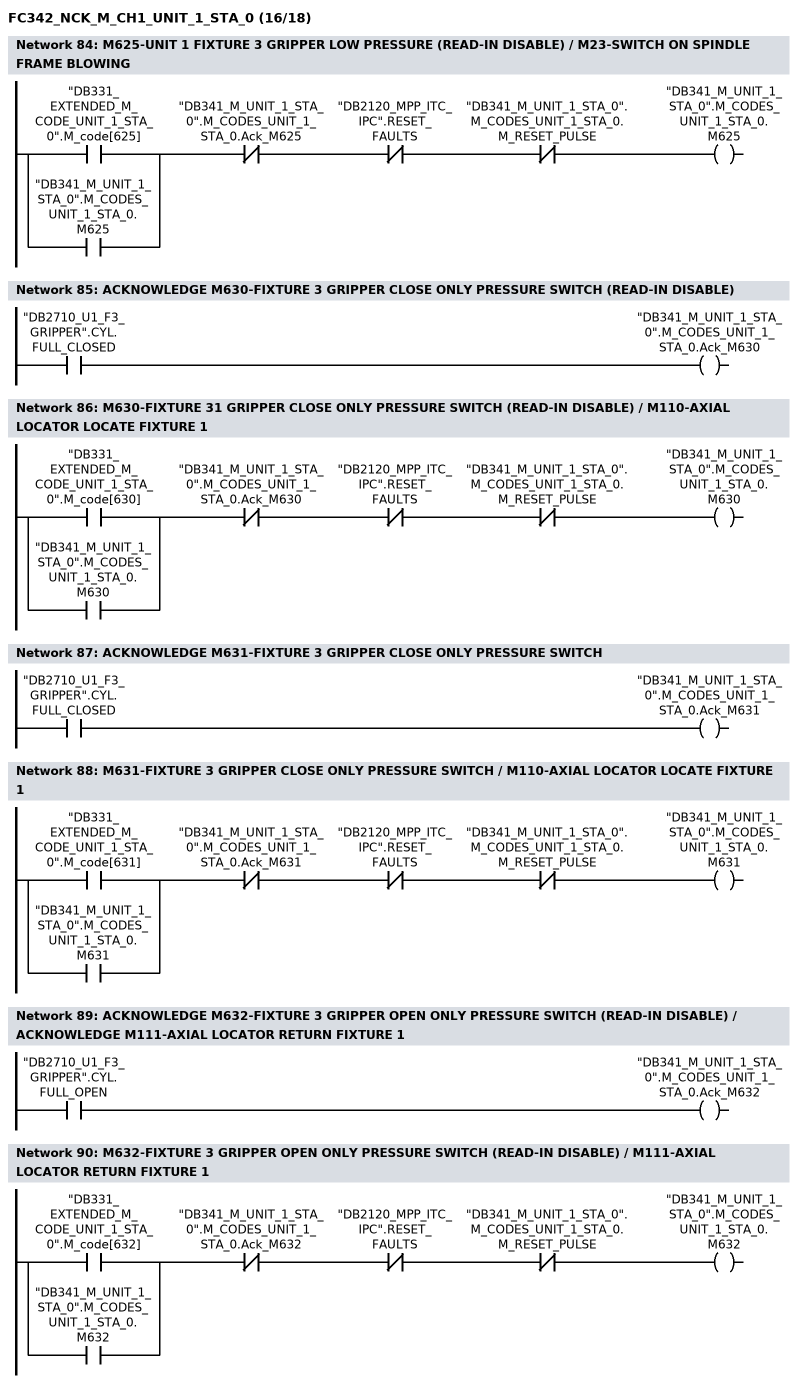
   RUNG wire#powerrail
      Contact( "DB331_EXTENDED_M_CODE_UNIT_1_STA_0".M_code[625] )
      wire#w1
      I_Contact( "DB341_M_UNIT_1_STA_0".M_CODES_UNIT_1_STA_0.Ack_M625 )
      I_Contact( "DB2120_MPP_ITC_IPC".RESET_FAULTS )
      I_Contact( "DB341_M_UNIT_1_STA_0".M_CODES_UNIT_1_STA_0.M_RESET_PULSE )
      Coil( "DB341_M_UNIT_1_STA_0".M_CODES_UNIT_1_STA_0.M625 )
   END_RUNG
   RUNG wire#powerrail
      Contact( "DB341_M_UNIT_1_STA_0".M_CODES_UNIT_1_STA_0.M625 )
   END_RUNG wire#w1
   // the same network as SCL:
   "DB341_M_UNIT_1_STA_0".M_CODES_UNIT_1_STA_0.M625 := ("DB331_EXTENDED_M_CODE_UNIT_1_STA_0".M_code[625] OR "DB341_M_UNIT_1_STA_0".M_CODES_UNIT_1_STA_0.M625) AND NOT "DB341_M_UNIT_1_STA_0".M_CODES_UNIT_1_STA_0.Ack_M625 AND NOT "DB2120_MPP_ITC_IPC".RESET_FAULTS AND NOT "DB341_M_UNIT_1_STA_0".M_CODES_UNIT_1_STA_0.M_RESET_PULSE;
END_REGION

REGION Network 85: ACKNOWLEDGE M630-FIXTURE 3 GRIPPER CLOSE ONLY PRESSURE SWITCH (READ-IN DISABLE)
   RUNG wire#powerrail
      Contact( "DB2710_U1_F3_GRIPPER".CYL.FULL_CLOSED )
      Coil( "DB341_M_UNIT_1_STA_0".M_CODES_UNIT_1_STA_0.Ack_M630 )
   END_RUNG
   // the same network as SCL:
   "DB341_M_UNIT_1_STA_0".M_CODES_UNIT_1_STA_0.Ack_M630 := "DB2710_U1_F3_GRIPPER".CYL.FULL_CLOSED;
END_REGION

REGION Network 86: M630-FIXTURE 31 GRIPPER CLOSE ONLY PRESSURE SWITCH (READ-IN DISABLE) / M110-AXIAL LOCATOR LOCATE FIXTURE 1
   RUNG wire#powerrail
      Contact( "DB331_EXTENDED_M_CODE_UNIT_1_STA_0".M_code[630] )
      wire#w1
      I_Contact( "DB341_M_UNIT_1_STA_0".M_CODES_UNIT_1_STA_0.Ack_M630 )
      I_Contact( "DB2120_MPP_ITC_IPC".RESET_FAULTS )
      I_Contact( "DB341_M_UNIT_1_STA_0".M_CODES_UNIT_1_STA_0.M_RESET_PULSE )
      Coil( "DB341_M_UNIT_1_STA_0".M_CODES_UNIT_1_STA_0.M630 )
   END_RUNG
   RUNG wire#powerrail
      Contact( "DB341_M_UNIT_1_STA_0".M_CODES_UNIT_1_STA_0.M630 )
   END_RUNG wire#w1
   // the same network as SCL:
   "DB341_M_UNIT_1_STA_0".M_CODES_UNIT_1_STA_0.M630 := ("DB331_EXTENDED_M_CODE_UNIT_1_STA_0".M_code[630] OR "DB341_M_UNIT_1_STA_0".M_CODES_UNIT_1_STA_0.M630) AND NOT "DB341_M_UNIT_1_STA_0".M_CODES_UNIT_1_STA_0.Ack_M630 AND NOT "DB2120_MPP_ITC_IPC".RESET_FAULTS AND NOT "DB341_M_UNIT_1_STA_0".M_CODES_UNIT_1_STA_0.M_RESET_PULSE;
END_REGION

REGION Network 87: ACKNOWLEDGE M631-FIXTURE 3 GRIPPER CLOSE ONLY PRESSURE SWITCH
   RUNG wire#powerrail
      Contact( "DB2710_U1_F3_GRIPPER".CYL.FULL_CLOSED )
      Coil( "DB341_M_UNIT_1_STA_0".M_CODES_UNIT_1_STA_0.Ack_M631 )
   END_RUNG
   // the same network as SCL:
   "DB341_M_UNIT_1_STA_0".M_CODES_UNIT_1_STA_0.Ack_M631 := "DB2710_U1_F3_GRIPPER".CYL.FULL_CLOSED;
END_REGION

REGION Network 88: M631-FIXTURE 3 GRIPPER CLOSE ONLY PRESSURE SWITCH / M110-AXIAL LOCATOR LOCATE FIXTURE 1
   RUNG wire#powerrail
      Contact( "DB331_EXTENDED_M_CODE_UNIT_1_STA_0".M_code[631] )
      wire#w1
      I_Contact( "DB341_M_UNIT_1_STA_0".M_CODES_UNIT_1_STA_0.Ack_M631 )
      I_Contact( "DB2120_MPP_ITC_IPC".RESET_FAULTS )
      I_Contact( "DB341_M_UNIT_1_STA_0".M_CODES_UNIT_1_STA_0.M_RESET_PULSE )
      Coil( "DB341_M_UNIT_1_STA_0".M_CODES_UNIT_1_STA_0.M631 )
   END_RUNG
   RUNG wire#powerrail
      Contact( "DB341_M_UNIT_1_STA_0".M_CODES_UNIT_1_STA_0.M631 )
   END_RUNG wire#w1
   // the same network as SCL:
   "DB341_M_UNIT_1_STA_0".M_CODES_UNIT_1_STA_0.M631 := ("DB331_EXTENDED_M_CODE_UNIT_1_STA_0".M_code[631] OR "DB341_M_UNIT_1_STA_0".M_CODES_UNIT_1_STA_0.M631) AND NOT "DB341_M_UNIT_1_STA_0".M_CODES_UNIT_1_STA_0.Ack_M631 AND NOT "DB2120_MPP_ITC_IPC".RESET_FAULTS AND NOT "DB341_M_UNIT_1_STA_0".M_CODES_UNIT_1_STA_0.M_RESET_PULSE;
END_REGION

REGION Network 89: ACKNOWLEDGE M632-FIXTURE 3 GRIPPER OPEN ONLY PRESSURE SWITCH (READ-IN DISABLE) / ACKNOWLEDGE M111-AXIAL LOCATOR RETURN FIXTURE 1
   RUNG wire#powerrail
      Contact( "DB2710_U1_F3_GRIPPER".CYL.FULL_OPEN )
      Coil( "DB341_M_UNIT_1_STA_0".M_CODES_UNIT_1_STA_0.Ack_M632 )
   END_RUNG
   // the same network as SCL:
   "DB341_M_UNIT_1_STA_0".M_CODES_UNIT_1_STA_0.Ack_M632 := "DB2710_U1_F3_GRIPPER".CYL.FULL_OPEN;
END_REGION

REGION Network 90: M632-FIXTURE 3 GRIPPER OPEN ONLY PRESSURE SWITCH (READ-IN DISABLE) / M111-AXIAL LOCATOR RETURN FIXTURE 1
   RUNG wire#powerrail
      Contact( "DB331_EXTENDED_M_CODE_UNIT_1_STA_0".M_code[632] )
      wire#w1
      I_Contact( "DB341_M_UNIT_1_STA_0".M_CODES_UNIT_1_STA_0.Ack_M632 )
      I_Contact( "DB2120_MPP_ITC_IPC".RESET_FAULTS )
      I_Contact( "DB341_M_UNIT_1_STA_0".M_CODES_UNIT_1_STA_0.M_RESET_PULSE )
      Coil( "DB341_M_UNIT_1_STA_0".M_CODES_UNIT_1_STA_0.M632 )
   END_RUNG
   RUNG wire#powerrail
      Contact( "DB341_M_UNIT_1_STA_0".M_CODES_UNIT_1_STA_0.M632 )
   END_RUNG wire#w1
   // the same network as SCL:
   "DB341_M_UNIT_1_STA_0".M_CODES_UNIT_1_STA_0.M632 := ("DB331_EXTENDED_M_CODE_UNIT_1_STA_0".M_code[632] OR "DB341_M_UNIT_1_STA_0".M_CODES_UNIT_1_STA_0.M632) AND NOT "DB341_M_UNIT_1_STA_0".M_CODES_UNIT_1_STA_0.Ack_M632 AND NOT "DB2120_MPP_ITC_IPC".RESET_FAULTS AND NOT "DB341_M_UNIT_1_STA_0".M_CODES_UNIT_1_STA_0.M_RESET_PULSE;
END_REGION

REGION Network 91: ACKNOWLEDGE M633-FIXTURE 3 GRIPPER OPEN ONLY PRESSURE SWITCH / ACKNOWLEDGE M111-AXIAL LOCATOR RETURN FIXTURE 1
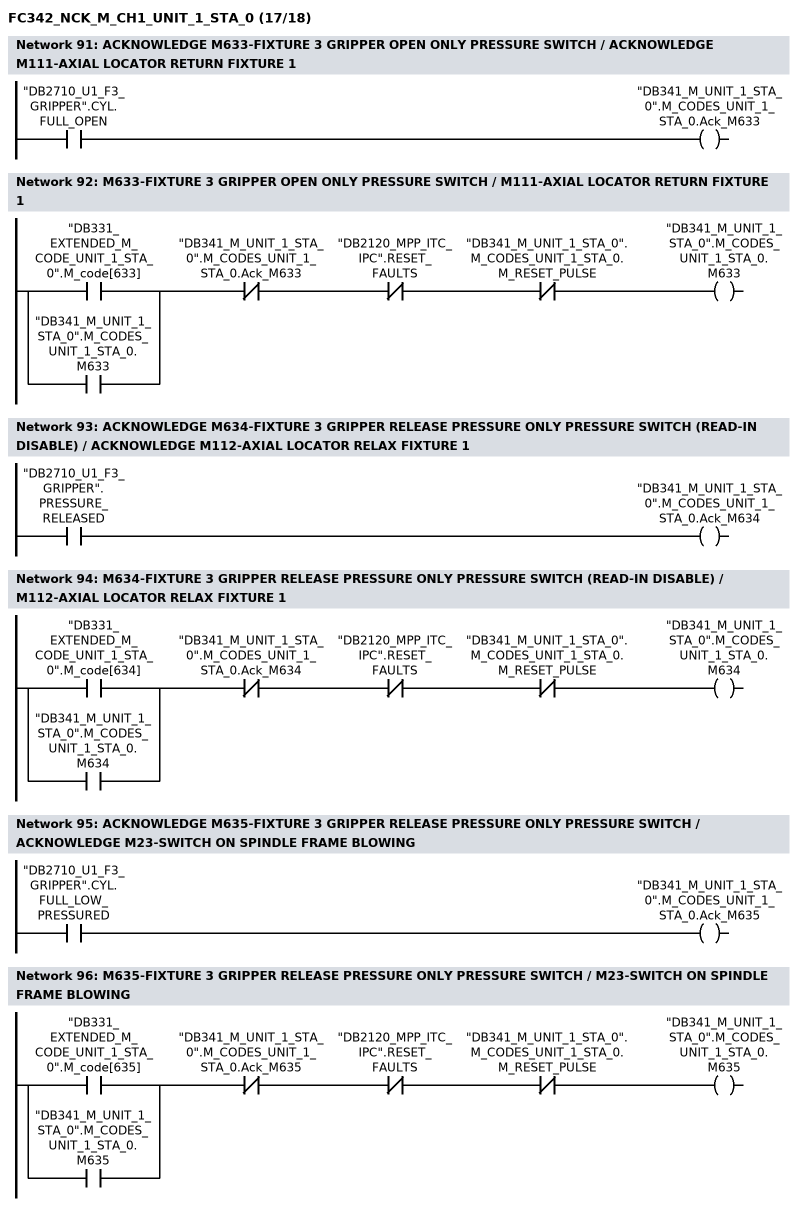
   RUNG wire#powerrail
      Contact( "DB2710_U1_F3_GRIPPER".CYL.FULL_OPEN )
      Coil( "DB341_M_UNIT_1_STA_0".M_CODES_UNIT_1_STA_0.Ack_M633 )
   END_RUNG
   // the same network as SCL:
   "DB341_M_UNIT_1_STA_0".M_CODES_UNIT_1_STA_0.Ack_M633 := "DB2710_U1_F3_GRIPPER".CYL.FULL_OPEN;
END_REGION

REGION Network 92: M633-FIXTURE 3 GRIPPER OPEN ONLY PRESSURE SWITCH / M111-AXIAL LOCATOR RETURN FIXTURE 1
   RUNG wire#powerrail
      Contact( "DB331_EXTENDED_M_CODE_UNIT_1_STA_0".M_code[633] )
      wire#w1
      I_Contact( "DB341_M_UNIT_1_STA_0".M_CODES_UNIT_1_STA_0.Ack_M633 )
      I_Contact( "DB2120_MPP_ITC_IPC".RESET_FAULTS )
      I_Contact( "DB341_M_UNIT_1_STA_0".M_CODES_UNIT_1_STA_0.M_RESET_PULSE )
      Coil( "DB341_M_UNIT_1_STA_0".M_CODES_UNIT_1_STA_0.M633 )
   END_RUNG
   RUNG wire#powerrail
      Contact( "DB341_M_UNIT_1_STA_0".M_CODES_UNIT_1_STA_0.M633 )
   END_RUNG wire#w1
   // the same network as SCL:
   "DB341_M_UNIT_1_STA_0".M_CODES_UNIT_1_STA_0.M633 := ("DB331_EXTENDED_M_CODE_UNIT_1_STA_0".M_code[633] OR "DB341_M_UNIT_1_STA_0".M_CODES_UNIT_1_STA_0.M633) AND NOT "DB341_M_UNIT_1_STA_0".M_CODES_UNIT_1_STA_0.Ack_M633 AND NOT "DB2120_MPP_ITC_IPC".RESET_FAULTS AND NOT "DB341_M_UNIT_1_STA_0".M_CODES_UNIT_1_STA_0.M_RESET_PULSE;
END_REGION

REGION Network 93: ACKNOWLEDGE M634-FIXTURE 3 GRIPPER RELEASE PRESSURE ONLY PRESSURE SWITCH (READ-IN DISABLE) / ACKNOWLEDGE M112-AXIAL LOCATOR RELAX FIXTURE 1
   RUNG wire#powerrail
      Contact( "DB2710_U1_F3_GRIPPER".PRESSURE_RELEASED )
      Coil( "DB341_M_UNIT_1_STA_0".M_CODES_UNIT_1_STA_0.Ack_M634 )
   END_RUNG
   // the same network as SCL:
   "DB341_M_UNIT_1_STA_0".M_CODES_UNIT_1_STA_0.Ack_M634 := "DB2710_U1_F3_GRIPPER".PRESSURE_RELEASED;
END_REGION

REGION Network 94: M634-FIXTURE 3 GRIPPER RELEASE PRESSURE ONLY PRESSURE SWITCH (READ-IN DISABLE) / M112-AXIAL LOCATOR RELAX FIXTURE 1
   RUNG wire#powerrail
      Contact( "DB331_EXTENDED_M_CODE_UNIT_1_STA_0".M_code[634] )
      wire#w1
      I_Contact( "DB341_M_UNIT_1_STA_0".M_CODES_UNIT_1_STA_0.Ack_M634 )
      I_Contact( "DB2120_MPP_ITC_IPC".RESET_FAULTS )
      I_Contact( "DB341_M_UNIT_1_STA_0".M_CODES_UNIT_1_STA_0.M_RESET_PULSE )
      Coil( "DB341_M_UNIT_1_STA_0".M_CODES_UNIT_1_STA_0.M634 )
   END_RUNG
   RUNG wire#powerrail
      Contact( "DB341_M_UNIT_1_STA_0".M_CODES_UNIT_1_STA_0.M634 )
   END_RUNG wire#w1
   // the same network as SCL:
   "DB341_M_UNIT_1_STA_0".M_CODES_UNIT_1_STA_0.M634 := ("DB331_EXTENDED_M_CODE_UNIT_1_STA_0".M_code[634] OR "DB341_M_UNIT_1_STA_0".M_CODES_UNIT_1_STA_0.M634) AND NOT "DB341_M_UNIT_1_STA_0".M_CODES_UNIT_1_STA_0.Ack_M634 AND NOT "DB2120_MPP_ITC_IPC".RESET_FAULTS AND NOT "DB341_M_UNIT_1_STA_0".M_CODES_UNIT_1_STA_0.M_RESET_PULSE;
END_REGION

REGION Network 95: ACKNOWLEDGE M635-FIXTURE 3 GRIPPER RELEASE PRESSURE ONLY PRESSURE SWITCH / ACKNOWLEDGE M23-SWITCH ON SPINDLE FRAME BLOWING
   RUNG wire#powerrail
      Contact( "DB2710_U1_F3_GRIPPER".CYL.FULL_LOW_PRESSURED )
      Coil( "DB341_M_UNIT_1_STA_0".M_CODES_UNIT_1_STA_0.Ack_M635 )
   END_RUNG
   // the same network as SCL:
   "DB341_M_UNIT_1_STA_0".M_CODES_UNIT_1_STA_0.Ack_M635 := "DB2710_U1_F3_GRIPPER".CYL.FULL_LOW_PRESSURED;
END_REGION

REGION Network 96: M635-FIXTURE 3 GRIPPER RELEASE PRESSURE ONLY PRESSURE SWITCH / M23-SWITCH ON SPINDLE FRAME BLOWING
   RUNG wire#powerrail
      Contact( "DB331_EXTENDED_M_CODE_UNIT_1_STA_0".M_code[635] )
      wire#w1
      I_Contact( "DB341_M_UNIT_1_STA_0".M_CODES_UNIT_1_STA_0.Ack_M635 )
      I_Contact( "DB2120_MPP_ITC_IPC".RESET_FAULTS )
      I_Contact( "DB341_M_UNIT_1_STA_0".M_CODES_UNIT_1_STA_0.M_RESET_PULSE )
      Coil( "DB341_M_UNIT_1_STA_0".M_CODES_UNIT_1_STA_0.M635 )
   END_RUNG
   RUNG wire#powerrail
      Contact( "DB341_M_UNIT_1_STA_0".M_CODES_UNIT_1_STA_0.M635 )
   END_RUNG wire#w1
   // the same network as SCL:
   "DB341_M_UNIT_1_STA_0".M_CODES_UNIT_1_STA_0.M635 := ("DB331_EXTENDED_M_CODE_UNIT_1_STA_0".M_code[635] OR "DB341_M_UNIT_1_STA_0".M_CODES_UNIT_1_STA_0.M635) AND NOT "DB341_M_UNIT_1_STA_0".M_CODES_UNIT_1_STA_0.Ack_M635 AND NOT "DB2120_MPP_ITC_IPC".RESET_FAULTS AND NOT "DB341_M_UNIT_1_STA_0".M_CODES_UNIT_1_STA_0.M_RESET_PULSE;
END_REGION

REGION Network 97: READ-IN DISABLE / Read-in disable
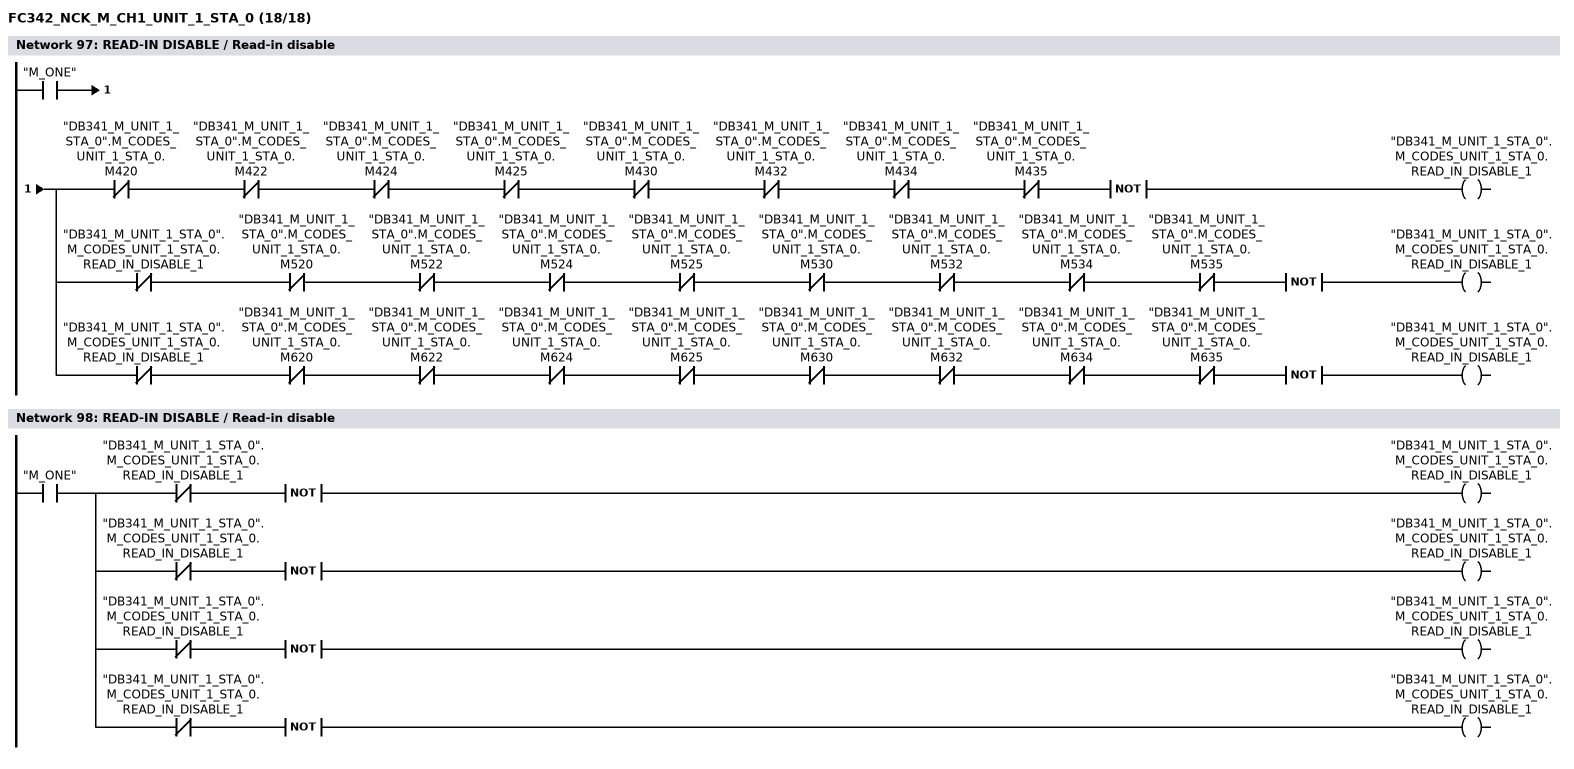
   RUNG wire#powerrail
      Contact( "M_ONE" )
      wire#w1
      I_Contact( "DB341_M_UNIT_1_STA_0".M_CODES_UNIT_1_STA_0.M420 )
      I_Contact( "DB341_M_UNIT_1_STA_0".M_CODES_UNIT_1_STA_0.M422 )
      I_Contact( "DB341_M_UNIT_1_STA_0".M_CODES_UNIT_1_STA_0.M424 )
      I_Contact( "DB341_M_UNIT_1_STA_0".M_CODES_UNIT_1_STA_0.M425 )
      I_Contact( "DB341_M_UNIT_1_STA_0".M_CODES_UNIT_1_STA_0.M430 )
      I_Contact( "DB341_M_UNIT_1_STA_0".M_CODES_UNIT_1_STA_0.M432 )
      I_Contact( "DB341_M_UNIT_1_STA_0".M_CODES_UNIT_1_STA_0.M434 )
      I_Contact( "DB341_M_UNIT_1_STA_0".M_CODES_UNIT_1_STA_0.M435 )
      Not()
      Coil( "DB341_M_UNIT_1_STA_0".M_CODES_UNIT_1_STA_0.READ_IN_DISABLE_1 )
   END_RUNG
   RUNG wire#w1
      I_Contact( "DB341_M_UNIT_1_STA_0".M_CODES_UNIT_1_STA_0.READ_IN_DISABLE_1 )
      I_Contact( "DB341_M_UNIT_1_STA_0".M_CODES_UNIT_1_STA_0.M520 )
      I_Contact( "DB341_M_UNIT_1_STA_0".M_CODES_UNIT_1_STA_0.M522 )
      I_Contact( "DB341_M_UNIT_1_STA_0".M_CODES_UNIT_1_STA_0.M524 )
      I_Contact( "DB341_M_UNIT_1_STA_0".M_CODES_UNIT_1_STA_0.M525 )
      I_Contact( "DB341_M_UNIT_1_STA_0".M_CODES_UNIT_1_STA_0.M530 )
      I_Contact( "DB341_M_UNIT_1_STA_0".M_CODES_UNIT_1_STA_0.M532 )
      I_Contact( "DB341_M_UNIT_1_STA_0".M_CODES_UNIT_1_STA_0.M534 )
      I_Contact( "DB341_M_UNIT_1_STA_0".M_CODES_UNIT_1_STA_0.M535 )
      Not()
      Coil( "DB341_M_UNIT_1_STA_0".M_CODES_UNIT_1_STA_0.READ_IN_DISABLE_1 )
   END_RUNG
   RUNG wire#w1
      I_Contact( "DB341_M_UNIT_1_STA_0".M_CODES_UNIT_1_STA_0.READ_IN_DISABLE_1 )
      I_Contact( "DB341_M_UNIT_1_STA_0".M_CODES_UNIT_1_STA_0.M620 )
      I_Contact( "DB341_M_UNIT_1_STA_0".M_CODES_UNIT_1_STA_0.M622 )
      I_Contact( "DB341_M_UNIT_1_STA_0".M_CODES_UNIT_1_STA_0.M624 )
      I_Contact( "DB341_M_UNIT_1_STA_0".M_CODES_UNIT_1_STA_0.M625 )
      I_Contact( "DB341_M_UNIT_1_STA_0".M_CODES_UNIT_1_STA_0.M630 )
      I_Contact( "DB341_M_UNIT_1_STA_0".M_CODES_UNIT_1_STA_0.M632 )
      I_Contact( "DB341_M_UNIT_1_STA_0".M_CODES_UNIT_1_STA_0.M634 )
      I_Contact( "DB341_M_UNIT_1_STA_0".M_CODES_UNIT_1_STA_0.M635 )
      Not()
      Coil( "DB341_M_UNIT_1_STA_0".M_CODES_UNIT_1_STA_0.READ_IN_DISABLE_1 )
   END_RUNG
   // the same network as SCL:
   "DB341_M_UNIT_1_STA_0".M_CODES_UNIT_1_STA_0.READ_IN_DISABLE_1 := NOT ("M_ONE" AND NOT "DB341_M_UNIT_1_STA_0".M_CODES_UNIT_1_STA_0.M420 AND NOT "DB341_M_UNIT_1_STA_0".M_CODES_UNIT_1_STA_0.M422 AND NOT "DB341_M_UNIT_1_STA_0".M_CODES_UNIT_1_STA_0.M424 AND NOT "DB341_M_UNIT_1_STA_0".M_CODES_UNIT_1_STA_0.M425 AND NOT "DB341_M_UNIT_1_STA_0".M_CODES_UNIT_1_STA_0.M430 AND NOT "DB341_M_UNIT_1_STA_0".M_CODES_UNIT_1_STA_0.M432 AND NOT "DB341_M_UNIT_1_STA_0".M_CODES_UNIT_1_STA_0.M434 AND NOT "DB341_M_UNIT_1_STA_0".M_CODES_UNIT_1_STA_0.M435);
   "DB341_M_UNIT_1_STA_0".M_CODES_UNIT_1_STA_0.READ_IN_DISABLE_1 := NOT ("M_ONE" AND NOT "DB341_M_UNIT_1_STA_0".M_CODES_UNIT_1_STA_0.READ_IN_DISABLE_1 AND NOT "DB341_M_UNIT_1_STA_0".M_CODES_UNIT_1_STA_0.M520 AND NOT "DB341_M_UNIT_1_STA_0".M_CODES_UNIT_1_STA_0.M522 AND NOT "DB341_M_UNIT_1_STA_0".M_CODES_UNIT_1_STA_0.M524 AND NOT "DB341_M_UNIT_1_STA_0".M_CODES_UNIT_1_STA_0.M525 AND NOT "DB341_M_UNIT_1_STA_0".M_CODES_UNIT_1_STA_0.M530 AND NOT "DB341_M_UNIT_1_STA_0".M_CODES_UNIT_1_STA_0.M532 AND NOT "DB341_M_UNIT_1_STA_0".M_CODES_UNIT_1_STA_0.M534 AND NOT "DB341_M_UNIT_1_STA_0".M_CODES_UNIT_1_STA_0.M535);
   "DB341_M_UNIT_1_STA_0".M_CODES_UNIT_1_STA_0.READ_IN_DISABLE_1 := NOT ("M_ONE" AND NOT "DB341_M_UNIT_1_STA_0".M_CODES_UNIT_1_STA_0.READ_IN_DISABLE_1 AND NOT "DB341_M_UNIT_1_STA_0".M_CODES_UNIT_1_STA_0.M620 AND NOT "DB341_M_UNIT_1_STA_0".M_CODES_UNIT_1_STA_0.M622 AND NOT "DB341_M_UNIT_1_STA_0".M_CODES_UNIT_1_STA_0.M624 AND NOT "DB341_M_UNIT_1_STA_0".M_CODES_UNIT_1_STA_0.M625 AND NOT "DB341_M_UNIT_1_STA_0".M_CODES_UNIT_1_STA_0.M630 AND NOT "DB341_M_UNIT_1_STA_0".M_CODES_UNIT_1_STA_0.M632 AND NOT "DB341_M_UNIT_1_STA_0".M_CODES_UNIT_1_STA_0.M634 AND NOT "DB341_M_UNIT_1_STA_0".M_CODES_UNIT_1_STA_0.M635);
END_REGION

REGION Network 98: READ-IN DISABLE / Read-in disable
   RUNG wire#powerrail
      Contact( "M_ONE" )
      wire#w1
      I_Contact( "DB341_M_UNIT_1_STA_0".M_CODES_UNIT_1_STA_0.READ_IN_DISABLE_1 )
      Not()
      Coil( "DB341_M_UNIT_1_STA_0".M_CODES_UNIT_1_STA_0.READ_IN_DISABLE_1 )
   END_RUNG
   RUNG wire#w1
      I_Contact( "DB341_M_UNIT_1_STA_0".M_CODES_UNIT_1_STA_0.READ_IN_DISABLE_1 )
      Not()
      Coil( "DB341_M_UNIT_1_STA_0".M_CODES_UNIT_1_STA_0.READ_IN_DISABLE_1 )
   END_RUNG
   RUNG wire#w1
      I_Contact( "DB341_M_UNIT_1_STA_0".M_CODES_UNIT_1_STA_0.READ_IN_DISABLE_1 )
      Not()
      Coil( "DB341_M_UNIT_1_STA_0".M_CODES_UNIT_1_STA_0.READ_IN_DISABLE_1 )
   END_RUNG
   RUNG wire#w1
      I_Contact( "DB341_M_UNIT_1_STA_0".M_CODES_UNIT_1_STA_0.READ_IN_DISABLE_1 )
      Not()
      Coil( "DB341_M_UNIT_1_STA_0".M_CODES_UNIT_1_STA_0.READ_IN_DISABLE_1 )
   END_RUNG
   // the same network as SCL:
   "DB341_M_UNIT_1_STA_0".M_CODES_UNIT_1_STA_0.READ_IN_DISABLE_1 := NOT ("M_ONE" AND NOT "DB341_M_UNIT_1_STA_0".M_CODES_UNIT_1_STA_0.READ_IN_DISABLE_1);
   "DB341_M_UNIT_1_STA_0".M_CODES_UNIT_1_STA_0.READ_IN_DISABLE_1 := NOT ("M_ONE" AND NOT "DB341_M_UNIT_1_STA_0".M_CODES_UNIT_1_STA_0.READ_IN_DISABLE_1);
   "DB341_M_UNIT_1_STA_0".M_CODES_UNIT_1_STA_0.READ_IN_DISABLE_1 := NOT ("M_ONE" AND NOT "DB341_M_UNIT_1_STA_0".M_CODES_UNIT_1_STA_0.READ_IN_DISABLE_1);
   "DB341_M_UNIT_1_STA_0".M_CODES_UNIT_1_STA_0.READ_IN_DISABLE_1 := NOT ("M_ONE" AND NOT "DB341_M_UNIT_1_STA_0".M_CODES_UNIT_1_STA_0.READ_IN_DISABLE_1);
END_REGION
END_FUNCTION
